// TIA Portal V17 export
// export: Created 2025-03-10T13:10:32.0915737Z, ExportSetting WithDefaults, DisplayName Totally Integrated Automation Portal, DisplayVersion V17 Update 8, DisplayName TIA Portal Openness, DisplayVersion V17 Update 8, DisplayName TIA Portal Version Control Interface, DisplayVersion V17, DisplayName SINAMICS Startdrive Advanced, DisplayVersion V17 SP2, DisplayName SINAMICS Startdrive G110M, G120, G120C, G120D, G120P, G115D, DisplayVersion V17 SP2, DisplayName SINAMICS Startdrive G130, G150, S120, S150, SINAMICS MV, S210, DisplayVersion V17 SP2, DisplayName STEP 7 Professional, DisplayVersion V17 Update 8, DisplayName SINUMERIK ONE STEP 7 Toolbox, DisplayVersion V17 Update 12, DisplayName SINUMERIK 840D sl STEP 7 Toolbox, DisplayVersion V17 Update 12, DisplayName STEP 7 Safety, DisplayVersion V17 Update 6, DisplayName WinCC Advanced, DisplayVersion V17 Update 8
FUNCTION "FC32_CLADDING_AXES" : Void   // FC32, LAD
{ S7_Optimized_Access := 'FALSE' }
AUTHOR : ETXETAR
VERSION : 1.0
// stored: AutoNumber false, IsIECCheckEnabled false, SetENOAutomatically false, UDAEnableTagReadback false
   VAR_TEMP
      O_BLOCKING_DEV_C : Bool;   // OPTION BLOCKING DEVICE FOR C AXIS
      AUX_1 : Real;
      POSITION_TO_GO_AUX : Real;
   END_VAR
   VAR_TEMP   // added for the SCL form of the ladder/FBD networks
      _w1 : Bool;
      _w2 : Bool;
   END_VAR
BEGIN

REGION Network 1: AXIS E10 MOVE AXIS AND FEED HOLD CONDITIONS
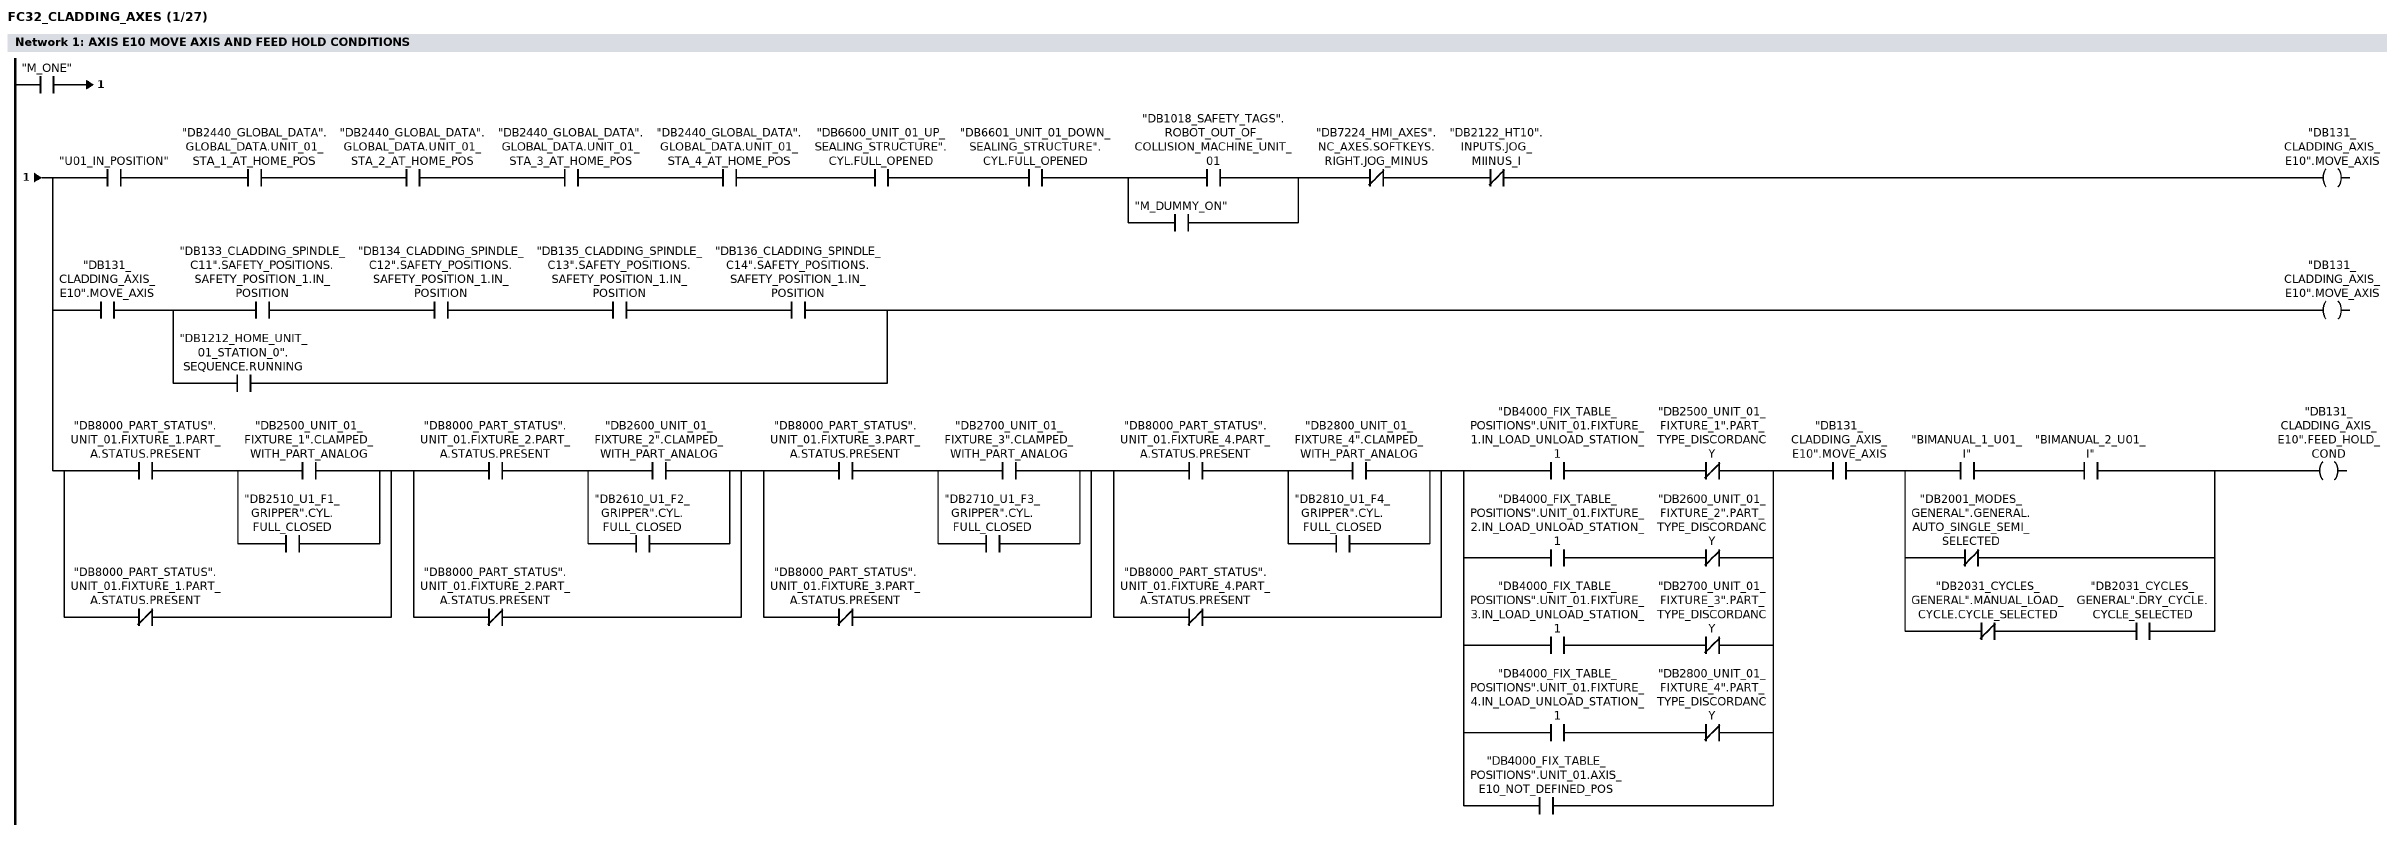
   RUNG wire#powerrail
      Contact( "M_ONE" )
      wire#w1
      Contact( "U01_IN_POSITION" )
      Contact( "DB2440_GLOBAL_DATA".GLOBAL_DATA.UNIT_01_STA_1_AT_HOME_POS )
      Contact( "DB2440_GLOBAL_DATA".GLOBAL_DATA.UNIT_01_STA_2_AT_HOME_POS )
      Contact( "DB2440_GLOBAL_DATA".GLOBAL_DATA.UNIT_01_STA_3_AT_HOME_POS )
      Contact( "DB2440_GLOBAL_DATA".GLOBAL_DATA.UNIT_01_STA_4_AT_HOME_POS )
      Contact( "DB6600_UNIT_01_UP_SEALING_STRUCTURE".CYL.FULL_OPENED )
      Contact( "DB6601_UNIT_01_DOWN_SEALING_STRUCTURE".CYL.FULL_OPENED )
      wire#w2
      Contact( "DB1018_SAFETY_TAGS".ROBOT_OUT_OF_COLLISION_MACHINE_UNIT_01 )
      wire#w3
      I_Contact( "DB7224_HMI_AXES".NC_AXES.SOFTKEYS.RIGHT.JOG_MINUS )
      I_Contact( "DB2122_HT10".INPUTS.JOG_MIINUS_I )
      Coil( "DB131_CLADDING_AXIS_E10".MOVE_AXIS )
   END_RUNG
   RUNG wire#w2
      Contact( "M_DUMMY_ON" )
   END_RUNG wire#w3
   RUNG wire#w1
      Contact( "DB131_CLADDING_AXIS_E10".MOVE_AXIS )
      wire#w4
      Contact( "DB133_CLADDING_SPINDLE_C11".SAFETY_POSITIONS.SAFETY_POSITION_1.IN_POSITION )
      Contact( "DB134_CLADDING_SPINDLE_C12".SAFETY_POSITIONS.SAFETY_POSITION_1.IN_POSITION )
      Contact( "DB135_CLADDING_SPINDLE_C13".SAFETY_POSITIONS.SAFETY_POSITION_1.IN_POSITION )
      Contact( "DB136_CLADDING_SPINDLE_C14".SAFETY_POSITIONS.SAFETY_POSITION_1.IN_POSITION )
      wire#w5
      Coil( "DB131_CLADDING_AXIS_E10".MOVE_AXIS )
   END_RUNG
   RUNG wire#w4
      Contact( "DB1212_HOME_UNIT_01_STATION_0".SEQUENCE.RUNNING )
   END_RUNG wire#w5
   RUNG wire#w1
      Contact( "DB8000_PART_STATUS".UNIT_01.FIXTURE_1.PART_A.STATUS.PRESENT )
      wire#w6
      Contact( "DB2500_UNIT_01_FIXTURE_1".CLAMPED_WITH_PART_ANALOG )
      wire#w7
      Contact( "DB8000_PART_STATUS".UNIT_01.FIXTURE_2.PART_A.STATUS.PRESENT )
      wire#w8
      Contact( "DB2600_UNIT_01_FIXTURE_2".CLAMPED_WITH_PART_ANALOG )
      wire#w9
      Contact( "DB8000_PART_STATUS".UNIT_01.FIXTURE_3.PART_A.STATUS.PRESENT )
      wire#w10
      Contact( "DB2700_UNIT_01_FIXTURE_3".CLAMPED_WITH_PART_ANALOG )
      wire#w11
      Contact( "DB8000_PART_STATUS".UNIT_01.FIXTURE_4.PART_A.STATUS.PRESENT )
      wire#w12
      Contact( "DB2800_UNIT_01_FIXTURE_4".CLAMPED_WITH_PART_ANALOG )
      wire#w13
      Contact( "DB4000_FIX_TABLE_POSITIONS".UNIT_01.FIXTURE_1.IN_LOAD_UNLOAD_STATION_1 )
      I_Contact( "DB2500_UNIT_01_FIXTURE_1".PART_TYPE_DISCORDANCY )
      wire#w14
      Contact( "DB131_CLADDING_AXIS_E10".MOVE_AXIS )
      wire#w15
      Contact( "BIMANUAL_1_U01_I" )
      Contact( "BIMANUAL_2_U01_I" )
      wire#w16
      Coil( "DB131_CLADDING_AXIS_E10".FEED_HOLD_COND )
   END_RUNG
   RUNG wire#w6
      Contact( "DB2510_U1_F1_GRIPPER".CYL.FULL_CLOSED )
   END_RUNG wire#w7
   RUNG wire#w1
      I_Contact( "DB8000_PART_STATUS".UNIT_01.FIXTURE_1.PART_A.STATUS.PRESENT )
   END_RUNG wire#w7
   RUNG wire#w8
      Contact( "DB2610_U1_F2_GRIPPER".CYL.FULL_CLOSED )
   END_RUNG wire#w9
   RUNG wire#w7
      I_Contact( "DB8000_PART_STATUS".UNIT_01.FIXTURE_2.PART_A.STATUS.PRESENT )
   END_RUNG wire#w9
   RUNG wire#w10
      Contact( "DB2710_U1_F3_GRIPPER".CYL.FULL_CLOSED )
   END_RUNG wire#w11
   RUNG wire#w9
      I_Contact( "DB8000_PART_STATUS".UNIT_01.FIXTURE_3.PART_A.STATUS.PRESENT )
   END_RUNG wire#w11
   RUNG wire#w12
      Contact( "DB2810_U1_F4_GRIPPER".CYL.FULL_CLOSED )
   END_RUNG wire#w13
   RUNG wire#w11
      I_Contact( "DB8000_PART_STATUS".UNIT_01.FIXTURE_4.PART_A.STATUS.PRESENT )
   END_RUNG wire#w13
   RUNG wire#w13
      Contact( "DB4000_FIX_TABLE_POSITIONS".UNIT_01.FIXTURE_2.IN_LOAD_UNLOAD_STATION_1 )
      I_Contact( "DB2600_UNIT_01_FIXTURE_2".PART_TYPE_DISCORDANCY )
   END_RUNG wire#w14
   RUNG wire#w13
      Contact( "DB4000_FIX_TABLE_POSITIONS".UNIT_01.FIXTURE_3.IN_LOAD_UNLOAD_STATION_1 )
      I_Contact( "DB2700_UNIT_01_FIXTURE_3".PART_TYPE_DISCORDANCY )
   END_RUNG wire#w14
   RUNG wire#w13
      Contact( "DB4000_FIX_TABLE_POSITIONS".UNIT_01.FIXTURE_4.IN_LOAD_UNLOAD_STATION_1 )
      I_Contact( "DB2800_UNIT_01_FIXTURE_4".PART_TYPE_DISCORDANCY )
   END_RUNG wire#w14
   RUNG wire#w13
      Contact( "DB4000_FIX_TABLE_POSITIONS".UNIT_01.AXIS_E10_NOT_DEFINED_POS )
   END_RUNG wire#w14
   RUNG wire#w15
      I_Contact( "DB2001_MODES_GENERAL".GENERAL.AUTO_SINGLE_SEMI_SELECTED )
   END_RUNG wire#w16
   RUNG wire#w15
      I_Contact( "DB2031_CYCLES_GENERAL".MANUAL_LOAD_CYCLE.CYCLE_SELECTED )
      Contact( "DB2031_CYCLES_GENERAL".DRY_CYCLE.CYCLE_SELECTED )
   END_RUNG wire#w16
   // the same network as SCL:
   "DB131_CLADDING_AXIS_E10".MOVE_AXIS := "M_ONE" AND "U01_IN_POSITION" AND "DB2440_GLOBAL_DATA".GLOBAL_DATA.UNIT_01_STA_1_AT_HOME_POS AND "DB2440_GLOBAL_DATA".GLOBAL_DATA.UNIT_01_STA_2_AT_HOME_POS AND "DB2440_GLOBAL_DATA".GLOBAL_DATA.UNIT_01_STA_3_AT_HOME_POS AND "DB2440_GLOBAL_DATA".GLOBAL_DATA.UNIT_01_STA_4_AT_HOME_POS AND "DB6600_UNIT_01_UP_SEALING_STRUCTURE".CYL.FULL_OPENED AND "DB6601_UNIT_01_DOWN_SEALING_STRUCTURE".CYL.FULL_OPENED AND ("DB1018_SAFETY_TAGS".ROBOT_OUT_OF_COLLISION_MACHINE_UNIT_01 OR "M_DUMMY_ON") AND NOT "DB7224_HMI_AXES".NC_AXES.SOFTKEYS.RIGHT.JOG_MINUS AND NOT "DB2122_HT10".INPUTS.JOG_MIINUS_I;
   "DB131_CLADDING_AXIS_E10".MOVE_AXIS := "M_ONE" AND "DB131_CLADDING_AXIS_E10".MOVE_AXIS AND (("DB133_CLADDING_SPINDLE_C11".SAFETY_POSITIONS.SAFETY_POSITION_1.IN_POSITION AND "DB134_CLADDING_SPINDLE_C12".SAFETY_POSITIONS.SAFETY_POSITION_1.IN_POSITION AND "DB135_CLADDING_SPINDLE_C13".SAFETY_POSITIONS.SAFETY_POSITION_1.IN_POSITION AND "DB136_CLADDING_SPINDLE_C14".SAFETY_POSITIONS.SAFETY_POSITION_1.IN_POSITION) OR "DB1212_HOME_UNIT_01_STATION_0".SEQUENCE.RUNNING);
   "DB131_CLADDING_AXIS_E10".FEED_HOLD_COND := "M_ONE" AND (("DB8000_PART_STATUS".UNIT_01.FIXTURE_1.PART_A.STATUS.PRESENT AND ("DB2500_UNIT_01_FIXTURE_1".CLAMPED_WITH_PART_ANALOG OR "DB2510_U1_F1_GRIPPER".CYL.FULL_CLOSED)) OR NOT "DB8000_PART_STATUS".UNIT_01.FIXTURE_1.PART_A.STATUS.PRESENT) AND (("DB8000_PART_STATUS".UNIT_01.FIXTURE_2.PART_A.STATUS.PRESENT AND ("DB2600_UNIT_01_FIXTURE_2".CLAMPED_WITH_PART_ANALOG OR "DB2610_U1_F2_GRIPPER".CYL.FULL_CLOSED)) OR NOT "DB8000_PART_STATUS".UNIT_01.FIXTURE_2.PART_A.STATUS.PRESENT) AND (("DB8000_PART_STATUS".UNIT_01.FIXTURE_3.PART_A.STATUS.PRESENT AND ("DB2700_UNIT_01_FIXTURE_3".CLAMPED_WITH_PART_ANALOG OR "DB2710_U1_F3_GRIPPER".CYL.FULL_CLOSED)) OR NOT "DB8000_PART_STATUS".UNIT_01.FIXTURE_3.PART_A.STATUS.PRESENT) AND (("DB8000_PART_STATUS".UNIT_01.FIXTURE_4.PART_A.STATUS.PRESENT AND ("DB2800_UNIT_01_FIXTURE_4".CLAMPED_WITH_PART_ANALOG OR "DB2810_U1_F4_GRIPPER".CYL.FULL_CLOSED)) OR NOT "DB8000_PART_STATUS".UNIT_01.FIXTURE_4.PART_A.STATUS.PRESENT) AND (("DB4000_FIX_TABLE_POSITIONS".UNIT_01.FIXTURE_1.IN_LOAD_UNLOAD_STATION_1 AND NOT "DB2500_UNIT_01_FIXTURE_1".PART_TYPE_DISCORDANCY) OR ("DB4000_FIX_TABLE_POSITIONS".UNIT_01.FIXTURE_2.IN_LOAD_UNLOAD_STATION_1 AND NOT "DB2600_UNIT_01_FIXTURE_2".PART_TYPE_DISCORDANCY) OR ("DB4000_FIX_TABLE_POSITIONS".UNIT_01.FIXTURE_3.IN_LOAD_UNLOAD_STATION_1 AND NOT "DB2700_UNIT_01_FIXTURE_3".PART_TYPE_DISCORDANCY) OR ("DB4000_FIX_TABLE_POSITIONS".UNIT_01.FIXTURE_4.IN_LOAD_UNLOAD_STATION_1 AND NOT "DB2800_UNIT_01_FIXTURE_4".PART_TYPE_DISCORDANCY) OR "DB4000_FIX_TABLE_POSITIONS".UNIT_01.AXIS_E10_NOT_DEFINED_POS) AND "DB131_CLADDING_AXIS_E10".MOVE_AXIS AND (("BIMANUAL_1_U01_I" AND "BIMANUAL_2_U01_I") OR NOT "DB2001_MODES_GENERAL".GENERAL.AUTO_SINGLE_SEMI_SELECTED OR (NOT "DB2031_CYCLES_GENERAL".MANUAL_LOAD_CYCLE.CYCLE_SELECTED AND "DB2031_CYCLES_GENERAL".DRY_CYCLE.CYCLE_SELECTED));
END_REGION

REGION Network 2: CALL FB32 AXIS E10
   // 2#0000_0001 OPTIONS 0 BIT 0 MEASURING SYSTEM 2 OPTION
   // 2#0000_0010 OPTIONS 0 BIT 1 ENABLE FC18 OPTION
   // 2#0000_0100 OPTIONS 0 BIT 2 FC18 EXTERNAL POSITION OPTION
   // 2#0000_1000 OPTIONS 0 BIT 3 AXIS B ENABLE FAULTS OPTION
   // 2#0001_0000 OPTIONS 0 BIT 4 SPARE OPTION
   // 2#0010_0000 OPTIONS 0 BIT 5 SPARE OPTION
   // 2#0100_0000 OPTIONS 0 BIT 6 SPARE OPTION
   // 2#1000_0000 OPTIONS 0 BIT 7 SPARE OPTION
   // 
   // 2#0000_0001 OPTIONS 1 BIT 0 AXIS ROLLER OPTION
   // 2#0000_0010 OPTIONS 1 BIT 1 MASTER AXIS OPTION
   // 2#0000_0100 OPTIONS 1 BIT 2 SLAVE AXIS OPTION
   // 2#0000_1000 OPTIONS 1 BIT 3 MASTER-SLAVE AXES INDEPENDENT MOVEMENT WITH HT10 OPTION
   // 2#0001_0000 OPTIONS 1 BIT 4 GANTRY MODE MASTER AXIS OPTION
   // 2#0010_0000 OPTIONS 1 BIT 5 SPARE OPTION
   // 2#0100_0000 OPTIONS 1 BIT 6 SPARE OPTION
   // 2#1000_0000 OPTIONS 1 BIT 7 SPARE OPTION
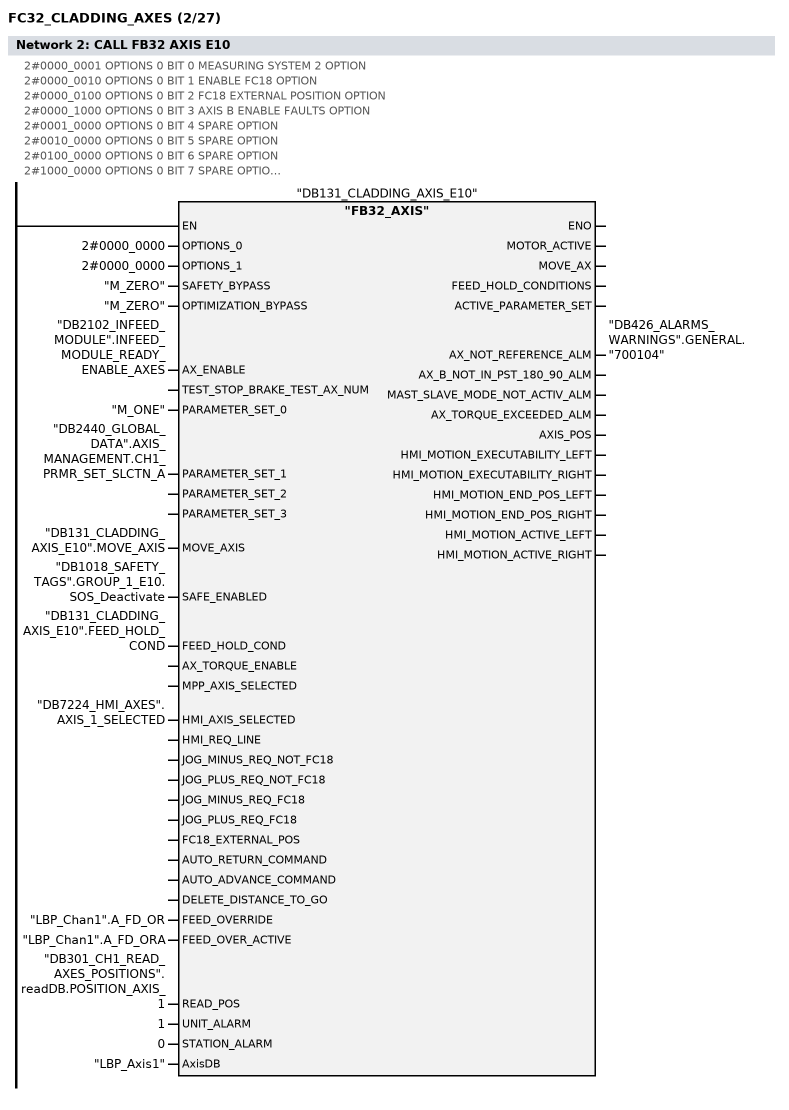
   RUNG wire#powerrail
      "DB131_CLADDING_AXIS_E10"(OPTIONS_0 := 2#0000_0000, OPTIONS_1 := 2#0000_0000, SAFETY_BYPASS := "M_ZERO", OPTIMIZATION_BYPASS := "M_ZERO", AX_ENABLE := "DB2102_INFEED_MODULE".INFEED_MODULE_READY_ENABLE_AXES, TEST_STOP_BRAKE_TEST_AX_NUM :=, PARAMETER_SET_0 := "M_ONE", PARAMETER_SET_1 := "DB2440_GLOBAL_DATA".AXIS_MANAGEMENT.CH1_PRMR_SET_SLCTN_A, PARAMETER_SET_2 :=, PARAMETER_SET_3 :=, MOVE_AXIS := "DB131_CLADDING_AXIS_E10".MOVE_AXIS, SAFE_ENABLED := "DB1018_SAFETY_TAGS".GROUP_1_E10.SOS_Deactivate, FEED_HOLD_COND := "DB131_CLADDING_AXIS_E10".FEED_HOLD_COND, AX_TORQUE_ENABLE :=, MPP_AXIS_SELECTED :=, HMI_AXIS_SELECTED := "DB7224_HMI_AXES".AXIS_1_SELECTED, HMI_REQ_LINE :=, JOG_MINUS_REQ_NOT_FC18 :=, JOG_PLUS_REQ_NOT_FC18 :=, JOG_MINUS_REQ_FC18 :=, JOG_PLUS_REQ_FC18 :=, FC18_EXTERNAL_POS :=, AUTO_RETURN_COMMAND :=, AUTO_ADVANCE_COMMAND :=, DELETE_DISTANCE_TO_GO :=, FEED_OVERRIDE := "LBP_Chan1".A_FD_OR, FEED_OVER_ACTIVE := "LBP_Chan1".A_FD_ORA, READ_POS := "DB301_CH1_READ_AXES_POSITIONS".readDB.POSITION_AXIS_1, UNIT_ALARM := 1, STATION_ALARM := 0, AxisDB := "LBP_Axis1", MOTOR_ACTIVE =>, MOVE_AX =>, FEED_HOLD_CONDITIONS =>, ACTIVE_PARAMETER_SET =>, AX_NOT_REFERENCE_ALM => "DB426_ALARMS_WARNINGS".GENERAL."700104", AX_B_NOT_IN_PST_180_90_ALM =>, MAST_SLAVE_MODE_NOT_ACTIV_ALM =>, AX_TORQUE_EXCEEDED_ALM =>, AXIS_POS =>, HMI_MOTION_EXECUTABILITY_LEFT =>, HMI_MOTION_EXECUTABILITY_RIGHT =>, HMI_MOTION_END_POS_LEFT =>, HMI_MOTION_END_POS_RIGHT =>, HMI_MOTION_ACTIVE_LEFT =>, HMI_MOTION_ACTIVE_RIGHT =>)
   END_RUNG
   // the same network as SCL:
   "DB131_CLADDING_AXIS_E10"(OPTIONS_0 := 2#0000_0000,   // "FB32_AXIS"
                           OPTIONS_1 := 2#0000_0000,
                           SAFETY_BYPASS := "M_ZERO",
                           OPTIMIZATION_BYPASS := "M_ZERO",
                           AX_ENABLE := "DB2102_INFEED_MODULE".INFEED_MODULE_READY_ENABLE_AXES,
                           PARAMETER_SET_0 := "M_ONE",
                           PARAMETER_SET_1 := "DB2440_GLOBAL_DATA".AXIS_MANAGEMENT.CH1_PRMR_SET_SLCTN_A,
                           MOVE_AXIS := "DB131_CLADDING_AXIS_E10".MOVE_AXIS,
                           SAFE_ENABLED := "DB1018_SAFETY_TAGS".GROUP_1_E10.SOS_Deactivate,
                           FEED_HOLD_COND := "DB131_CLADDING_AXIS_E10".FEED_HOLD_COND,
                           HMI_AXIS_SELECTED := "DB7224_HMI_AXES".AXIS_1_SELECTED,
                           FEED_OVERRIDE := "LBP_Chan1".A_FD_OR,
                           FEED_OVER_ACTIVE := "LBP_Chan1".A_FD_ORA,
                           READ_POS := "DB301_CH1_READ_AXES_POSITIONS".readDB.POSITION_AXIS_1,
                           UNIT_ALARM := 1,
                           STATION_ALARM := 0,
                           AxisDB := "LBP_Axis1",
                           AX_NOT_REFERENCE_ALM => "DB426_ALARMS_WARNINGS".GENERAL."700104");
END_REGION

REGION Network 3: AXIS E10 OPERATOR HELP
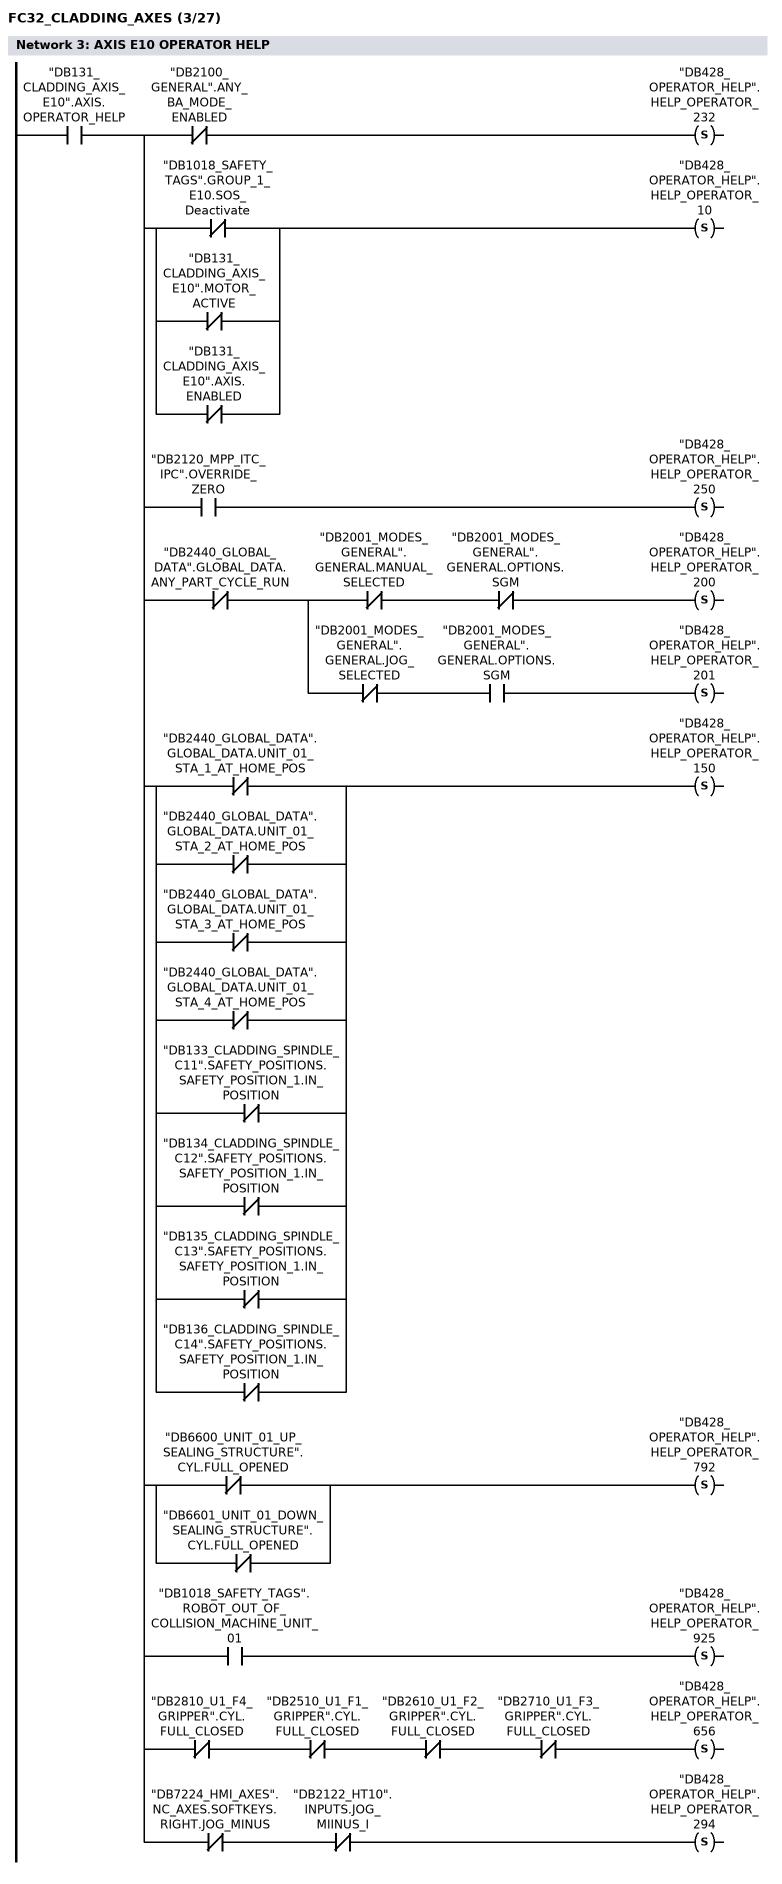
   RUNG wire#powerrail
      Contact( "DB131_CLADDING_AXIS_E10".AXIS.OPERATOR_HELP )
      wire#w1
      I_Contact( "DB2100_GENERAL".ANY_BA_MODE_ENABLED )
      S_Coil( "DB428_OPERATOR_HELP".HELP_OPERATOR_232 )
   END_RUNG
   RUNG wire#w1
      I_Contact( "DB1018_SAFETY_TAGS".GROUP_1_E10.SOS_Deactivate )
      wire#w2
      S_Coil( "DB428_OPERATOR_HELP".HELP_OPERATOR_10 )
   END_RUNG
   RUNG wire#w1
      I_Contact( "DB131_CLADDING_AXIS_E10".MOTOR_ACTIVE )
   END_RUNG wire#w2
   RUNG wire#w1
      I_Contact( "DB131_CLADDING_AXIS_E10".AXIS.ENABLED )
   END_RUNG wire#w2
   RUNG wire#w1
      Contact( "DB2120_MPP_ITC_IPC".OVERRIDE_ZERO )
      S_Coil( "DB428_OPERATOR_HELP".HELP_OPERATOR_250 )
   END_RUNG
   RUNG wire#w1
      I_Contact( "DB2440_GLOBAL_DATA".GLOBAL_DATA.ANY_PART_CYCLE_RUN )
      wire#w3
      I_Contact( "DB2001_MODES_GENERAL".GENERAL.MANUAL_SELECTED )
      I_Contact( "DB2001_MODES_GENERAL".GENERAL.OPTIONS.SGM )
      S_Coil( "DB428_OPERATOR_HELP".HELP_OPERATOR_200 )
   END_RUNG
   RUNG wire#w3
      I_Contact( "DB2001_MODES_GENERAL".GENERAL.JOG_SELECTED )
      Contact( "DB2001_MODES_GENERAL".GENERAL.OPTIONS.SGM )
      S_Coil( "DB428_OPERATOR_HELP".HELP_OPERATOR_201 )
   END_RUNG
   RUNG wire#w1
      I_Contact( "DB2440_GLOBAL_DATA".GLOBAL_DATA.UNIT_01_STA_1_AT_HOME_POS )
      wire#w4
      S_Coil( "DB428_OPERATOR_HELP".HELP_OPERATOR_150 )
   END_RUNG
   RUNG wire#w1
      I_Contact( "DB2440_GLOBAL_DATA".GLOBAL_DATA.UNIT_01_STA_2_AT_HOME_POS )
   END_RUNG wire#w4
   RUNG wire#w1
      I_Contact( "DB2440_GLOBAL_DATA".GLOBAL_DATA.UNIT_01_STA_3_AT_HOME_POS )
   END_RUNG wire#w4
   RUNG wire#w1
      I_Contact( "DB2440_GLOBAL_DATA".GLOBAL_DATA.UNIT_01_STA_4_AT_HOME_POS )
   END_RUNG wire#w4
   RUNG wire#w1
      I_Contact( "DB133_CLADDING_SPINDLE_C11".SAFETY_POSITIONS.SAFETY_POSITION_1.IN_POSITION )
   END_RUNG wire#w4
   RUNG wire#w1
      I_Contact( "DB134_CLADDING_SPINDLE_C12".SAFETY_POSITIONS.SAFETY_POSITION_1.IN_POSITION )
   END_RUNG wire#w4
   RUNG wire#w1
      I_Contact( "DB135_CLADDING_SPINDLE_C13".SAFETY_POSITIONS.SAFETY_POSITION_1.IN_POSITION )
   END_RUNG wire#w4
   RUNG wire#w1
      I_Contact( "DB136_CLADDING_SPINDLE_C14".SAFETY_POSITIONS.SAFETY_POSITION_1.IN_POSITION )
   END_RUNG wire#w4
   RUNG wire#w1
      I_Contact( "DB6600_UNIT_01_UP_SEALING_STRUCTURE".CYL.FULL_OPENED )
      wire#w5
      S_Coil( "DB428_OPERATOR_HELP".HELP_OPERATOR_792 )
   END_RUNG
   RUNG wire#w1
      I_Contact( "DB6601_UNIT_01_DOWN_SEALING_STRUCTURE".CYL.FULL_OPENED )
   END_RUNG wire#w5
   RUNG wire#w1
      Contact( "DB1018_SAFETY_TAGS".ROBOT_OUT_OF_COLLISION_MACHINE_UNIT_01 )
      S_Coil( "DB428_OPERATOR_HELP".HELP_OPERATOR_925 )
   END_RUNG
   RUNG wire#w1
      I_Contact( "DB2810_U1_F4_GRIPPER".CYL.FULL_CLOSED )
      I_Contact( "DB2510_U1_F1_GRIPPER".CYL.FULL_CLOSED )
      I_Contact( "DB2610_U1_F2_GRIPPER".CYL.FULL_CLOSED )
      I_Contact( "DB2710_U1_F3_GRIPPER".CYL.FULL_CLOSED )
      S_Coil( "DB428_OPERATOR_HELP".HELP_OPERATOR_656 )
   END_RUNG
   RUNG wire#w1
      I_Contact( "DB7224_HMI_AXES".NC_AXES.SOFTKEYS.RIGHT.JOG_MINUS )
      I_Contact( "DB2122_HT10".INPUTS.JOG_MIINUS_I )
      S_Coil( "DB428_OPERATOR_HELP".HELP_OPERATOR_294 )
   END_RUNG
   // the same network as SCL:
   IF "DB131_CLADDING_AXIS_E10".AXIS.OPERATOR_HELP AND NOT "DB2100_GENERAL".ANY_BA_MODE_ENABLED THEN
       "DB428_OPERATOR_HELP".HELP_OPERATOR_232 := TRUE;
   END_IF;
   IF "DB131_CLADDING_AXIS_E10".AXIS.OPERATOR_HELP AND (NOT "DB1018_SAFETY_TAGS".GROUP_1_E10.SOS_Deactivate OR NOT "DB131_CLADDING_AXIS_E10".MOTOR_ACTIVE OR NOT "DB131_CLADDING_AXIS_E10".AXIS.ENABLED) THEN
       "DB428_OPERATOR_HELP".HELP_OPERATOR_10 := TRUE;
   END_IF;
   IF "DB131_CLADDING_AXIS_E10".AXIS.OPERATOR_HELP AND "DB2120_MPP_ITC_IPC".OVERRIDE_ZERO THEN
       "DB428_OPERATOR_HELP".HELP_OPERATOR_250 := TRUE;
   END_IF;
   #_w1 := "DB131_CLADDING_AXIS_E10".AXIS.OPERATOR_HELP AND NOT "DB2440_GLOBAL_DATA".GLOBAL_DATA.ANY_PART_CYCLE_RUN;
   IF #_w1 AND NOT "DB2001_MODES_GENERAL".GENERAL.MANUAL_SELECTED AND NOT "DB2001_MODES_GENERAL".GENERAL.OPTIONS.SGM THEN
       "DB428_OPERATOR_HELP".HELP_OPERATOR_200 := TRUE;
   END_IF;
   IF #_w1 AND NOT "DB2001_MODES_GENERAL".GENERAL.JOG_SELECTED AND "DB2001_MODES_GENERAL".GENERAL.OPTIONS.SGM THEN
       "DB428_OPERATOR_HELP".HELP_OPERATOR_201 := TRUE;
   END_IF;
   IF "DB131_CLADDING_AXIS_E10".AXIS.OPERATOR_HELP AND (NOT "DB2440_GLOBAL_DATA".GLOBAL_DATA.UNIT_01_STA_1_AT_HOME_POS OR NOT "DB2440_GLOBAL_DATA".GLOBAL_DATA.UNIT_01_STA_2_AT_HOME_POS OR NOT "DB2440_GLOBAL_DATA".GLOBAL_DATA.UNIT_01_STA_3_AT_HOME_POS OR NOT "DB2440_GLOBAL_DATA".GLOBAL_DATA.UNIT_01_STA_4_AT_HOME_POS OR NOT "DB133_CLADDING_SPINDLE_C11".SAFETY_POSITIONS.SAFETY_POSITION_1.IN_POSITION OR NOT "DB134_CLADDING_SPINDLE_C12".SAFETY_POSITIONS.SAFETY_POSITION_1.IN_POSITION OR NOT "DB135_CLADDING_SPINDLE_C13".SAFETY_POSITIONS.SAFETY_POSITION_1.IN_POSITION OR NOT "DB136_CLADDING_SPINDLE_C14".SAFETY_POSITIONS.SAFETY_POSITION_1.IN_POSITION) THEN
       "DB428_OPERATOR_HELP".HELP_OPERATOR_150 := TRUE;
   END_IF;
   IF "DB131_CLADDING_AXIS_E10".AXIS.OPERATOR_HELP AND (NOT "DB6600_UNIT_01_UP_SEALING_STRUCTURE".CYL.FULL_OPENED OR NOT "DB6601_UNIT_01_DOWN_SEALING_STRUCTURE".CYL.FULL_OPENED) THEN
       "DB428_OPERATOR_HELP".HELP_OPERATOR_792 := TRUE;
   END_IF;
   IF "DB131_CLADDING_AXIS_E10".AXIS.OPERATOR_HELP AND "DB1018_SAFETY_TAGS".ROBOT_OUT_OF_COLLISION_MACHINE_UNIT_01 THEN
       "DB428_OPERATOR_HELP".HELP_OPERATOR_925 := TRUE;
   END_IF;
   IF "DB131_CLADDING_AXIS_E10".AXIS.OPERATOR_HELP AND NOT "DB2810_U1_F4_GRIPPER".CYL.FULL_CLOSED AND NOT "DB2510_U1_F1_GRIPPER".CYL.FULL_CLOSED AND NOT "DB2610_U1_F2_GRIPPER".CYL.FULL_CLOSED AND NOT "DB2710_U1_F3_GRIPPER".CYL.FULL_CLOSED THEN
       "DB428_OPERATOR_HELP".HELP_OPERATOR_656 := TRUE;
   END_IF;
   IF "DB131_CLADDING_AXIS_E10".AXIS.OPERATOR_HELP AND NOT "DB7224_HMI_AXES".NC_AXES.SOFTKEYS.RIGHT.JOG_MINUS AND NOT "DB2122_HT10".INPUTS.JOG_MIINUS_I THEN
       "DB428_OPERATOR_HELP".HELP_OPERATOR_294 := TRUE;
   END_IF;
END_REGION

REGION Network 4: AXIS X13 MOVE AXIS AND FEED HOLD CONDITIONS
   // AÑADIR QUE TODO ESTE CONECTADO
   // DISCO AMARRADO
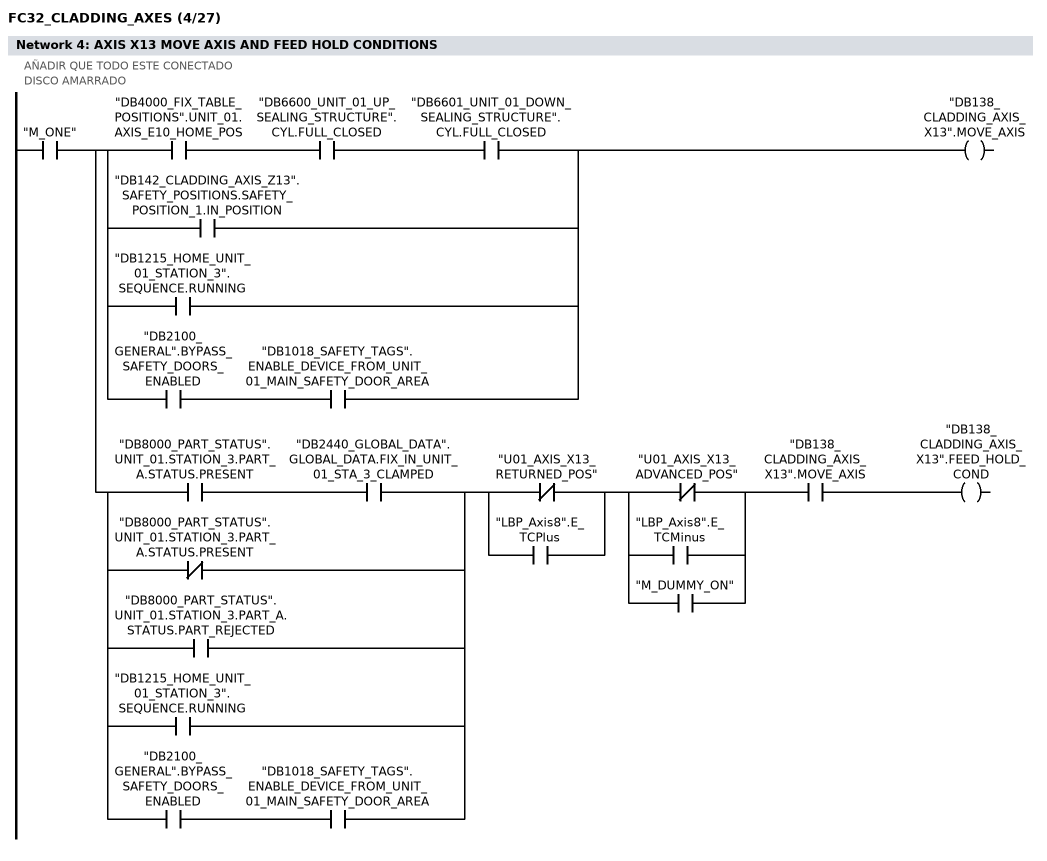
   RUNG wire#powerrail
      Contact( "M_ONE" )
      wire#w1
      Contact( "DB4000_FIX_TABLE_POSITIONS".UNIT_01.AXIS_E10_HOME_POS )
      Contact( "DB6600_UNIT_01_UP_SEALING_STRUCTURE".CYL.FULL_CLOSED )
      Contact( "DB6601_UNIT_01_DOWN_SEALING_STRUCTURE".CYL.FULL_CLOSED )
      wire#w2
      Coil( "DB138_CLADDING_AXIS_X13".MOVE_AXIS )
   END_RUNG
   RUNG wire#w1
      Contact( "DB142_CLADDING_AXIS_Z13".SAFETY_POSITIONS.SAFETY_POSITION_1.IN_POSITION )
   END_RUNG wire#w2
   RUNG wire#w1
      Contact( "DB1215_HOME_UNIT_01_STATION_3".SEQUENCE.RUNNING )
   END_RUNG wire#w2
   RUNG wire#w1
      Contact( "DB2100_GENERAL".BYPASS_SAFETY_DOORS_ENABLED )
      Contact( "DB1018_SAFETY_TAGS".ENABLE_DEVICE_FROM_UNIT_01_MAIN_SAFETY_DOOR_AREA )
   END_RUNG wire#w2
   RUNG wire#w1
      Contact( "DB8000_PART_STATUS".UNIT_01.STATION_3.PART_A.STATUS.PRESENT )
      Contact( "DB2440_GLOBAL_DATA".GLOBAL_DATA.FIX_IN_UNIT_01_STA_3_CLAMPED )
      wire#w3
      I_Contact( "U01_AXIS_X13_RETURNED_POS" )
      wire#w4
      I_Contact( "U01_AXIS_X13_ADVANCED_POS" )
      wire#w5
      Contact( "DB138_CLADDING_AXIS_X13".MOVE_AXIS )
      Coil( "DB138_CLADDING_AXIS_X13".FEED_HOLD_COND )
   END_RUNG
   RUNG wire#w1
      I_Contact( "DB8000_PART_STATUS".UNIT_01.STATION_3.PART_A.STATUS.PRESENT )
   END_RUNG wire#w3
   RUNG wire#w1
      Contact( "DB8000_PART_STATUS".UNIT_01.STATION_3.PART_A.STATUS.PART_REJECTED )
   END_RUNG wire#w3
   RUNG wire#w1
      Contact( "DB1215_HOME_UNIT_01_STATION_3".SEQUENCE.RUNNING )
   END_RUNG wire#w3
   RUNG wire#w1
      Contact( "DB2100_GENERAL".BYPASS_SAFETY_DOORS_ENABLED )
      Contact( "DB1018_SAFETY_TAGS".ENABLE_DEVICE_FROM_UNIT_01_MAIN_SAFETY_DOOR_AREA )
   END_RUNG wire#w3
   RUNG wire#w3
      Contact( "LBP_Axis8".E_TCPlus )
   END_RUNG wire#w4
   RUNG wire#w4
      Contact( "LBP_Axis8".E_TCMinus )
   END_RUNG wire#w5
   RUNG wire#w4
      Contact( "M_DUMMY_ON" )
   END_RUNG wire#w5
   // the same network as SCL:
   "DB138_CLADDING_AXIS_X13".MOVE_AXIS := "M_ONE" AND (("DB4000_FIX_TABLE_POSITIONS".UNIT_01.AXIS_E10_HOME_POS AND "DB6600_UNIT_01_UP_SEALING_STRUCTURE".CYL.FULL_CLOSED AND "DB6601_UNIT_01_DOWN_SEALING_STRUCTURE".CYL.FULL_CLOSED) OR "DB142_CLADDING_AXIS_Z13".SAFETY_POSITIONS.SAFETY_POSITION_1.IN_POSITION OR "DB1215_HOME_UNIT_01_STATION_3".SEQUENCE.RUNNING OR ("DB2100_GENERAL".BYPASS_SAFETY_DOORS_ENABLED AND "DB1018_SAFETY_TAGS".ENABLE_DEVICE_FROM_UNIT_01_MAIN_SAFETY_DOOR_AREA));
   "DB138_CLADDING_AXIS_X13".FEED_HOLD_COND := "M_ONE" AND (("DB8000_PART_STATUS".UNIT_01.STATION_3.PART_A.STATUS.PRESENT AND "DB2440_GLOBAL_DATA".GLOBAL_DATA.FIX_IN_UNIT_01_STA_3_CLAMPED) OR NOT "DB8000_PART_STATUS".UNIT_01.STATION_3.PART_A.STATUS.PRESENT OR "DB8000_PART_STATUS".UNIT_01.STATION_3.PART_A.STATUS.PART_REJECTED OR "DB1215_HOME_UNIT_01_STATION_3".SEQUENCE.RUNNING OR ("DB2100_GENERAL".BYPASS_SAFETY_DOORS_ENABLED AND "DB1018_SAFETY_TAGS".ENABLE_DEVICE_FROM_UNIT_01_MAIN_SAFETY_DOOR_AREA)) AND (NOT "U01_AXIS_X13_RETURNED_POS" OR "LBP_Axis8".E_TCPlus) AND (NOT "U01_AXIS_X13_ADVANCED_POS" OR "LBP_Axis8".E_TCMinus OR "M_DUMMY_ON") AND "DB138_CLADDING_AXIS_X13".MOVE_AXIS;
END_REGION

REGION Network 5: CALL FB32 AXIS X13
   // 2#0000_0001 OPTIONS 0 BIT 0 MEASURING SYSTEM 2 OPTION
   // 2#0000_0010 OPTIONS 0 BIT 1 ENABLE FC18 OPTION
   // 2#0000_0100 OPTIONS 0 BIT 2 FC18 EXTERNAL POSITION OPTION
   // 2#0000_1000 OPTIONS 0 BIT 3 AXIS B ENABLE FAULTS OPTION
   // 2#0001_0000 OPTIONS 0 BIT 4 SPARE OPTION
   // 2#0010_0000 OPTIONS 0 BIT 5 SPARE OPTION
   // 2#0100_0000 OPTIONS 0 BIT 6 SPARE OPTION
   // 2#1000_0000 OPTIONS 0 BIT 7 SPARE OPTION
   // 
   // 2#0000_0001 OPTIONS 1 BIT 0 AXIS ROLLER OPTION
   // 2#0000_0010 OPTIONS 1 BIT 1 MASTER AXIS OPTION
   // 2#0000_0100 OPTIONS 1 BIT 2 SLAVE AXIS OPTION
   // 2#0000_1000 OPTIONS 1 BIT 3 MASTER-SLAVE AXES INDEPENDENT MOVEMENT WITH HT10 OPTION
   // 2#0001_0000 OPTIONS 1 BIT 4 GANTRY MODE MASTER AXIS OPTION
   // 2#0010_0000 OPTIONS 1 BIT 5 SPARE OPTION
   // 2#0100_0000 OPTIONS 1 BIT 6 SPARE OPTION
   // 2#1000_0000 OPTIONS 1 BIT 7 SPARE OPTION
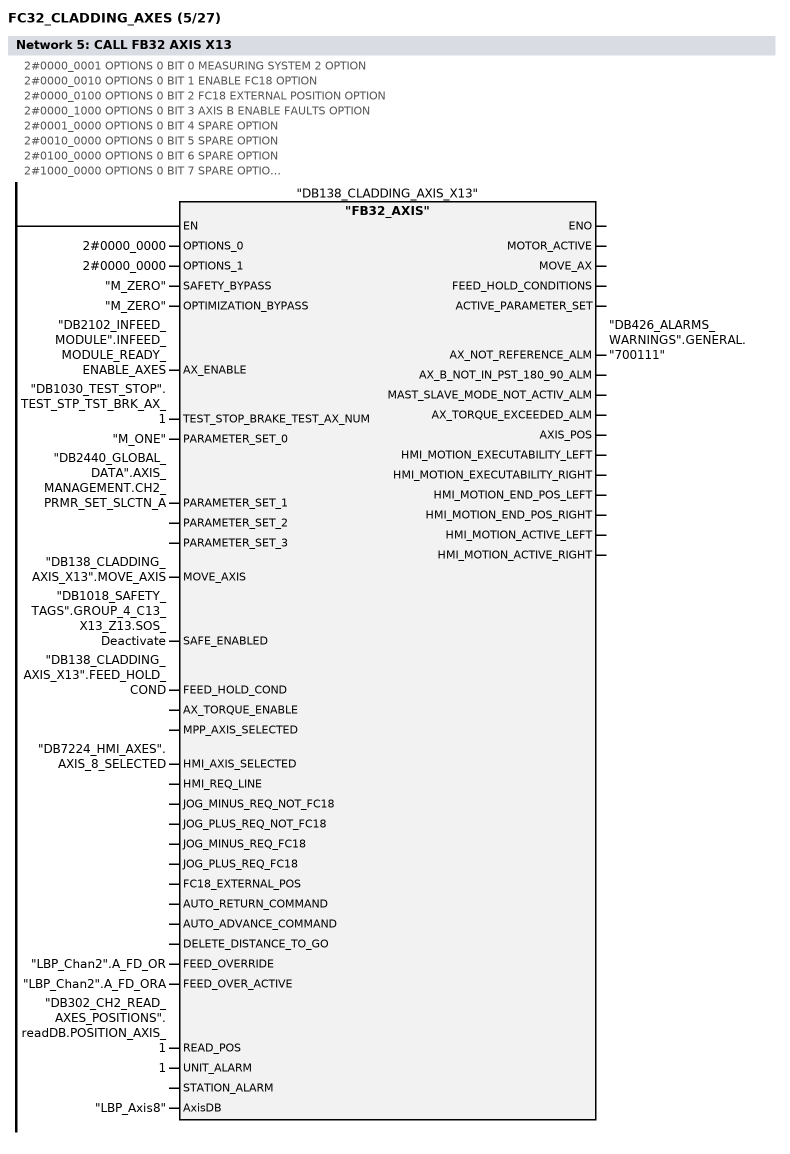
   RUNG wire#powerrail
      "DB138_CLADDING_AXIS_X13"(OPTIONS_0 := 2#0000_0000, OPTIONS_1 := 2#0000_0000, SAFETY_BYPASS := "M_ZERO", OPTIMIZATION_BYPASS := "M_ZERO", AX_ENABLE := "DB2102_INFEED_MODULE".INFEED_MODULE_READY_ENABLE_AXES, TEST_STOP_BRAKE_TEST_AX_NUM := "DB1030_TEST_STOP".TEST_STP_TST_BRK_AX_1, PARAMETER_SET_0 := "M_ONE", PARAMETER_SET_1 := "DB2440_GLOBAL_DATA".AXIS_MANAGEMENT.CH2_PRMR_SET_SLCTN_A, PARAMETER_SET_2 :=, PARAMETER_SET_3 :=, MOVE_AXIS := "DB138_CLADDING_AXIS_X13".MOVE_AXIS, SAFE_ENABLED := "DB1018_SAFETY_TAGS".GROUP_4_C13_X13_Z13.SOS_Deactivate, FEED_HOLD_COND := "DB138_CLADDING_AXIS_X13".FEED_HOLD_COND, AX_TORQUE_ENABLE :=, MPP_AXIS_SELECTED :=, HMI_AXIS_SELECTED := "DB7224_HMI_AXES".AXIS_8_SELECTED, HMI_REQ_LINE :=, JOG_MINUS_REQ_NOT_FC18 :=, JOG_PLUS_REQ_NOT_FC18 :=, JOG_MINUS_REQ_FC18 :=, JOG_PLUS_REQ_FC18 :=, FC18_EXTERNAL_POS :=, AUTO_RETURN_COMMAND :=, AUTO_ADVANCE_COMMAND :=, DELETE_DISTANCE_TO_GO :=, FEED_OVERRIDE := "LBP_Chan2".A_FD_OR, FEED_OVER_ACTIVE := "LBP_Chan2".A_FD_ORA, READ_POS := "DB302_CH2_READ_AXES_POSITIONS".readDB.POSITION_AXIS_1, UNIT_ALARM := 1, STATION_ALARM :=, AxisDB := "LBP_Axis8", MOTOR_ACTIVE =>, MOVE_AX =>, FEED_HOLD_CONDITIONS =>, ACTIVE_PARAMETER_SET =>, AX_NOT_REFERENCE_ALM => "DB426_ALARMS_WARNINGS".GENERAL."700111", AX_B_NOT_IN_PST_180_90_ALM =>, MAST_SLAVE_MODE_NOT_ACTIV_ALM =>, AX_TORQUE_EXCEEDED_ALM =>, AXIS_POS =>, HMI_MOTION_EXECUTABILITY_LEFT =>, HMI_MOTION_EXECUTABILITY_RIGHT =>, HMI_MOTION_END_POS_LEFT =>, HMI_MOTION_END_POS_RIGHT =>, HMI_MOTION_ACTIVE_LEFT =>, HMI_MOTION_ACTIVE_RIGHT =>)
   END_RUNG
   // the same network as SCL:
   "DB138_CLADDING_AXIS_X13"(OPTIONS_0 := 2#0000_0000,   // "FB32_AXIS"
                           OPTIONS_1 := 2#0000_0000,
                           SAFETY_BYPASS := "M_ZERO",
                           OPTIMIZATION_BYPASS := "M_ZERO",
                           AX_ENABLE := "DB2102_INFEED_MODULE".INFEED_MODULE_READY_ENABLE_AXES,
                           TEST_STOP_BRAKE_TEST_AX_NUM := "DB1030_TEST_STOP".TEST_STP_TST_BRK_AX_1,
                           PARAMETER_SET_0 := "M_ONE",
                           PARAMETER_SET_1 := "DB2440_GLOBAL_DATA".AXIS_MANAGEMENT.CH2_PRMR_SET_SLCTN_A,
                           MOVE_AXIS := "DB138_CLADDING_AXIS_X13".MOVE_AXIS,
                           SAFE_ENABLED := "DB1018_SAFETY_TAGS".GROUP_4_C13_X13_Z13.SOS_Deactivate,
                           FEED_HOLD_COND := "DB138_CLADDING_AXIS_X13".FEED_HOLD_COND,
                           HMI_AXIS_SELECTED := "DB7224_HMI_AXES".AXIS_8_SELECTED,
                           FEED_OVERRIDE := "LBP_Chan2".A_FD_OR,
                           FEED_OVER_ACTIVE := "LBP_Chan2".A_FD_ORA,
                           READ_POS := "DB302_CH2_READ_AXES_POSITIONS".readDB.POSITION_AXIS_1,
                           UNIT_ALARM := 1,
                           AxisDB := "LBP_Axis8",
                           AX_NOT_REFERENCE_ALM => "DB426_ALARMS_WARNINGS".GENERAL."700111");
END_REGION

REGION Network 6: AXIS X13 OPERATOR HELP
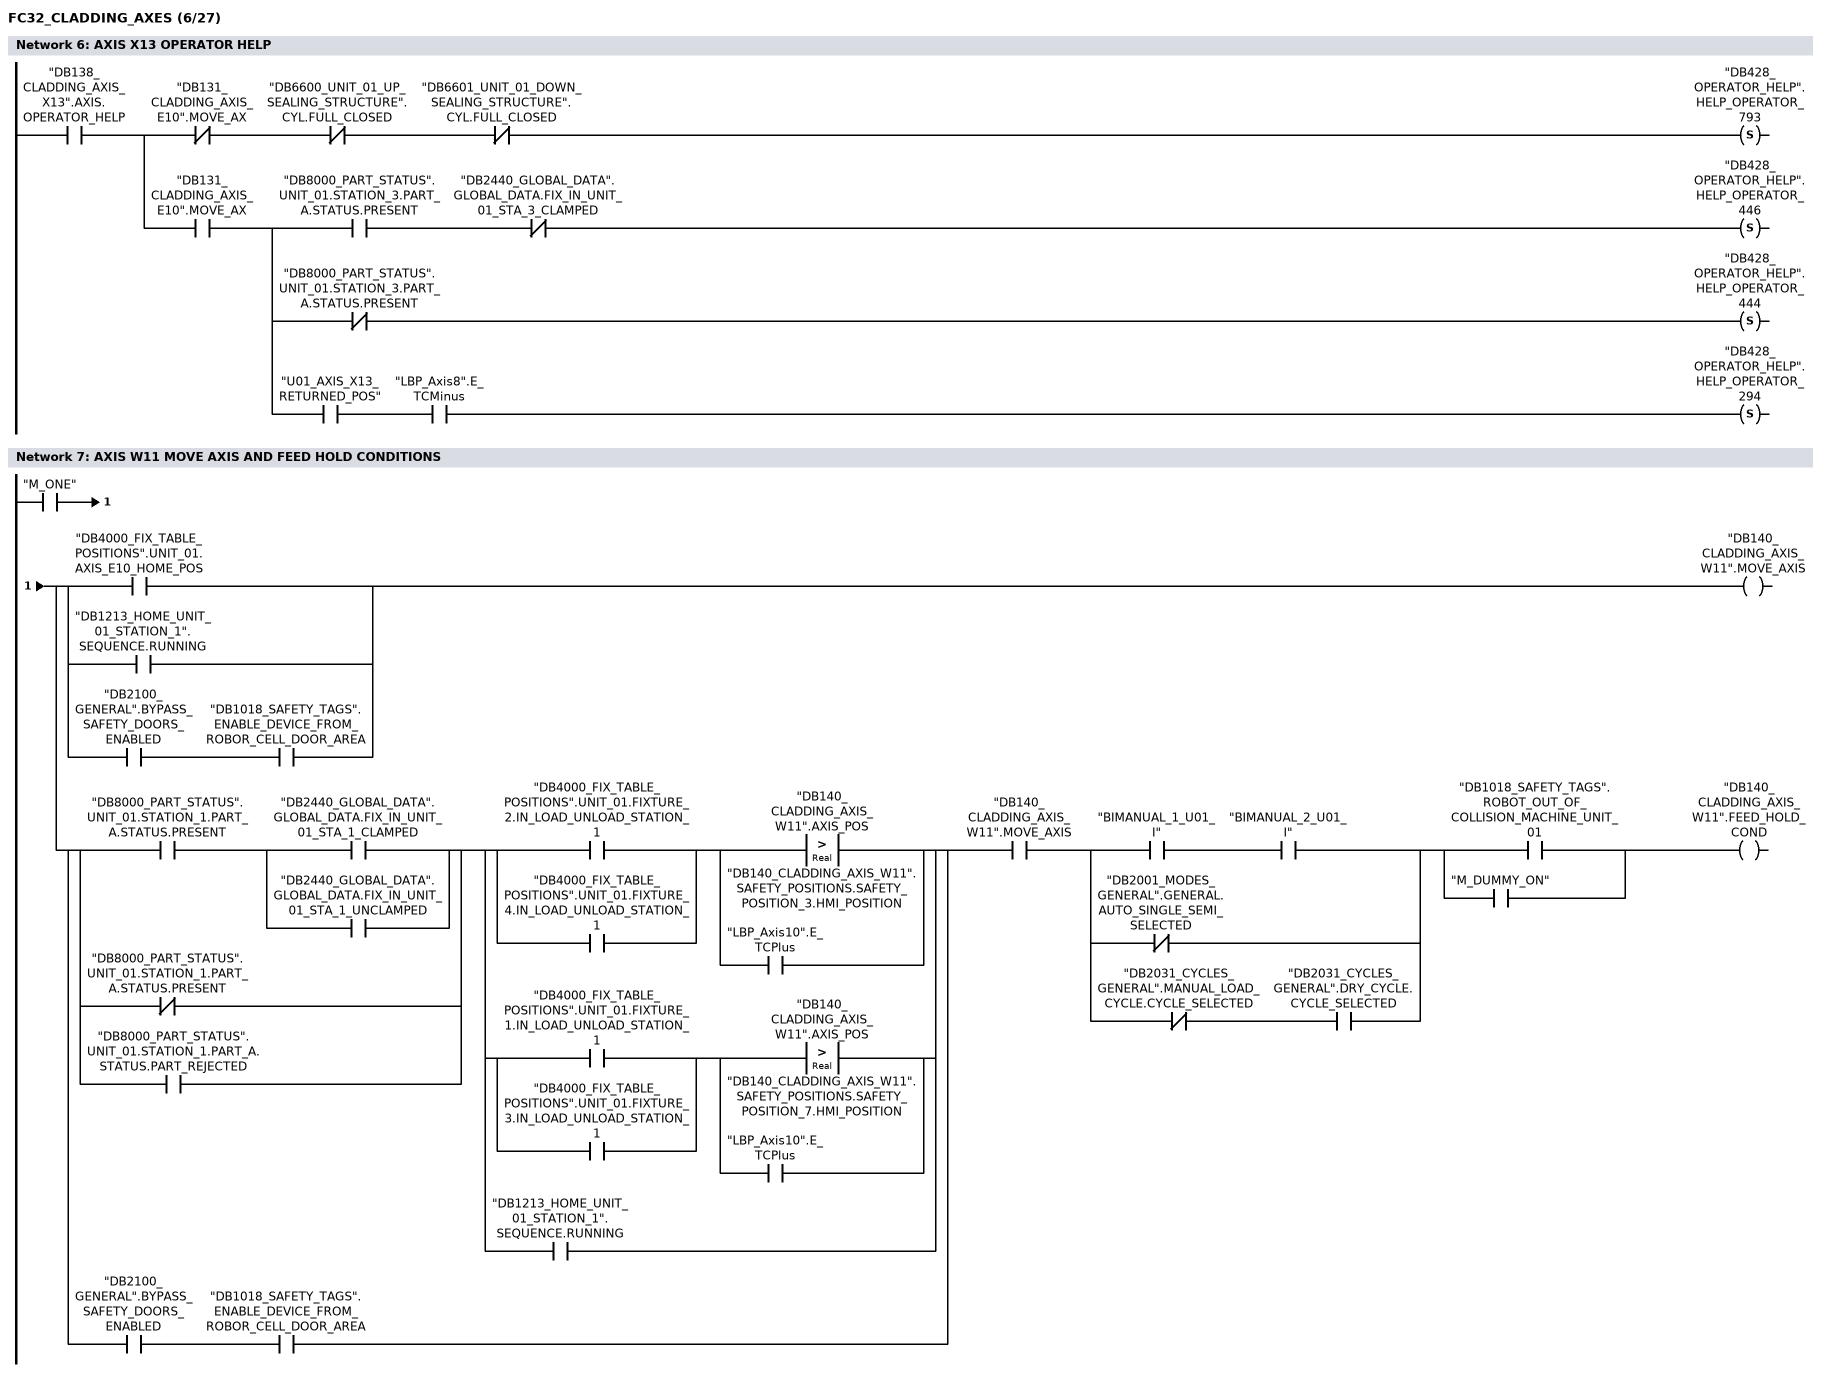
   RUNG wire#powerrail
      Contact( "DB138_CLADDING_AXIS_X13".AXIS.OPERATOR_HELP )
      wire#w1
      I_Contact( "DB131_CLADDING_AXIS_E10".MOVE_AX )
      I_Contact( "DB6600_UNIT_01_UP_SEALING_STRUCTURE".CYL.FULL_CLOSED )
      I_Contact( "DB6601_UNIT_01_DOWN_SEALING_STRUCTURE".CYL.FULL_CLOSED )
      S_Coil( "DB428_OPERATOR_HELP".HELP_OPERATOR_793 )
   END_RUNG
   RUNG wire#w1
      Contact( "DB131_CLADDING_AXIS_E10".MOVE_AX )
      wire#w2
      Contact( "DB8000_PART_STATUS".UNIT_01.STATION_3.PART_A.STATUS.PRESENT )
      I_Contact( "DB2440_GLOBAL_DATA".GLOBAL_DATA.FIX_IN_UNIT_01_STA_3_CLAMPED )
      S_Coil( "DB428_OPERATOR_HELP".HELP_OPERATOR_446 )
   END_RUNG
   RUNG wire#w2
      I_Contact( "DB8000_PART_STATUS".UNIT_01.STATION_3.PART_A.STATUS.PRESENT )
      S_Coil( "DB428_OPERATOR_HELP".HELP_OPERATOR_444 )
   END_RUNG
   RUNG wire#w2
      Contact( "U01_AXIS_X13_RETURNED_POS" )
      Contact( "LBP_Axis8".E_TCMinus )
      S_Coil( "DB428_OPERATOR_HELP".HELP_OPERATOR_294 )
   END_RUNG
   // the same network as SCL:
   IF "DB138_CLADDING_AXIS_X13".AXIS.OPERATOR_HELP AND NOT "DB131_CLADDING_AXIS_E10".MOVE_AX AND NOT "DB6600_UNIT_01_UP_SEALING_STRUCTURE".CYL.FULL_CLOSED AND NOT "DB6601_UNIT_01_DOWN_SEALING_STRUCTURE".CYL.FULL_CLOSED THEN
       "DB428_OPERATOR_HELP".HELP_OPERATOR_793 := TRUE;
   END_IF;
   #_w1 := "DB138_CLADDING_AXIS_X13".AXIS.OPERATOR_HELP AND "DB131_CLADDING_AXIS_E10".MOVE_AX;
   IF #_w1 AND "DB8000_PART_STATUS".UNIT_01.STATION_3.PART_A.STATUS.PRESENT AND NOT "DB2440_GLOBAL_DATA".GLOBAL_DATA.FIX_IN_UNIT_01_STA_3_CLAMPED THEN
       "DB428_OPERATOR_HELP".HELP_OPERATOR_446 := TRUE;
   END_IF;
   IF #_w1 AND NOT "DB8000_PART_STATUS".UNIT_01.STATION_3.PART_A.STATUS.PRESENT THEN
       "DB428_OPERATOR_HELP".HELP_OPERATOR_444 := TRUE;
   END_IF;
   IF #_w1 AND "U01_AXIS_X13_RETURNED_POS" AND "LBP_Axis8".E_TCMinus THEN
       "DB428_OPERATOR_HELP".HELP_OPERATOR_294 := TRUE;
   END_IF;
END_REGION

REGION Network 7: AXIS W11 MOVE AXIS AND FEED HOLD CONDITIONS
   RUNG wire#powerrail
      Contact( "M_ONE" )
      wire#w1
      Contact( "DB4000_FIX_TABLE_POSITIONS".UNIT_01.AXIS_E10_HOME_POS )
      wire#w2
      Coil( "DB140_CLADDING_AXIS_W11".MOVE_AXIS )
   END_RUNG
   RUNG wire#w1
      Contact( "DB1213_HOME_UNIT_01_STATION_1".SEQUENCE.RUNNING )
   END_RUNG wire#w2
   RUNG wire#w1
      Contact( "DB2100_GENERAL".BYPASS_SAFETY_DOORS_ENABLED )
      Contact( "DB1018_SAFETY_TAGS".ENABLE_DEVICE_FROM_ROBOR_CELL_DOOR_AREA )
   END_RUNG wire#w2
   RUNG wire#w1
      Contact( "DB8000_PART_STATUS".UNIT_01.STATION_1.PART_A.STATUS.PRESENT )
      wire#w3
      Contact( "DB2440_GLOBAL_DATA".GLOBAL_DATA.FIX_IN_UNIT_01_STA_1_CLAMPED )
      wire#w4
      Contact( "DB4000_FIX_TABLE_POSITIONS".UNIT_01.FIXTURE_2.IN_LOAD_UNLOAD_STATION_1 )
      wire#w5
      { S7_Templates := "SrcType := Real" } GT_Contact(in1 := "DB140_CLADDING_AXIS_W11".AXIS_POS, in2 := "DB140_CLADDING_AXIS_W11".SAFETY_POSITIONS.SAFETY_POSITION_3.HMI_POSITION)
      wire#w6
      Contact( "DB140_CLADDING_AXIS_W11".MOVE_AXIS )
      wire#w8
      Contact( "BIMANUAL_1_U01_I" )
      Contact( "BIMANUAL_2_U01_I" )
      wire#w9
      Contact( "DB1018_SAFETY_TAGS".ROBOT_OUT_OF_COLLISION_MACHINE_UNIT_01 )
      wire#w10
      Coil( "DB140_CLADDING_AXIS_W11".FEED_HOLD_COND )
   END_RUNG
   RUNG wire#w3
      Contact( "DB2440_GLOBAL_DATA".GLOBAL_DATA.FIX_IN_UNIT_01_STA_1_UNCLAMPED )
   END_RUNG wire#w4
   RUNG wire#w1
      I_Contact( "DB8000_PART_STATUS".UNIT_01.STATION_1.PART_A.STATUS.PRESENT )
   END_RUNG wire#w4
   RUNG wire#w1
      Contact( "DB8000_PART_STATUS".UNIT_01.STATION_1.PART_A.STATUS.PART_REJECTED )
   END_RUNG wire#w4
   RUNG wire#w4
      Contact( "DB4000_FIX_TABLE_POSITIONS".UNIT_01.FIXTURE_4.IN_LOAD_UNLOAD_STATION_1 )
   END_RUNG wire#w5
   RUNG wire#w5
      Contact( "LBP_Axis10".E_TCPlus )
   END_RUNG wire#w6
   RUNG wire#w4
      Contact( "DB4000_FIX_TABLE_POSITIONS".UNIT_01.FIXTURE_1.IN_LOAD_UNLOAD_STATION_1 )
      wire#w7
      { S7_Templates := "SrcType := Real" } GT_Contact(in1 := "DB140_CLADDING_AXIS_W11".AXIS_POS, in2 := "DB140_CLADDING_AXIS_W11".SAFETY_POSITIONS.SAFETY_POSITION_7.HMI_POSITION)
   END_RUNG wire#w6
   RUNG wire#w4
      Contact( "DB4000_FIX_TABLE_POSITIONS".UNIT_01.FIXTURE_3.IN_LOAD_UNLOAD_STATION_1 )
   END_RUNG wire#w7
   RUNG wire#w7
      Contact( "LBP_Axis10".E_TCPlus )
   END_RUNG wire#w6
   RUNG wire#w4
      Contact( "DB1213_HOME_UNIT_01_STATION_1".SEQUENCE.RUNNING )
   END_RUNG wire#w6
   RUNG wire#w1
      Contact( "DB2100_GENERAL".BYPASS_SAFETY_DOORS_ENABLED )
      Contact( "DB1018_SAFETY_TAGS".ENABLE_DEVICE_FROM_ROBOR_CELL_DOOR_AREA )
   END_RUNG wire#w6
   RUNG wire#w8
      I_Contact( "DB2001_MODES_GENERAL".GENERAL.AUTO_SINGLE_SEMI_SELECTED )
   END_RUNG wire#w9
   RUNG wire#w8
      I_Contact( "DB2031_CYCLES_GENERAL".MANUAL_LOAD_CYCLE.CYCLE_SELECTED )
      Contact( "DB2031_CYCLES_GENERAL".DRY_CYCLE.CYCLE_SELECTED )
   END_RUNG wire#w9
   RUNG wire#w9
      Contact( "M_DUMMY_ON" )
   END_RUNG wire#w10
   // the same network as SCL:
   "DB140_CLADDING_AXIS_W11".MOVE_AXIS := "M_ONE" AND ("DB4000_FIX_TABLE_POSITIONS".UNIT_01.AXIS_E10_HOME_POS OR "DB1213_HOME_UNIT_01_STATION_1".SEQUENCE.RUNNING OR ("DB2100_GENERAL".BYPASS_SAFETY_DOORS_ENABLED AND "DB1018_SAFETY_TAGS".ENABLE_DEVICE_FROM_ROBOR_CELL_DOOR_AREA));
   "DB140_CLADDING_AXIS_W11".FEED_HOLD_COND := "M_ONE" AND (((("DB8000_PART_STATUS".UNIT_01.STATION_1.PART_A.STATUS.PRESENT AND ("DB2440_GLOBAL_DATA".GLOBAL_DATA.FIX_IN_UNIT_01_STA_1_CLAMPED OR "DB2440_GLOBAL_DATA".GLOBAL_DATA.FIX_IN_UNIT_01_STA_1_UNCLAMPED)) OR NOT "DB8000_PART_STATUS".UNIT_01.STATION_1.PART_A.STATUS.PRESENT OR "DB8000_PART_STATUS".UNIT_01.STATION_1.PART_A.STATUS.PART_REJECTED) AND ((("DB4000_FIX_TABLE_POSITIONS".UNIT_01.FIXTURE_2.IN_LOAD_UNLOAD_STATION_1 OR "DB4000_FIX_TABLE_POSITIONS".UNIT_01.FIXTURE_4.IN_LOAD_UNLOAD_STATION_1) AND (("DB140_CLADDING_AXIS_W11".AXIS_POS > "DB140_CLADDING_AXIS_W11".SAFETY_POSITIONS.SAFETY_POSITION_3.HMI_POSITION) OR "LBP_Axis10".E_TCPlus)) OR (("DB4000_FIX_TABLE_POSITIONS".UNIT_01.FIXTURE_1.IN_LOAD_UNLOAD_STATION_1 OR "DB4000_FIX_TABLE_POSITIONS".UNIT_01.FIXTURE_3.IN_LOAD_UNLOAD_STATION_1) AND (("DB140_CLADDING_AXIS_W11".AXIS_POS > "DB140_CLADDING_AXIS_W11".SAFETY_POSITIONS.SAFETY_POSITION_7.HMI_POSITION) OR "LBP_Axis10".E_TCPlus)) OR "DB1213_HOME_UNIT_01_STATION_1".SEQUENCE.RUNNING)) OR ("DB2100_GENERAL".BYPASS_SAFETY_DOORS_ENABLED AND "DB1018_SAFETY_TAGS".ENABLE_DEVICE_FROM_ROBOR_CELL_DOOR_AREA)) AND "DB140_CLADDING_AXIS_W11".MOVE_AXIS AND (("BIMANUAL_1_U01_I" AND "BIMANUAL_2_U01_I") OR NOT "DB2001_MODES_GENERAL".GENERAL.AUTO_SINGLE_SEMI_SELECTED OR (NOT "DB2031_CYCLES_GENERAL".MANUAL_LOAD_CYCLE.CYCLE_SELECTED AND "DB2031_CYCLES_GENERAL".DRY_CYCLE.CYCLE_SELECTED)) AND ("DB1018_SAFETY_TAGS".ROBOT_OUT_OF_COLLISION_MACHINE_UNIT_01 OR "M_DUMMY_ON");
END_REGION

REGION Network 8: CALL FB32 AXIS W11
   // 2#0000_0001 OPTIONS 0 BIT 0 MEASURING SYSTEM 2 OPTION
   // 2#0000_0010 OPTIONS 0 BIT 1 ENABLE FC18 OPTION
   // 2#0000_0100 OPTIONS 0 BIT 2 FC18 EXTERNAL POSITION OPTION
   // 2#0000_1000 OPTIONS 0 BIT 3 AXIS B ENABLE FAULTS OPTION
   // 2#0001_0000 OPTIONS 0 BIT 4 SPARE OPTION
   // 2#0010_0000 OPTIONS 0 BIT 5 SPARE OPTION
   // 2#0100_0000 OPTIONS 0 BIT 6 SPARE OPTION
   // 2#1000_0000 OPTIONS 0 BIT 7 SPARE OPTION
   // 
   // 2#0000_0001 OPTIONS 1 BIT 0 AXIS ROLLER OPTION
   // 2#0000_0010 OPTIONS 1 BIT 1 MASTER AXIS OPTION
   // 2#0000_0100 OPTIONS 1 BIT 2 SLAVE AXIS OPTION
   // 2#0000_1000 OPTIONS 1 BIT 3 MASTER-SLAVE AXES INDEPENDENT MOVEMENT WITH HT10 OPTION
   // 2#0001_0000 OPTIONS 1 BIT 4 GANTRY MODE MASTER AXIS OPTION
   // 2#0010_0000 OPTIONS 1 BIT 5 SPARE OPTION
   // 2#0100_0000 OPTIONS 1 BIT 6 SPARE OPTION
   // 2#1000_0000 OPTIONS 1 BIT 7 SPARE OPTION
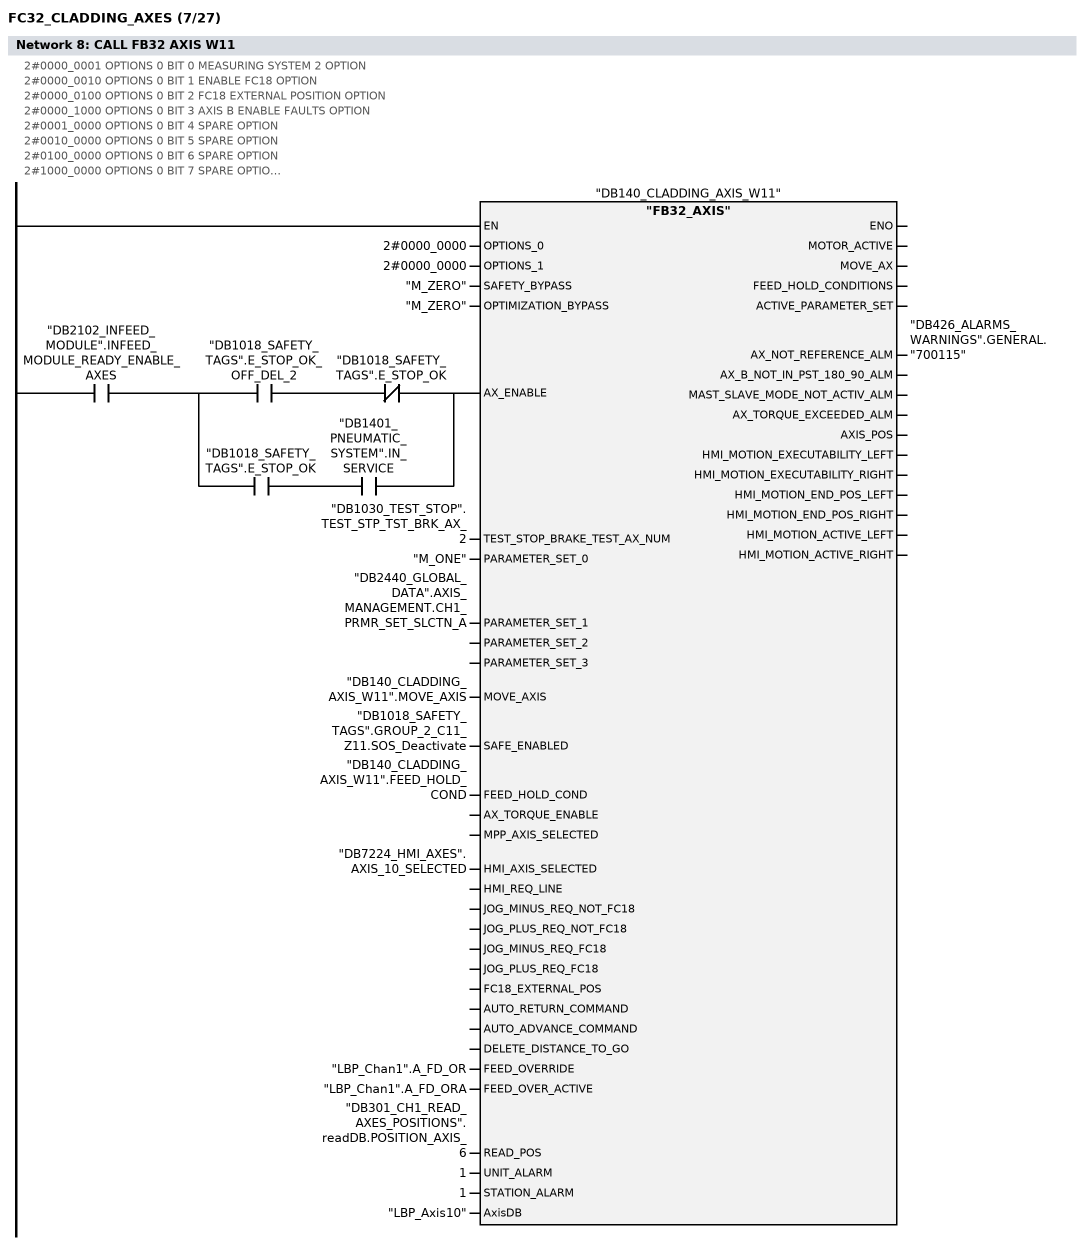
   RUNG wire#powerrail
      "DB140_CLADDING_AXIS_W11"(AX_ENABLE := wire#w2, OPTIONS_0 := 2#0000_0000, OPTIONS_1 := 2#0000_0000, SAFETY_BYPASS := "M_ZERO", OPTIMIZATION_BYPASS := "M_ZERO", TEST_STOP_BRAKE_TEST_AX_NUM := "DB1030_TEST_STOP".TEST_STP_TST_BRK_AX_2, PARAMETER_SET_0 := "M_ONE", PARAMETER_SET_1 := "DB2440_GLOBAL_DATA".AXIS_MANAGEMENT.CH1_PRMR_SET_SLCTN_A, PARAMETER_SET_2 :=, PARAMETER_SET_3 :=, MOVE_AXIS := "DB140_CLADDING_AXIS_W11".MOVE_AXIS, SAFE_ENABLED := "DB1018_SAFETY_TAGS".GROUP_2_C11_Z11.SOS_Deactivate, FEED_HOLD_COND := "DB140_CLADDING_AXIS_W11".FEED_HOLD_COND, AX_TORQUE_ENABLE :=, MPP_AXIS_SELECTED :=, HMI_AXIS_SELECTED := "DB7224_HMI_AXES".AXIS_10_SELECTED, HMI_REQ_LINE :=, JOG_MINUS_REQ_NOT_FC18 :=, JOG_PLUS_REQ_NOT_FC18 :=, JOG_MINUS_REQ_FC18 :=, JOG_PLUS_REQ_FC18 :=, FC18_EXTERNAL_POS :=, AUTO_RETURN_COMMAND :=, AUTO_ADVANCE_COMMAND :=, DELETE_DISTANCE_TO_GO :=, FEED_OVERRIDE := "LBP_Chan1".A_FD_OR, FEED_OVER_ACTIVE := "LBP_Chan1".A_FD_ORA, READ_POS := "DB301_CH1_READ_AXES_POSITIONS".readDB.POSITION_AXIS_6, UNIT_ALARM := 1, STATION_ALARM := 1, AxisDB := "LBP_Axis10", MOTOR_ACTIVE =>, MOVE_AX =>, FEED_HOLD_CONDITIONS =>, ACTIVE_PARAMETER_SET =>, AX_NOT_REFERENCE_ALM => "DB426_ALARMS_WARNINGS".GENERAL."700115", AX_B_NOT_IN_PST_180_90_ALM =>, MAST_SLAVE_MODE_NOT_ACTIV_ALM =>, AX_TORQUE_EXCEEDED_ALM =>, AXIS_POS =>, HMI_MOTION_EXECUTABILITY_LEFT =>, HMI_MOTION_EXECUTABILITY_RIGHT =>, HMI_MOTION_END_POS_LEFT =>, HMI_MOTION_END_POS_RIGHT =>, HMI_MOTION_ACTIVE_LEFT =>, HMI_MOTION_ACTIVE_RIGHT =>)
   END_RUNG
   RUNG wire#powerrail
      Contact( "DB2102_INFEED_MODULE".INFEED_MODULE_READY_ENABLE_AXES )
      wire#w1
      Contact( "DB1018_SAFETY_TAGS".E_STOP_OK_OFF_DEL_2 )
      I_Contact( "DB1018_SAFETY_TAGS".E_STOP_OK )
   END_RUNG wire#w2
   RUNG wire#w1
      Contact( "DB1018_SAFETY_TAGS".E_STOP_OK )
      Contact( "DB1401_PNEUMATIC_SYSTEM".IN_SERVICE )
   END_RUNG wire#w2
   // the same network as SCL:
   "DB140_CLADDING_AXIS_W11"(OPTIONS_0 := 2#0000_0000,   // "FB32_AXIS"
                           OPTIONS_1 := 2#0000_0000,
                           SAFETY_BYPASS := "M_ZERO",
                           OPTIMIZATION_BYPASS := "M_ZERO",
                           AX_ENABLE := "DB2102_INFEED_MODULE".INFEED_MODULE_READY_ENABLE_AXES AND (("DB1018_SAFETY_TAGS".E_STOP_OK_OFF_DEL_2 AND NOT "DB1018_SAFETY_TAGS".E_STOP_OK) OR ("DB1018_SAFETY_TAGS".E_STOP_OK AND "DB1401_PNEUMATIC_SYSTEM".IN_SERVICE)),
                           TEST_STOP_BRAKE_TEST_AX_NUM := "DB1030_TEST_STOP".TEST_STP_TST_BRK_AX_2,
                           PARAMETER_SET_0 := "M_ONE",
                           PARAMETER_SET_1 := "DB2440_GLOBAL_DATA".AXIS_MANAGEMENT.CH1_PRMR_SET_SLCTN_A,
                           MOVE_AXIS := "DB140_CLADDING_AXIS_W11".MOVE_AXIS,
                           SAFE_ENABLED := "DB1018_SAFETY_TAGS".GROUP_2_C11_Z11.SOS_Deactivate,
                           FEED_HOLD_COND := "DB140_CLADDING_AXIS_W11".FEED_HOLD_COND,
                           HMI_AXIS_SELECTED := "DB7224_HMI_AXES".AXIS_10_SELECTED,
                           FEED_OVERRIDE := "LBP_Chan1".A_FD_OR,
                           FEED_OVER_ACTIVE := "LBP_Chan1".A_FD_ORA,
                           READ_POS := "DB301_CH1_READ_AXES_POSITIONS".readDB.POSITION_AXIS_6,
                           UNIT_ALARM := 1,
                           STATION_ALARM := 1,
                           AxisDB := "LBP_Axis10",
                           AX_NOT_REFERENCE_ALM => "DB426_ALARMS_WARNINGS".GENERAL."700115");
END_REGION

REGION Network 9: AXIS W11 OPERATOR HELP
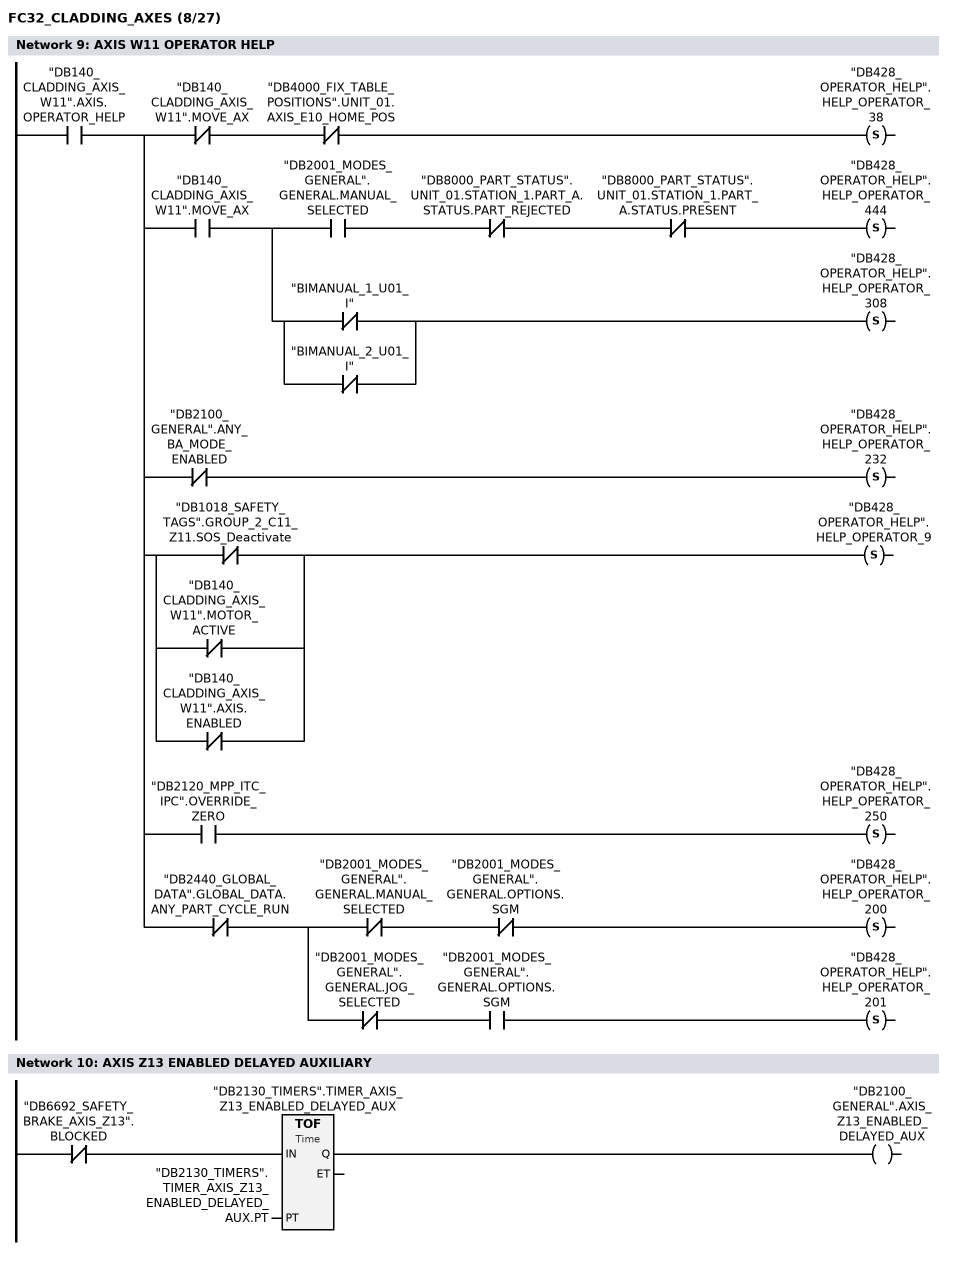
   RUNG wire#powerrail
      Contact( "DB140_CLADDING_AXIS_W11".AXIS.OPERATOR_HELP )
      wire#w1
      I_Contact( "DB140_CLADDING_AXIS_W11".MOVE_AX )
      I_Contact( "DB4000_FIX_TABLE_POSITIONS".UNIT_01.AXIS_E10_HOME_POS )
      S_Coil( "DB428_OPERATOR_HELP".HELP_OPERATOR_38 )
   END_RUNG
   RUNG wire#w1
      Contact( "DB140_CLADDING_AXIS_W11".MOVE_AX )
      wire#w2
      Contact( "DB2001_MODES_GENERAL".GENERAL.MANUAL_SELECTED )
      I_Contact( "DB8000_PART_STATUS".UNIT_01.STATION_1.PART_A.STATUS.PART_REJECTED )
      I_Contact( "DB8000_PART_STATUS".UNIT_01.STATION_1.PART_A.STATUS.PRESENT )
      S_Coil( "DB428_OPERATOR_HELP".HELP_OPERATOR_444 )
   END_RUNG
   RUNG wire#w2
      I_Contact( "BIMANUAL_1_U01_I" )
      wire#w3
      S_Coil( "DB428_OPERATOR_HELP".HELP_OPERATOR_308 )
   END_RUNG
   RUNG wire#w2
      I_Contact( "BIMANUAL_2_U01_I" )
   END_RUNG wire#w3
   RUNG wire#w1
      I_Contact( "DB2100_GENERAL".ANY_BA_MODE_ENABLED )
      S_Coil( "DB428_OPERATOR_HELP".HELP_OPERATOR_232 )
   END_RUNG
   RUNG wire#w1
      I_Contact( "DB1018_SAFETY_TAGS".GROUP_2_C11_Z11.SOS_Deactivate )
      wire#w4
      S_Coil( "DB428_OPERATOR_HELP".HELP_OPERATOR_9 )
   END_RUNG
   RUNG wire#w1
      I_Contact( "DB140_CLADDING_AXIS_W11".MOTOR_ACTIVE )
   END_RUNG wire#w4
   RUNG wire#w1
      I_Contact( "DB140_CLADDING_AXIS_W11".AXIS.ENABLED )
   END_RUNG wire#w4
   RUNG wire#w1
      Contact( "DB2120_MPP_ITC_IPC".OVERRIDE_ZERO )
      S_Coil( "DB428_OPERATOR_HELP".HELP_OPERATOR_250 )
   END_RUNG
   RUNG wire#w1
      I_Contact( "DB2440_GLOBAL_DATA".GLOBAL_DATA.ANY_PART_CYCLE_RUN )
      wire#w5
      I_Contact( "DB2001_MODES_GENERAL".GENERAL.MANUAL_SELECTED )
      I_Contact( "DB2001_MODES_GENERAL".GENERAL.OPTIONS.SGM )
      S_Coil( "DB428_OPERATOR_HELP".HELP_OPERATOR_200 )
   END_RUNG
   RUNG wire#w5
      I_Contact( "DB2001_MODES_GENERAL".GENERAL.JOG_SELECTED )
      Contact( "DB2001_MODES_GENERAL".GENERAL.OPTIONS.SGM )
      S_Coil( "DB428_OPERATOR_HELP".HELP_OPERATOR_201 )
   END_RUNG
   // the same network as SCL:
   IF "DB140_CLADDING_AXIS_W11".AXIS.OPERATOR_HELP AND NOT "DB140_CLADDING_AXIS_W11".MOVE_AX AND NOT "DB4000_FIX_TABLE_POSITIONS".UNIT_01.AXIS_E10_HOME_POS THEN
       "DB428_OPERATOR_HELP".HELP_OPERATOR_38 := TRUE;
   END_IF;
   #_w1 := "DB140_CLADDING_AXIS_W11".AXIS.OPERATOR_HELP AND "DB140_CLADDING_AXIS_W11".MOVE_AX;
   IF #_w1 AND "DB2001_MODES_GENERAL".GENERAL.MANUAL_SELECTED AND NOT "DB8000_PART_STATUS".UNIT_01.STATION_1.PART_A.STATUS.PART_REJECTED AND NOT "DB8000_PART_STATUS".UNIT_01.STATION_1.PART_A.STATUS.PRESENT THEN
       "DB428_OPERATOR_HELP".HELP_OPERATOR_444 := TRUE;
   END_IF;
   IF #_w1 AND (NOT "BIMANUAL_1_U01_I" OR NOT "BIMANUAL_2_U01_I") THEN
       "DB428_OPERATOR_HELP".HELP_OPERATOR_308 := TRUE;
   END_IF;
   IF "DB140_CLADDING_AXIS_W11".AXIS.OPERATOR_HELP AND NOT "DB2100_GENERAL".ANY_BA_MODE_ENABLED THEN
       "DB428_OPERATOR_HELP".HELP_OPERATOR_232 := TRUE;
   END_IF;
   IF "DB140_CLADDING_AXIS_W11".AXIS.OPERATOR_HELP AND (NOT "DB1018_SAFETY_TAGS".GROUP_2_C11_Z11.SOS_Deactivate OR NOT "DB140_CLADDING_AXIS_W11".MOTOR_ACTIVE OR NOT "DB140_CLADDING_AXIS_W11".AXIS.ENABLED) THEN
       "DB428_OPERATOR_HELP".HELP_OPERATOR_9 := TRUE;
   END_IF;
   IF "DB140_CLADDING_AXIS_W11".AXIS.OPERATOR_HELP AND "DB2120_MPP_ITC_IPC".OVERRIDE_ZERO THEN
       "DB428_OPERATOR_HELP".HELP_OPERATOR_250 := TRUE;
   END_IF;
   #_w2 := "DB140_CLADDING_AXIS_W11".AXIS.OPERATOR_HELP AND NOT "DB2440_GLOBAL_DATA".GLOBAL_DATA.ANY_PART_CYCLE_RUN;
   IF #_w2 AND NOT "DB2001_MODES_GENERAL".GENERAL.MANUAL_SELECTED AND NOT "DB2001_MODES_GENERAL".GENERAL.OPTIONS.SGM THEN
       "DB428_OPERATOR_HELP".HELP_OPERATOR_200 := TRUE;
   END_IF;
   IF #_w2 AND NOT "DB2001_MODES_GENERAL".GENERAL.JOG_SELECTED AND "DB2001_MODES_GENERAL".GENERAL.OPTIONS.SGM THEN
       "DB428_OPERATOR_HELP".HELP_OPERATOR_201 := TRUE;
   END_IF;
END_REGION

REGION Network 10: AXIS Z13 ENABLED DELAYED AUXILIARY
   RUNG wire#powerrail
      I_Contact( "DB6692_SAFETY_BRAKE_AXIS_Z13".BLOCKED )
      { S7_Templates := "time_type := Time" } "DB2130_TIMERS".TIMER_AXIS_Z13_ENABLED_DELAYED_AUX.TOF(pt := "DB2130_TIMERS".TIMER_AXIS_Z13_ENABLED_DELAYED_AUX.PT, et =>)
      Coil( "DB2100_GENERAL".AXIS_Z13_ENABLED_DELAYED_AUX )
   END_RUNG
   // the same network as SCL:
   "DB2130_TIMERS".TIMER_AXIS_Z13_ENABLED_DELAYED_AUX.TOF(IN := NOT "DB6692_SAFETY_BRAKE_AXIS_Z13".BLOCKED,
                           PT := "DB2130_TIMERS".TIMER_AXIS_Z13_ENABLED_DELAYED_AUX.PT);
   "DB2100_GENERAL".AXIS_Z13_ENABLED_DELAYED_AUX := "DB2130_TIMERS".TIMER_AXIS_Z13_ENABLED_DELAYED_AUX.Q;
END_REGION

REGION Network 11: AXIS Z13 MOVE AXIS AND FEED HOLD CONDITIONS
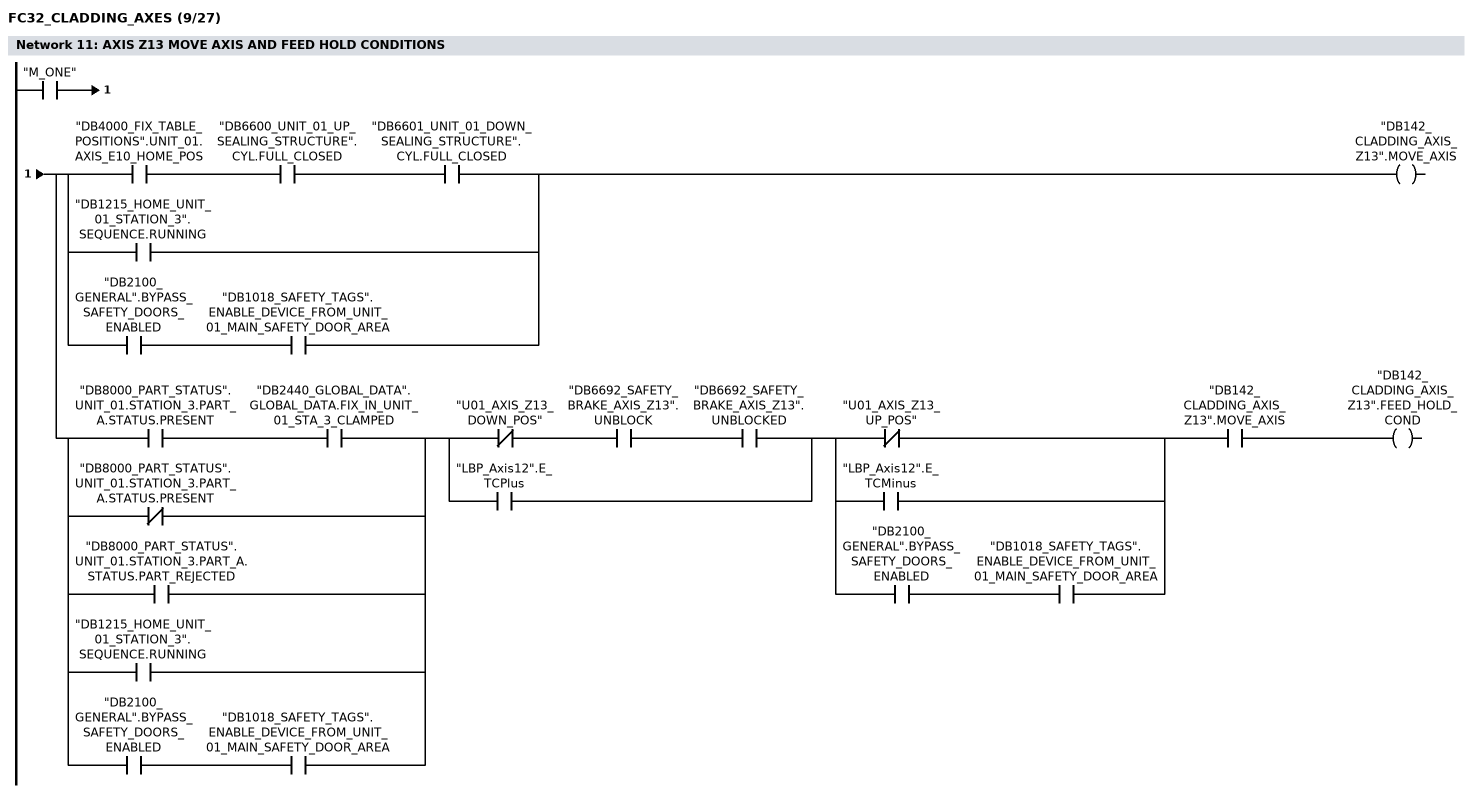
   RUNG wire#powerrail
      Contact( "M_ONE" )
      wire#w1
      Contact( "DB4000_FIX_TABLE_POSITIONS".UNIT_01.AXIS_E10_HOME_POS )
      Contact( "DB6600_UNIT_01_UP_SEALING_STRUCTURE".CYL.FULL_CLOSED )
      Contact( "DB6601_UNIT_01_DOWN_SEALING_STRUCTURE".CYL.FULL_CLOSED )
      wire#w2
      Coil( "DB142_CLADDING_AXIS_Z13".MOVE_AXIS )
   END_RUNG
   RUNG wire#w1
      Contact( "DB1215_HOME_UNIT_01_STATION_3".SEQUENCE.RUNNING )
   END_RUNG wire#w2
   RUNG wire#w1
      Contact( "DB2100_GENERAL".BYPASS_SAFETY_DOORS_ENABLED )
      Contact( "DB1018_SAFETY_TAGS".ENABLE_DEVICE_FROM_UNIT_01_MAIN_SAFETY_DOOR_AREA )
   END_RUNG wire#w2
   RUNG wire#w1
      Contact( "DB8000_PART_STATUS".UNIT_01.STATION_3.PART_A.STATUS.PRESENT )
      Contact( "DB2440_GLOBAL_DATA".GLOBAL_DATA.FIX_IN_UNIT_01_STA_3_CLAMPED )
      wire#w3
      I_Contact( "U01_AXIS_Z13_DOWN_POS" )
      Contact( "DB6692_SAFETY_BRAKE_AXIS_Z13".UNBLOCK )
      Contact( "DB6692_SAFETY_BRAKE_AXIS_Z13".UNBLOCKED )
      wire#w4
      I_Contact( "U01_AXIS_Z13_UP_POS" )
      wire#w5
      Contact( "DB142_CLADDING_AXIS_Z13".MOVE_AXIS )
      Coil( "DB142_CLADDING_AXIS_Z13".FEED_HOLD_COND )
   END_RUNG
   RUNG wire#w1
      I_Contact( "DB8000_PART_STATUS".UNIT_01.STATION_3.PART_A.STATUS.PRESENT )
   END_RUNG wire#w3
   RUNG wire#w1
      Contact( "DB8000_PART_STATUS".UNIT_01.STATION_3.PART_A.STATUS.PART_REJECTED )
   END_RUNG wire#w3
   RUNG wire#w1
      Contact( "DB1215_HOME_UNIT_01_STATION_3".SEQUENCE.RUNNING )
   END_RUNG wire#w3
   RUNG wire#w1
      Contact( "DB2100_GENERAL".BYPASS_SAFETY_DOORS_ENABLED )
      Contact( "DB1018_SAFETY_TAGS".ENABLE_DEVICE_FROM_UNIT_01_MAIN_SAFETY_DOOR_AREA )
   END_RUNG wire#w3
   RUNG wire#w3
      Contact( "LBP_Axis12".E_TCPlus )
   END_RUNG wire#w4
   RUNG wire#w4
      Contact( "LBP_Axis12".E_TCMinus )
   END_RUNG wire#w5
   RUNG wire#w4
      Contact( "DB2100_GENERAL".BYPASS_SAFETY_DOORS_ENABLED )
      Contact( "DB1018_SAFETY_TAGS".ENABLE_DEVICE_FROM_UNIT_01_MAIN_SAFETY_DOOR_AREA )
   END_RUNG wire#w5
   // the same network as SCL:
   "DB142_CLADDING_AXIS_Z13".MOVE_AXIS := "M_ONE" AND (("DB4000_FIX_TABLE_POSITIONS".UNIT_01.AXIS_E10_HOME_POS AND "DB6600_UNIT_01_UP_SEALING_STRUCTURE".CYL.FULL_CLOSED AND "DB6601_UNIT_01_DOWN_SEALING_STRUCTURE".CYL.FULL_CLOSED) OR "DB1215_HOME_UNIT_01_STATION_3".SEQUENCE.RUNNING OR ("DB2100_GENERAL".BYPASS_SAFETY_DOORS_ENABLED AND "DB1018_SAFETY_TAGS".ENABLE_DEVICE_FROM_UNIT_01_MAIN_SAFETY_DOOR_AREA));
   "DB142_CLADDING_AXIS_Z13".FEED_HOLD_COND := "M_ONE" AND (("DB8000_PART_STATUS".UNIT_01.STATION_3.PART_A.STATUS.PRESENT AND "DB2440_GLOBAL_DATA".GLOBAL_DATA.FIX_IN_UNIT_01_STA_3_CLAMPED) OR NOT "DB8000_PART_STATUS".UNIT_01.STATION_3.PART_A.STATUS.PRESENT OR "DB8000_PART_STATUS".UNIT_01.STATION_3.PART_A.STATUS.PART_REJECTED OR "DB1215_HOME_UNIT_01_STATION_3".SEQUENCE.RUNNING OR ("DB2100_GENERAL".BYPASS_SAFETY_DOORS_ENABLED AND "DB1018_SAFETY_TAGS".ENABLE_DEVICE_FROM_UNIT_01_MAIN_SAFETY_DOOR_AREA)) AND ((NOT "U01_AXIS_Z13_DOWN_POS" AND "DB6692_SAFETY_BRAKE_AXIS_Z13".UNBLOCK AND "DB6692_SAFETY_BRAKE_AXIS_Z13".UNBLOCKED) OR "LBP_Axis12".E_TCPlus) AND (NOT "U01_AXIS_Z13_UP_POS" OR "LBP_Axis12".E_TCMinus OR ("DB2100_GENERAL".BYPASS_SAFETY_DOORS_ENABLED AND "DB1018_SAFETY_TAGS".ENABLE_DEVICE_FROM_UNIT_01_MAIN_SAFETY_DOOR_AREA)) AND "DB142_CLADDING_AXIS_Z13".MOVE_AXIS;
END_REGION

REGION Network 12: CALL FB32 AXIS Z13
   // 2#0000_0001 OPTIONS 0 BIT 0 MEASURING SYSTEM 2 OPTION
   // 2#0000_0010 OPTIONS 0 BIT 1 ENABLE FC18 OPTION
   // 2#0000_0100 OPTIONS 0 BIT 2 FC18 EXTERNAL POSITION OPTION
   // 2#0000_1000 OPTIONS 0 BIT 3 AXIS B ENABLE FAULTS OPTION
   // 2#0001_0000 OPTIONS 0 BIT 4 SPARE OPTION
   // 2#0010_0000 OPTIONS 0 BIT 5 SPARE OPTION
   // 2#0100_0000 OPTIONS 0 BIT 6 SPARE OPTION
   // 2#1000_0000 OPTIONS 0 BIT 7 SPARE OPTION
   // 
   // 2#0000_0001 OPTIONS 1 BIT 0 AXIS ROLLER OPTION
   // 2#0000_0010 OPTIONS 1 BIT 1 MASTER AXIS OPTION
   // 2#0000_0100 OPTIONS 1 BIT 2 SLAVE AXIS OPTION
   // 2#0000_1000 OPTIONS 1 BIT 3 MASTER-SLAVE AXES INDEPENDENT MOVEMENT WITH HT10 OPTION
   // 2#0001_0000 OPTIONS 1 BIT 4 GANTRY MODE MASTER AXIS OPTION
   // 2#0010_0000 OPTIONS 1 BIT 5 SPARE OPTION
   // 2#0100_0000 OPTIONS 1 BIT 6 SPARE OPTION
   // 2#1000_0000 OPTIONS 1 BIT 7 SPARE OPTION
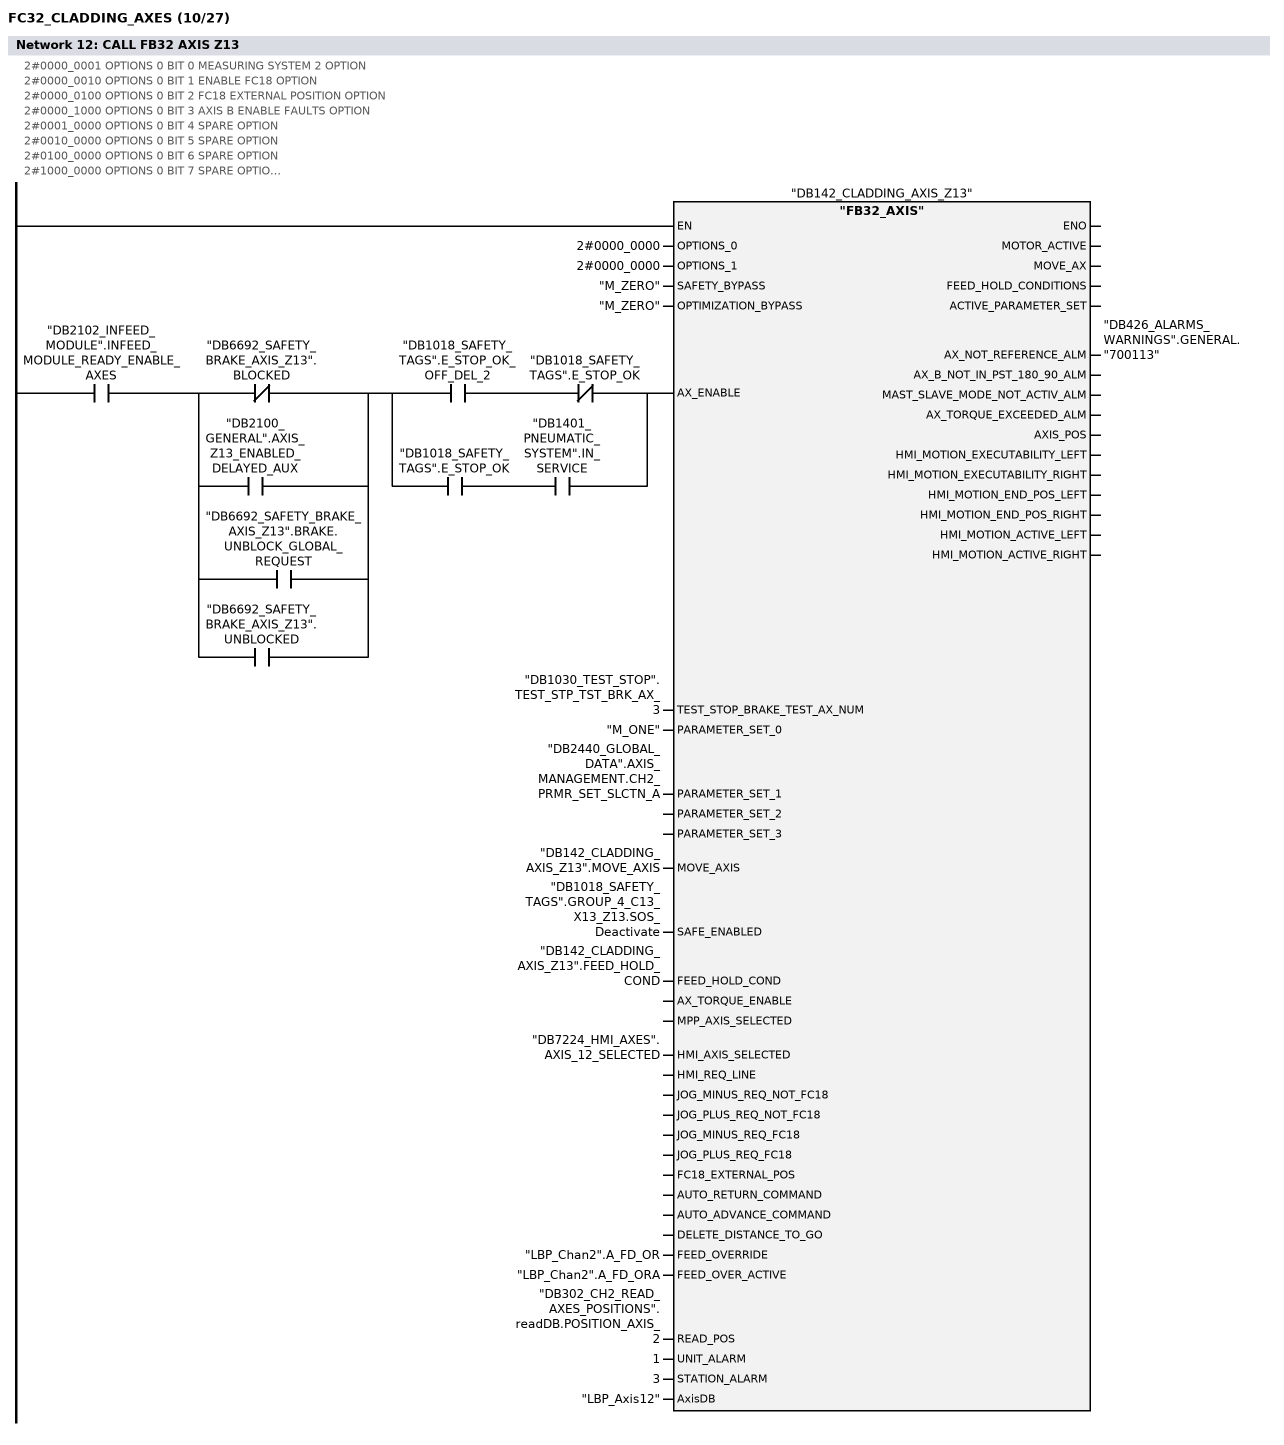
   RUNG wire#powerrail
      "DB142_CLADDING_AXIS_Z13"(AX_ENABLE := wire#w3, OPTIONS_0 := 2#0000_0000, OPTIONS_1 := 2#0000_0000, SAFETY_BYPASS := "M_ZERO", OPTIMIZATION_BYPASS := "M_ZERO", TEST_STOP_BRAKE_TEST_AX_NUM := "DB1030_TEST_STOP".TEST_STP_TST_BRK_AX_3, PARAMETER_SET_0 := "M_ONE", PARAMETER_SET_1 := "DB2440_GLOBAL_DATA".AXIS_MANAGEMENT.CH2_PRMR_SET_SLCTN_A, PARAMETER_SET_2 :=, PARAMETER_SET_3 :=, MOVE_AXIS := "DB142_CLADDING_AXIS_Z13".MOVE_AXIS, SAFE_ENABLED := "DB1018_SAFETY_TAGS".GROUP_4_C13_X13_Z13.SOS_Deactivate, FEED_HOLD_COND := "DB142_CLADDING_AXIS_Z13".FEED_HOLD_COND, AX_TORQUE_ENABLE :=, MPP_AXIS_SELECTED :=, HMI_AXIS_SELECTED := "DB7224_HMI_AXES".AXIS_12_SELECTED, HMI_REQ_LINE :=, JOG_MINUS_REQ_NOT_FC18 :=, JOG_PLUS_REQ_NOT_FC18 :=, JOG_MINUS_REQ_FC18 :=, JOG_PLUS_REQ_FC18 :=, FC18_EXTERNAL_POS :=, AUTO_RETURN_COMMAND :=, AUTO_ADVANCE_COMMAND :=, DELETE_DISTANCE_TO_GO :=, FEED_OVERRIDE := "LBP_Chan2".A_FD_OR, FEED_OVER_ACTIVE := "LBP_Chan2".A_FD_ORA, READ_POS := "DB302_CH2_READ_AXES_POSITIONS".readDB.POSITION_AXIS_2, UNIT_ALARM := 1, STATION_ALARM := 3, AxisDB := "LBP_Axis12", MOTOR_ACTIVE =>, MOVE_AX =>, FEED_HOLD_CONDITIONS =>, ACTIVE_PARAMETER_SET =>, AX_NOT_REFERENCE_ALM => "DB426_ALARMS_WARNINGS".GENERAL."700113", AX_B_NOT_IN_PST_180_90_ALM =>, MAST_SLAVE_MODE_NOT_ACTIV_ALM =>, AX_TORQUE_EXCEEDED_ALM =>, AXIS_POS =>, HMI_MOTION_EXECUTABILITY_LEFT =>, HMI_MOTION_EXECUTABILITY_RIGHT =>, HMI_MOTION_END_POS_LEFT =>, HMI_MOTION_END_POS_RIGHT =>, HMI_MOTION_ACTIVE_LEFT =>, HMI_MOTION_ACTIVE_RIGHT =>)
   END_RUNG
   RUNG wire#powerrail
      Contact( "DB2102_INFEED_MODULE".INFEED_MODULE_READY_ENABLE_AXES )
      wire#w1
      I_Contact( "DB6692_SAFETY_BRAKE_AXIS_Z13".BLOCKED )
      wire#w2
      Contact( "DB1018_SAFETY_TAGS".E_STOP_OK_OFF_DEL_2 )
      I_Contact( "DB1018_SAFETY_TAGS".E_STOP_OK )
   END_RUNG wire#w3
   RUNG wire#w1
      Contact( "DB2100_GENERAL".AXIS_Z13_ENABLED_DELAYED_AUX )
   END_RUNG wire#w2
   RUNG wire#w1
      Contact( "DB6692_SAFETY_BRAKE_AXIS_Z13".BRAKE.UNBLOCK_GLOBAL_REQUEST )
   END_RUNG wire#w2
   RUNG wire#w1
      Contact( "DB6692_SAFETY_BRAKE_AXIS_Z13".UNBLOCKED )
   END_RUNG wire#w2
   RUNG wire#w2
      Contact( "DB1018_SAFETY_TAGS".E_STOP_OK )
      Contact( "DB1401_PNEUMATIC_SYSTEM".IN_SERVICE )
   END_RUNG wire#w3
   // the same network as SCL:
   "DB142_CLADDING_AXIS_Z13"(OPTIONS_0 := 2#0000_0000,   // "FB32_AXIS"
                           OPTIONS_1 := 2#0000_0000,
                           SAFETY_BYPASS := "M_ZERO",
                           OPTIMIZATION_BYPASS := "M_ZERO",
                           AX_ENABLE := "DB2102_INFEED_MODULE".INFEED_MODULE_READY_ENABLE_AXES AND (NOT "DB6692_SAFETY_BRAKE_AXIS_Z13".BLOCKED OR "DB2100_GENERAL".AXIS_Z13_ENABLED_DELAYED_AUX OR "DB6692_SAFETY_BRAKE_AXIS_Z13".BRAKE.UNBLOCK_GLOBAL_REQUEST OR "DB6692_SAFETY_BRAKE_AXIS_Z13".UNBLOCKED) AND (("DB1018_SAFETY_TAGS".E_STOP_OK_OFF_DEL_2 AND NOT "DB1018_SAFETY_TAGS".E_STOP_OK) OR ("DB1018_SAFETY_TAGS".E_STOP_OK AND "DB1401_PNEUMATIC_SYSTEM".IN_SERVICE)),
                           TEST_STOP_BRAKE_TEST_AX_NUM := "DB1030_TEST_STOP".TEST_STP_TST_BRK_AX_3,
                           PARAMETER_SET_0 := "M_ONE",
                           PARAMETER_SET_1 := "DB2440_GLOBAL_DATA".AXIS_MANAGEMENT.CH2_PRMR_SET_SLCTN_A,
                           MOVE_AXIS := "DB142_CLADDING_AXIS_Z13".MOVE_AXIS,
                           SAFE_ENABLED := "DB1018_SAFETY_TAGS".GROUP_4_C13_X13_Z13.SOS_Deactivate,
                           FEED_HOLD_COND := "DB142_CLADDING_AXIS_Z13".FEED_HOLD_COND,
                           HMI_AXIS_SELECTED := "DB7224_HMI_AXES".AXIS_12_SELECTED,
                           FEED_OVERRIDE := "LBP_Chan2".A_FD_OR,
                           FEED_OVER_ACTIVE := "LBP_Chan2".A_FD_ORA,
                           READ_POS := "DB302_CH2_READ_AXES_POSITIONS".readDB.POSITION_AXIS_2,
                           UNIT_ALARM := 1,
                           STATION_ALARM := 3,
                           AxisDB := "LBP_Axis12",
                           AX_NOT_REFERENCE_ALM => "DB426_ALARMS_WARNINGS".GENERAL."700113");
END_REGION

REGION Network 13: AXIS Z13 OPERATOR HELP
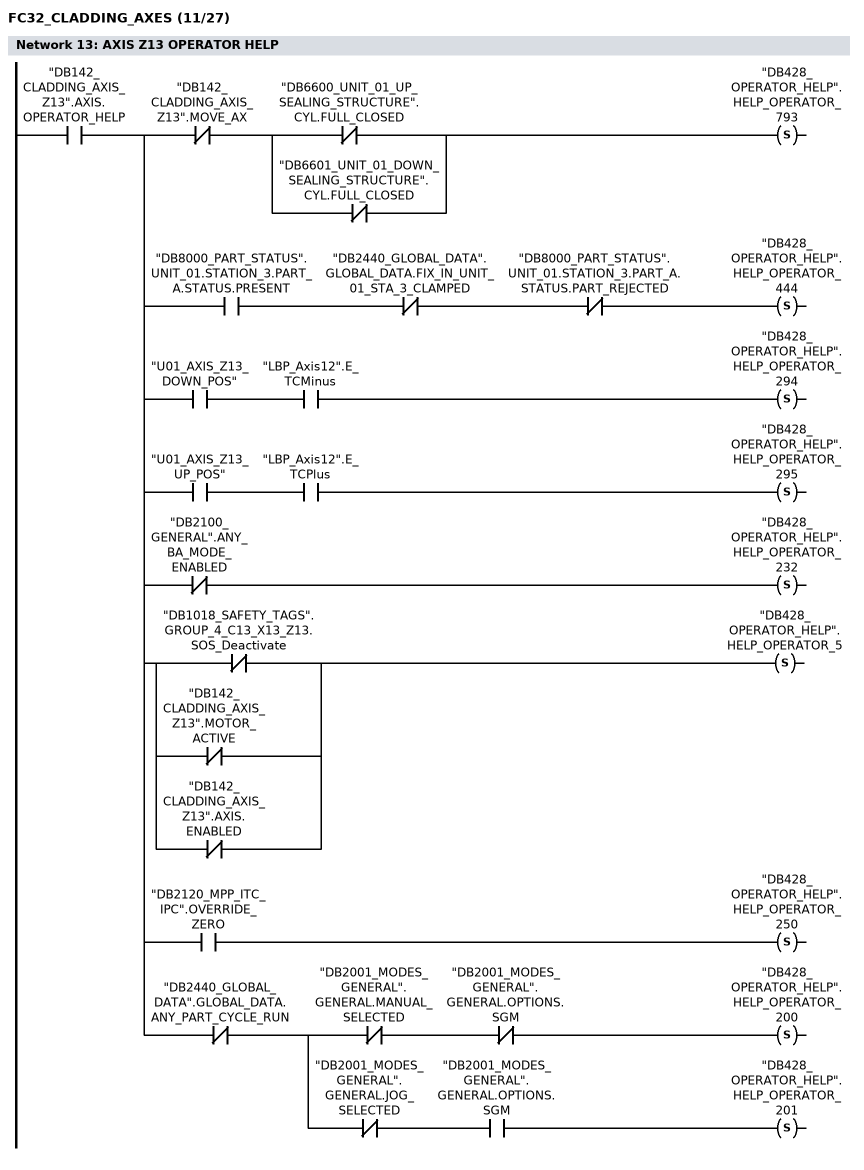
   RUNG wire#powerrail
      Contact( "DB142_CLADDING_AXIS_Z13".AXIS.OPERATOR_HELP )
      wire#w1
      I_Contact( "DB142_CLADDING_AXIS_Z13".MOVE_AX )
      wire#w2
      I_Contact( "DB6600_UNIT_01_UP_SEALING_STRUCTURE".CYL.FULL_CLOSED )
      wire#w3
      S_Coil( "DB428_OPERATOR_HELP".HELP_OPERATOR_793 )
   END_RUNG
   RUNG wire#w2
      I_Contact( "DB6601_UNIT_01_DOWN_SEALING_STRUCTURE".CYL.FULL_CLOSED )
   END_RUNG wire#w3
   RUNG wire#w1
      Contact( "DB8000_PART_STATUS".UNIT_01.STATION_3.PART_A.STATUS.PRESENT )
      I_Contact( "DB2440_GLOBAL_DATA".GLOBAL_DATA.FIX_IN_UNIT_01_STA_3_CLAMPED )
      I_Contact( "DB8000_PART_STATUS".UNIT_01.STATION_3.PART_A.STATUS.PART_REJECTED )
      S_Coil( "DB428_OPERATOR_HELP".HELP_OPERATOR_444 )
   END_RUNG
   RUNG wire#w1
      Contact( "U01_AXIS_Z13_DOWN_POS" )
      Contact( "LBP_Axis12".E_TCMinus )
      S_Coil( "DB428_OPERATOR_HELP".HELP_OPERATOR_294 )
   END_RUNG
   RUNG wire#w1
      Contact( "U01_AXIS_Z13_UP_POS" )
      Contact( "LBP_Axis12".E_TCPlus )
      S_Coil( "DB428_OPERATOR_HELP".HELP_OPERATOR_295 )
   END_RUNG
   RUNG wire#w1
      I_Contact( "DB2100_GENERAL".ANY_BA_MODE_ENABLED )
      S_Coil( "DB428_OPERATOR_HELP".HELP_OPERATOR_232 )
   END_RUNG
   RUNG wire#w1
      I_Contact( "DB1018_SAFETY_TAGS".GROUP_4_C13_X13_Z13.SOS_Deactivate )
      wire#w4
      S_Coil( "DB428_OPERATOR_HELP".HELP_OPERATOR_5 )
   END_RUNG
   RUNG wire#w1
      I_Contact( "DB142_CLADDING_AXIS_Z13".MOTOR_ACTIVE )
   END_RUNG wire#w4
   RUNG wire#w1
      I_Contact( "DB142_CLADDING_AXIS_Z13".AXIS.ENABLED )
   END_RUNG wire#w4
   RUNG wire#w1
      Contact( "DB2120_MPP_ITC_IPC".OVERRIDE_ZERO )
      S_Coil( "DB428_OPERATOR_HELP".HELP_OPERATOR_250 )
   END_RUNG
   RUNG wire#w1
      I_Contact( "DB2440_GLOBAL_DATA".GLOBAL_DATA.ANY_PART_CYCLE_RUN )
      wire#w5
      I_Contact( "DB2001_MODES_GENERAL".GENERAL.MANUAL_SELECTED )
      I_Contact( "DB2001_MODES_GENERAL".GENERAL.OPTIONS.SGM )
      S_Coil( "DB428_OPERATOR_HELP".HELP_OPERATOR_200 )
   END_RUNG
   RUNG wire#w5
      I_Contact( "DB2001_MODES_GENERAL".GENERAL.JOG_SELECTED )
      Contact( "DB2001_MODES_GENERAL".GENERAL.OPTIONS.SGM )
      S_Coil( "DB428_OPERATOR_HELP".HELP_OPERATOR_201 )
   END_RUNG
   // the same network as SCL:
   IF "DB142_CLADDING_AXIS_Z13".AXIS.OPERATOR_HELP AND NOT "DB142_CLADDING_AXIS_Z13".MOVE_AX AND (NOT "DB6600_UNIT_01_UP_SEALING_STRUCTURE".CYL.FULL_CLOSED OR NOT "DB6601_UNIT_01_DOWN_SEALING_STRUCTURE".CYL.FULL_CLOSED) THEN
       "DB428_OPERATOR_HELP".HELP_OPERATOR_793 := TRUE;
   END_IF;
   IF "DB142_CLADDING_AXIS_Z13".AXIS.OPERATOR_HELP AND "DB8000_PART_STATUS".UNIT_01.STATION_3.PART_A.STATUS.PRESENT AND NOT "DB2440_GLOBAL_DATA".GLOBAL_DATA.FIX_IN_UNIT_01_STA_3_CLAMPED AND NOT "DB8000_PART_STATUS".UNIT_01.STATION_3.PART_A.STATUS.PART_REJECTED THEN
       "DB428_OPERATOR_HELP".HELP_OPERATOR_444 := TRUE;
   END_IF;
   IF "DB142_CLADDING_AXIS_Z13".AXIS.OPERATOR_HELP AND "U01_AXIS_Z13_DOWN_POS" AND "LBP_Axis12".E_TCMinus THEN
       "DB428_OPERATOR_HELP".HELP_OPERATOR_294 := TRUE;
   END_IF;
   IF "DB142_CLADDING_AXIS_Z13".AXIS.OPERATOR_HELP AND "U01_AXIS_Z13_UP_POS" AND "LBP_Axis12".E_TCPlus THEN
       "DB428_OPERATOR_HELP".HELP_OPERATOR_295 := TRUE;
   END_IF;
   IF "DB142_CLADDING_AXIS_Z13".AXIS.OPERATOR_HELP AND NOT "DB2100_GENERAL".ANY_BA_MODE_ENABLED THEN
       "DB428_OPERATOR_HELP".HELP_OPERATOR_232 := TRUE;
   END_IF;
   IF "DB142_CLADDING_AXIS_Z13".AXIS.OPERATOR_HELP AND (NOT "DB1018_SAFETY_TAGS".GROUP_4_C13_X13_Z13.SOS_Deactivate OR NOT "DB142_CLADDING_AXIS_Z13".MOTOR_ACTIVE OR NOT "DB142_CLADDING_AXIS_Z13".AXIS.ENABLED) THEN
       "DB428_OPERATOR_HELP".HELP_OPERATOR_5 := TRUE;
   END_IF;
   IF "DB142_CLADDING_AXIS_Z13".AXIS.OPERATOR_HELP AND "DB2120_MPP_ITC_IPC".OVERRIDE_ZERO THEN
       "DB428_OPERATOR_HELP".HELP_OPERATOR_250 := TRUE;
   END_IF;
   #_w1 := "DB142_CLADDING_AXIS_Z13".AXIS.OPERATOR_HELP AND NOT "DB2440_GLOBAL_DATA".GLOBAL_DATA.ANY_PART_CYCLE_RUN;
   IF #_w1 AND NOT "DB2001_MODES_GENERAL".GENERAL.MANUAL_SELECTED AND NOT "DB2001_MODES_GENERAL".GENERAL.OPTIONS.SGM THEN
       "DB428_OPERATOR_HELP".HELP_OPERATOR_200 := TRUE;
   END_IF;
   IF #_w1 AND NOT "DB2001_MODES_GENERAL".GENERAL.JOG_SELECTED AND "DB2001_MODES_GENERAL".GENERAL.OPTIONS.SGM THEN
       "DB428_OPERATOR_HELP".HELP_OPERATOR_201 := TRUE;
   END_IF;
END_REGION

REGION Network 14: AXIS E20 MOVE AXIS AND FEED HOLD CONDITIONS
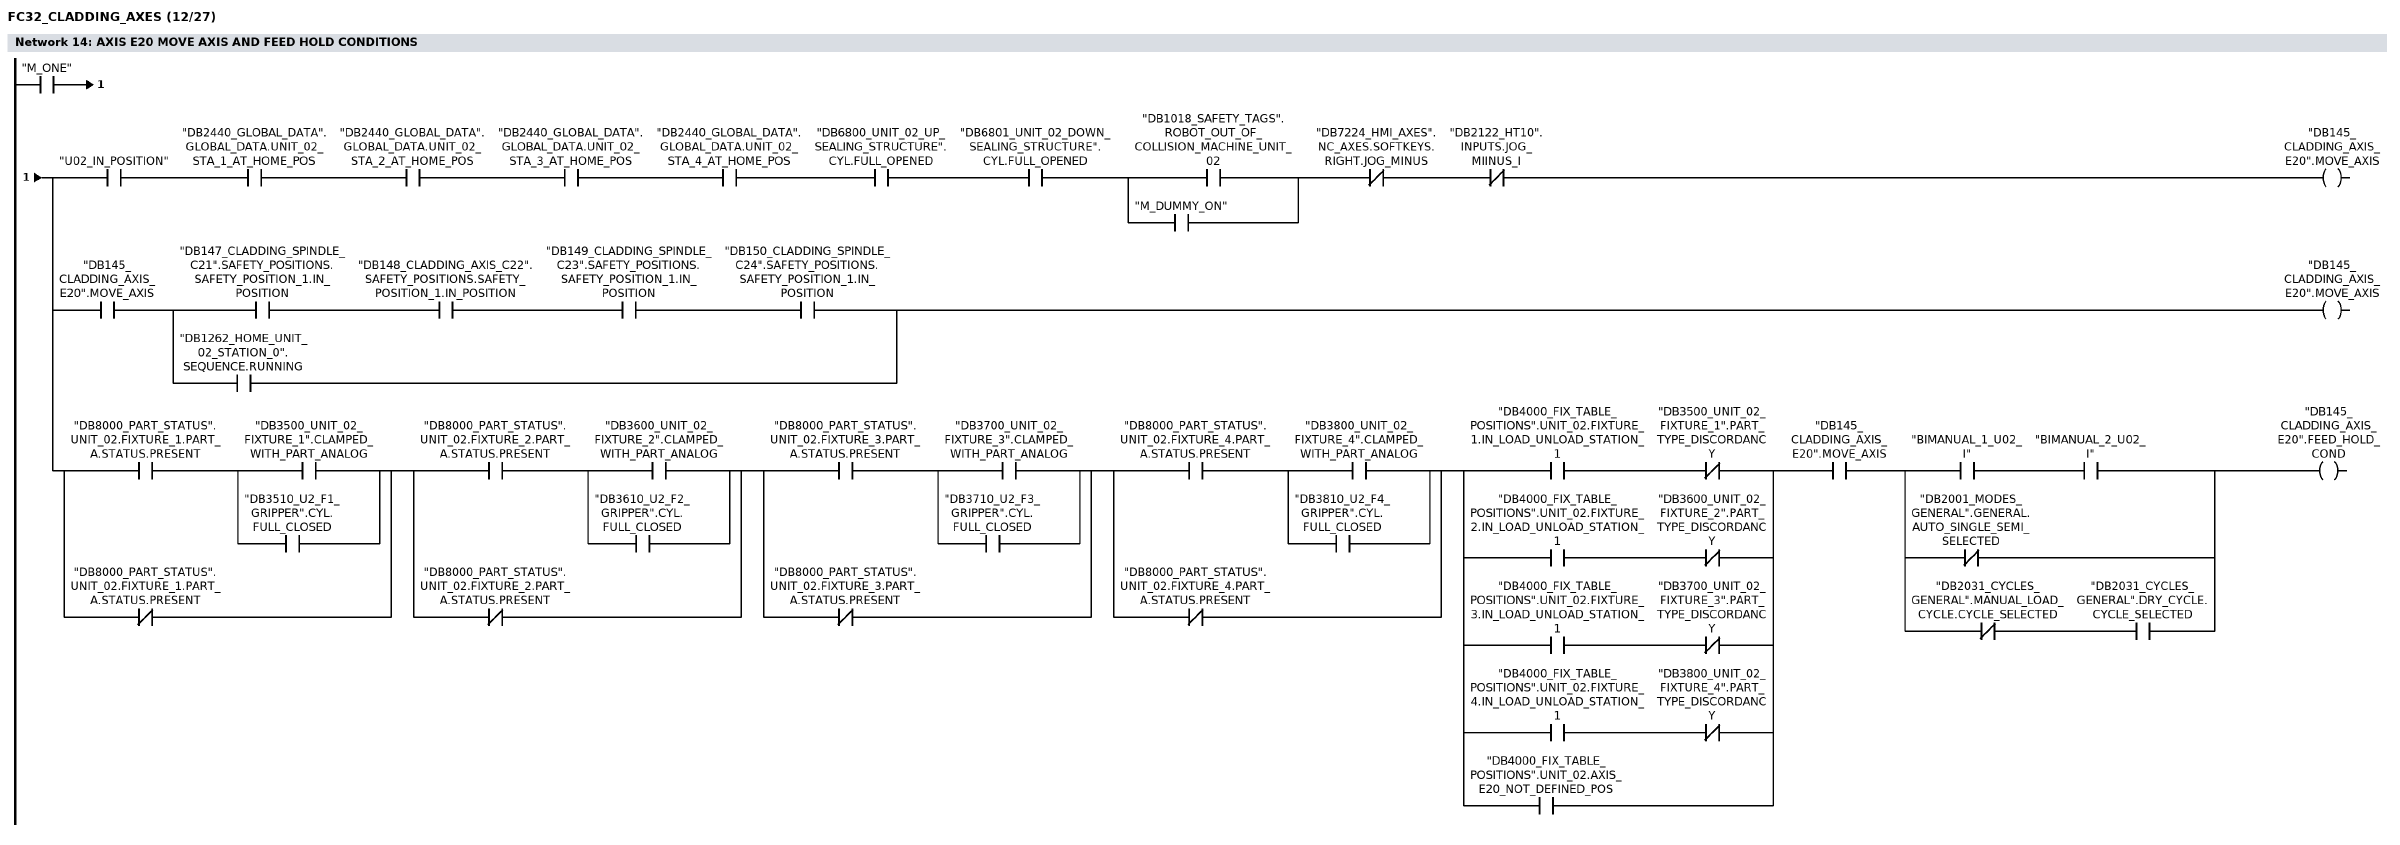
   RUNG wire#powerrail
      Contact( "M_ONE" )
      wire#w1
      Contact( "U02_IN_POSITION" )
      Contact( "DB2440_GLOBAL_DATA".GLOBAL_DATA.UNIT_02_STA_1_AT_HOME_POS )
      Contact( "DB2440_GLOBAL_DATA".GLOBAL_DATA.UNIT_02_STA_2_AT_HOME_POS )
      Contact( "DB2440_GLOBAL_DATA".GLOBAL_DATA.UNIT_02_STA_3_AT_HOME_POS )
      Contact( "DB2440_GLOBAL_DATA".GLOBAL_DATA.UNIT_02_STA_4_AT_HOME_POS )
      Contact( "DB6800_UNIT_02_UP_SEALING_STRUCTURE".CYL.FULL_OPENED )
      Contact( "DB6801_UNIT_02_DOWN_SEALING_STRUCTURE".CYL.FULL_OPENED )
      wire#w2
      Contact( "DB1018_SAFETY_TAGS".ROBOT_OUT_OF_COLLISION_MACHINE_UNIT_02 )
      wire#w3
      I_Contact( "DB7224_HMI_AXES".NC_AXES.SOFTKEYS.RIGHT.JOG_MINUS )
      I_Contact( "DB2122_HT10".INPUTS.JOG_MIINUS_I )
      Coil( "DB145_CLADDING_AXIS_E20".MOVE_AXIS )
   END_RUNG
   RUNG wire#w2
      Contact( "M_DUMMY_ON" )
   END_RUNG wire#w3
   RUNG wire#w1
      Contact( "DB145_CLADDING_AXIS_E20".MOVE_AXIS )
      wire#w4
      Contact( "DB147_CLADDING_SPINDLE_C21".SAFETY_POSITIONS.SAFETY_POSITION_1.IN_POSITION )
      Contact( "DB148_CLADDING_AXIS_C22".SAFETY_POSITIONS.SAFETY_POSITION_1.IN_POSITION )
      Contact( "DB149_CLADDING_SPINDLE_C23".SAFETY_POSITIONS.SAFETY_POSITION_1.IN_POSITION )
      Contact( "DB150_CLADDING_SPINDLE_C24".SAFETY_POSITIONS.SAFETY_POSITION_1.IN_POSITION )
      wire#w5
      Coil( "DB145_CLADDING_AXIS_E20".MOVE_AXIS )
   END_RUNG
   RUNG wire#w4
      Contact( "DB1262_HOME_UNIT_02_STATION_0".SEQUENCE.RUNNING )
   END_RUNG wire#w5
   RUNG wire#w1
      Contact( "DB8000_PART_STATUS".UNIT_02.FIXTURE_1.PART_A.STATUS.PRESENT )
      wire#w6
      Contact( "DB3500_UNIT_02_FIXTURE_1".CLAMPED_WITH_PART_ANALOG )
      wire#w7
      Contact( "DB8000_PART_STATUS".UNIT_02.FIXTURE_2.PART_A.STATUS.PRESENT )
      wire#w8
      Contact( "DB3600_UNIT_02_FIXTURE_2".CLAMPED_WITH_PART_ANALOG )
      wire#w9
      Contact( "DB8000_PART_STATUS".UNIT_02.FIXTURE_3.PART_A.STATUS.PRESENT )
      wire#w10
      Contact( "DB3700_UNIT_02_FIXTURE_3".CLAMPED_WITH_PART_ANALOG )
      wire#w11
      Contact( "DB8000_PART_STATUS".UNIT_02.FIXTURE_4.PART_A.STATUS.PRESENT )
      wire#w12
      Contact( "DB3800_UNIT_02_FIXTURE_4".CLAMPED_WITH_PART_ANALOG )
      wire#w13
      Contact( "DB4000_FIX_TABLE_POSITIONS".UNIT_02.FIXTURE_1.IN_LOAD_UNLOAD_STATION_1 )
      I_Contact( "DB3500_UNIT_02_FIXTURE_1".PART_TYPE_DISCORDANCY )
      wire#w14
      Contact( "DB145_CLADDING_AXIS_E20".MOVE_AXIS )
      wire#w15
      Contact( "BIMANUAL_1_U02_I" )
      Contact( "BIMANUAL_2_U02_I" )
      wire#w16
      Coil( "DB145_CLADDING_AXIS_E20".FEED_HOLD_COND )
   END_RUNG
   RUNG wire#w6
      Contact( "DB3510_U2_F1_GRIPPER".CYL.FULL_CLOSED )
   END_RUNG wire#w7
   RUNG wire#w1
      I_Contact( "DB8000_PART_STATUS".UNIT_02.FIXTURE_1.PART_A.STATUS.PRESENT )
   END_RUNG wire#w7
   RUNG wire#w8
      Contact( "DB3610_U2_F2_GRIPPER".CYL.FULL_CLOSED )
   END_RUNG wire#w9
   RUNG wire#w7
      I_Contact( "DB8000_PART_STATUS".UNIT_02.FIXTURE_2.PART_A.STATUS.PRESENT )
   END_RUNG wire#w9
   RUNG wire#w10
      Contact( "DB3710_U2_F3_GRIPPER".CYL.FULL_CLOSED )
   END_RUNG wire#w11
   RUNG wire#w9
      I_Contact( "DB8000_PART_STATUS".UNIT_02.FIXTURE_3.PART_A.STATUS.PRESENT )
   END_RUNG wire#w11
   RUNG wire#w12
      Contact( "DB3810_U2_F4_GRIPPER".CYL.FULL_CLOSED )
   END_RUNG wire#w13
   RUNG wire#w11
      I_Contact( "DB8000_PART_STATUS".UNIT_02.FIXTURE_4.PART_A.STATUS.PRESENT )
   END_RUNG wire#w13
   RUNG wire#w13
      Contact( "DB4000_FIX_TABLE_POSITIONS".UNIT_02.FIXTURE_2.IN_LOAD_UNLOAD_STATION_1 )
      I_Contact( "DB3600_UNIT_02_FIXTURE_2".PART_TYPE_DISCORDANCY )
   END_RUNG wire#w14
   RUNG wire#w13
      Contact( "DB4000_FIX_TABLE_POSITIONS".UNIT_02.FIXTURE_3.IN_LOAD_UNLOAD_STATION_1 )
      I_Contact( "DB3700_UNIT_02_FIXTURE_3".PART_TYPE_DISCORDANCY )
   END_RUNG wire#w14
   RUNG wire#w13
      Contact( "DB4000_FIX_TABLE_POSITIONS".UNIT_02.FIXTURE_4.IN_LOAD_UNLOAD_STATION_1 )
      I_Contact( "DB3800_UNIT_02_FIXTURE_4".PART_TYPE_DISCORDANCY )
   END_RUNG wire#w14
   RUNG wire#w13
      Contact( "DB4000_FIX_TABLE_POSITIONS".UNIT_02.AXIS_E20_NOT_DEFINED_POS )
   END_RUNG wire#w14
   RUNG wire#w15
      I_Contact( "DB2001_MODES_GENERAL".GENERAL.AUTO_SINGLE_SEMI_SELECTED )
   END_RUNG wire#w16
   RUNG wire#w15
      I_Contact( "DB2031_CYCLES_GENERAL".MANUAL_LOAD_CYCLE.CYCLE_SELECTED )
      Contact( "DB2031_CYCLES_GENERAL".DRY_CYCLE.CYCLE_SELECTED )
   END_RUNG wire#w16
   // the same network as SCL:
   "DB145_CLADDING_AXIS_E20".MOVE_AXIS := "M_ONE" AND "U02_IN_POSITION" AND "DB2440_GLOBAL_DATA".GLOBAL_DATA.UNIT_02_STA_1_AT_HOME_POS AND "DB2440_GLOBAL_DATA".GLOBAL_DATA.UNIT_02_STA_2_AT_HOME_POS AND "DB2440_GLOBAL_DATA".GLOBAL_DATA.UNIT_02_STA_3_AT_HOME_POS AND "DB2440_GLOBAL_DATA".GLOBAL_DATA.UNIT_02_STA_4_AT_HOME_POS AND "DB6800_UNIT_02_UP_SEALING_STRUCTURE".CYL.FULL_OPENED AND "DB6801_UNIT_02_DOWN_SEALING_STRUCTURE".CYL.FULL_OPENED AND ("DB1018_SAFETY_TAGS".ROBOT_OUT_OF_COLLISION_MACHINE_UNIT_02 OR "M_DUMMY_ON") AND NOT "DB7224_HMI_AXES".NC_AXES.SOFTKEYS.RIGHT.JOG_MINUS AND NOT "DB2122_HT10".INPUTS.JOG_MIINUS_I;
   "DB145_CLADDING_AXIS_E20".MOVE_AXIS := "M_ONE" AND "DB145_CLADDING_AXIS_E20".MOVE_AXIS AND (("DB147_CLADDING_SPINDLE_C21".SAFETY_POSITIONS.SAFETY_POSITION_1.IN_POSITION AND "DB148_CLADDING_AXIS_C22".SAFETY_POSITIONS.SAFETY_POSITION_1.IN_POSITION AND "DB149_CLADDING_SPINDLE_C23".SAFETY_POSITIONS.SAFETY_POSITION_1.IN_POSITION AND "DB150_CLADDING_SPINDLE_C24".SAFETY_POSITIONS.SAFETY_POSITION_1.IN_POSITION) OR "DB1262_HOME_UNIT_02_STATION_0".SEQUENCE.RUNNING);
   "DB145_CLADDING_AXIS_E20".FEED_HOLD_COND := "M_ONE" AND (("DB8000_PART_STATUS".UNIT_02.FIXTURE_1.PART_A.STATUS.PRESENT AND ("DB3500_UNIT_02_FIXTURE_1".CLAMPED_WITH_PART_ANALOG OR "DB3510_U2_F1_GRIPPER".CYL.FULL_CLOSED)) OR NOT "DB8000_PART_STATUS".UNIT_02.FIXTURE_1.PART_A.STATUS.PRESENT) AND (("DB8000_PART_STATUS".UNIT_02.FIXTURE_2.PART_A.STATUS.PRESENT AND ("DB3600_UNIT_02_FIXTURE_2".CLAMPED_WITH_PART_ANALOG OR "DB3610_U2_F2_GRIPPER".CYL.FULL_CLOSED)) OR NOT "DB8000_PART_STATUS".UNIT_02.FIXTURE_2.PART_A.STATUS.PRESENT) AND (("DB8000_PART_STATUS".UNIT_02.FIXTURE_3.PART_A.STATUS.PRESENT AND ("DB3700_UNIT_02_FIXTURE_3".CLAMPED_WITH_PART_ANALOG OR "DB3710_U2_F3_GRIPPER".CYL.FULL_CLOSED)) OR NOT "DB8000_PART_STATUS".UNIT_02.FIXTURE_3.PART_A.STATUS.PRESENT) AND (("DB8000_PART_STATUS".UNIT_02.FIXTURE_4.PART_A.STATUS.PRESENT AND ("DB3800_UNIT_02_FIXTURE_4".CLAMPED_WITH_PART_ANALOG OR "DB3810_U2_F4_GRIPPER".CYL.FULL_CLOSED)) OR NOT "DB8000_PART_STATUS".UNIT_02.FIXTURE_4.PART_A.STATUS.PRESENT) AND (("DB4000_FIX_TABLE_POSITIONS".UNIT_02.FIXTURE_1.IN_LOAD_UNLOAD_STATION_1 AND NOT "DB3500_UNIT_02_FIXTURE_1".PART_TYPE_DISCORDANCY) OR ("DB4000_FIX_TABLE_POSITIONS".UNIT_02.FIXTURE_2.IN_LOAD_UNLOAD_STATION_1 AND NOT "DB3600_UNIT_02_FIXTURE_2".PART_TYPE_DISCORDANCY) OR ("DB4000_FIX_TABLE_POSITIONS".UNIT_02.FIXTURE_3.IN_LOAD_UNLOAD_STATION_1 AND NOT "DB3700_UNIT_02_FIXTURE_3".PART_TYPE_DISCORDANCY) OR ("DB4000_FIX_TABLE_POSITIONS".UNIT_02.FIXTURE_4.IN_LOAD_UNLOAD_STATION_1 AND NOT "DB3800_UNIT_02_FIXTURE_4".PART_TYPE_DISCORDANCY) OR "DB4000_FIX_TABLE_POSITIONS".UNIT_02.AXIS_E20_NOT_DEFINED_POS) AND "DB145_CLADDING_AXIS_E20".MOVE_AXIS AND (("BIMANUAL_1_U02_I" AND "BIMANUAL_2_U02_I") OR NOT "DB2001_MODES_GENERAL".GENERAL.AUTO_SINGLE_SEMI_SELECTED OR (NOT "DB2031_CYCLES_GENERAL".MANUAL_LOAD_CYCLE.CYCLE_SELECTED AND "DB2031_CYCLES_GENERAL".DRY_CYCLE.CYCLE_SELECTED));
END_REGION

REGION Network 15: CALL FB32 AXIS E20
   // 2#0000_0001 OPTIONS 0 BIT 0 MEASURING SYSTEM 2 OPTION
   // 2#0000_0010 OPTIONS 0 BIT 1 ENABLE FC18 OPTION
   // 2#0000_0100 OPTIONS 0 BIT 2 FC18 EXTERNAL POSITION OPTION
   // 2#0000_1000 OPTIONS 0 BIT 3 AXIS B ENABLE FAULTS OPTION
   // 2#0001_0000 OPTIONS 0 BIT 4 SPARE OPTION
   // 2#0010_0000 OPTIONS 0 BIT 5 SPARE OPTION
   // 2#0100_0000 OPTIONS 0 BIT 6 SPARE OPTION
   // 2#1000_0000 OPTIONS 0 BIT 7 SPARE OPTION
   // 
   // 2#0000_0001 OPTIONS 1 BIT 0 AXIS ROLLER OPTION
   // 2#0000_0010 OPTIONS 1 BIT 1 MASTER AXIS OPTION
   // 2#0000_0100 OPTIONS 1 BIT 2 SLAVE AXIS OPTION
   // 2#0000_1000 OPTIONS 1 BIT 3 MASTER-SLAVE AXES INDEPENDENT MOVEMENT WITH HT10 OPTION
   // 2#0001_0000 OPTIONS 1 BIT 4 GANTRY MODE MASTER AXIS OPTION
   // 2#0010_0000 OPTIONS 1 BIT 5 SPARE OPTION
   // 2#0100_0000 OPTIONS 1 BIT 6 SPARE OPTION
   // 2#1000_0000 OPTIONS 1 BIT 7 SPARE OPTION
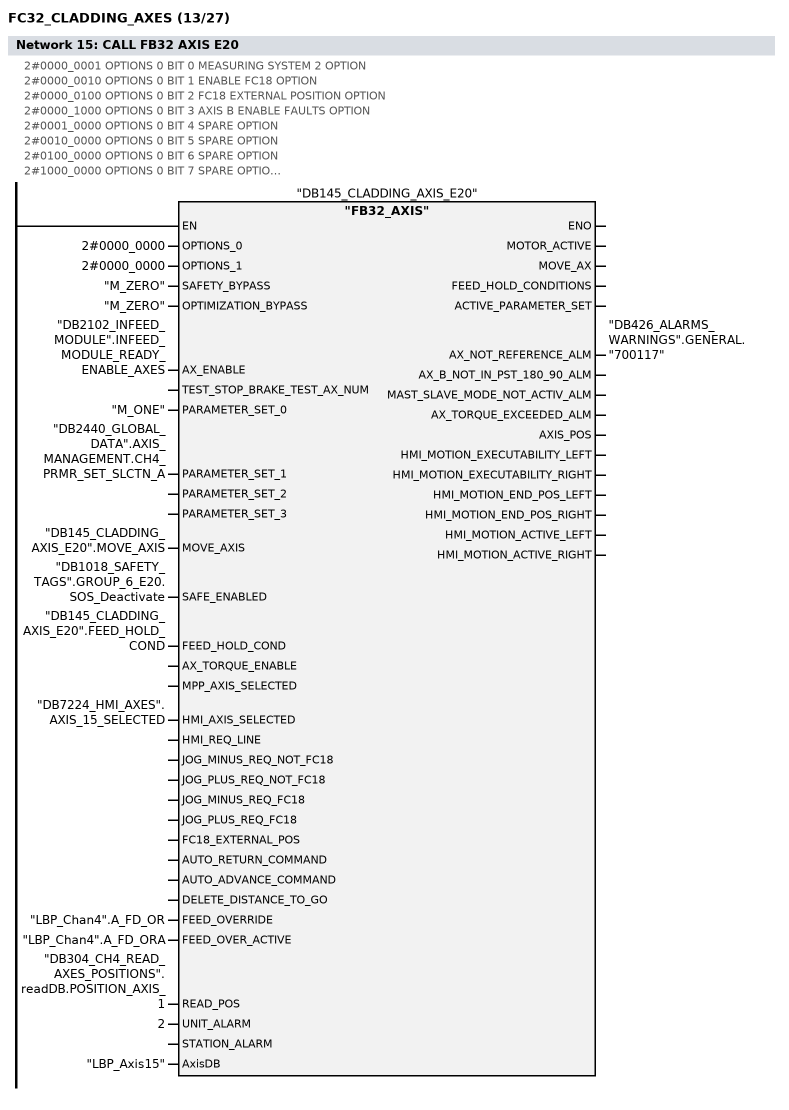
   RUNG wire#powerrail
      "DB145_CLADDING_AXIS_E20"(OPTIONS_0 := 2#0000_0000, OPTIONS_1 := 2#0000_0000, SAFETY_BYPASS := "M_ZERO", OPTIMIZATION_BYPASS := "M_ZERO", AX_ENABLE := "DB2102_INFEED_MODULE".INFEED_MODULE_READY_ENABLE_AXES, TEST_STOP_BRAKE_TEST_AX_NUM :=, PARAMETER_SET_0 := "M_ONE", PARAMETER_SET_1 := "DB2440_GLOBAL_DATA".AXIS_MANAGEMENT.CH4_PRMR_SET_SLCTN_A, PARAMETER_SET_2 :=, PARAMETER_SET_3 :=, MOVE_AXIS := "DB145_CLADDING_AXIS_E20".MOVE_AXIS, SAFE_ENABLED := "DB1018_SAFETY_TAGS".GROUP_6_E20.SOS_Deactivate, FEED_HOLD_COND := "DB145_CLADDING_AXIS_E20".FEED_HOLD_COND, AX_TORQUE_ENABLE :=, MPP_AXIS_SELECTED :=, HMI_AXIS_SELECTED := "DB7224_HMI_AXES".AXIS_15_SELECTED, HMI_REQ_LINE :=, JOG_MINUS_REQ_NOT_FC18 :=, JOG_PLUS_REQ_NOT_FC18 :=, JOG_MINUS_REQ_FC18 :=, JOG_PLUS_REQ_FC18 :=, FC18_EXTERNAL_POS :=, AUTO_RETURN_COMMAND :=, AUTO_ADVANCE_COMMAND :=, DELETE_DISTANCE_TO_GO :=, FEED_OVERRIDE := "LBP_Chan4".A_FD_OR, FEED_OVER_ACTIVE := "LBP_Chan4".A_FD_ORA, READ_POS := "DB304_CH4_READ_AXES_POSITIONS".readDB.POSITION_AXIS_1, UNIT_ALARM := 2, STATION_ALARM :=, AxisDB := "LBP_Axis15", MOTOR_ACTIVE =>, MOVE_AX =>, FEED_HOLD_CONDITIONS =>, ACTIVE_PARAMETER_SET =>, AX_NOT_REFERENCE_ALM => "DB426_ALARMS_WARNINGS".GENERAL."700117", AX_B_NOT_IN_PST_180_90_ALM =>, MAST_SLAVE_MODE_NOT_ACTIV_ALM =>, AX_TORQUE_EXCEEDED_ALM =>, AXIS_POS =>, HMI_MOTION_EXECUTABILITY_LEFT =>, HMI_MOTION_EXECUTABILITY_RIGHT =>, HMI_MOTION_END_POS_LEFT =>, HMI_MOTION_END_POS_RIGHT =>, HMI_MOTION_ACTIVE_LEFT =>, HMI_MOTION_ACTIVE_RIGHT =>)
   END_RUNG
   // the same network as SCL:
   "DB145_CLADDING_AXIS_E20"(OPTIONS_0 := 2#0000_0000,   // "FB32_AXIS"
                           OPTIONS_1 := 2#0000_0000,
                           SAFETY_BYPASS := "M_ZERO",
                           OPTIMIZATION_BYPASS := "M_ZERO",
                           AX_ENABLE := "DB2102_INFEED_MODULE".INFEED_MODULE_READY_ENABLE_AXES,
                           PARAMETER_SET_0 := "M_ONE",
                           PARAMETER_SET_1 := "DB2440_GLOBAL_DATA".AXIS_MANAGEMENT.CH4_PRMR_SET_SLCTN_A,
                           MOVE_AXIS := "DB145_CLADDING_AXIS_E20".MOVE_AXIS,
                           SAFE_ENABLED := "DB1018_SAFETY_TAGS".GROUP_6_E20.SOS_Deactivate,
                           FEED_HOLD_COND := "DB145_CLADDING_AXIS_E20".FEED_HOLD_COND,
                           HMI_AXIS_SELECTED := "DB7224_HMI_AXES".AXIS_15_SELECTED,
                           FEED_OVERRIDE := "LBP_Chan4".A_FD_OR,
                           FEED_OVER_ACTIVE := "LBP_Chan4".A_FD_ORA,
                           READ_POS := "DB304_CH4_READ_AXES_POSITIONS".readDB.POSITION_AXIS_1,
                           UNIT_ALARM := 2,
                           AxisDB := "LBP_Axis15",
                           AX_NOT_REFERENCE_ALM => "DB426_ALARMS_WARNINGS".GENERAL."700117");
END_REGION

REGION Network 16: AXIS E20 OPERATOR HELP
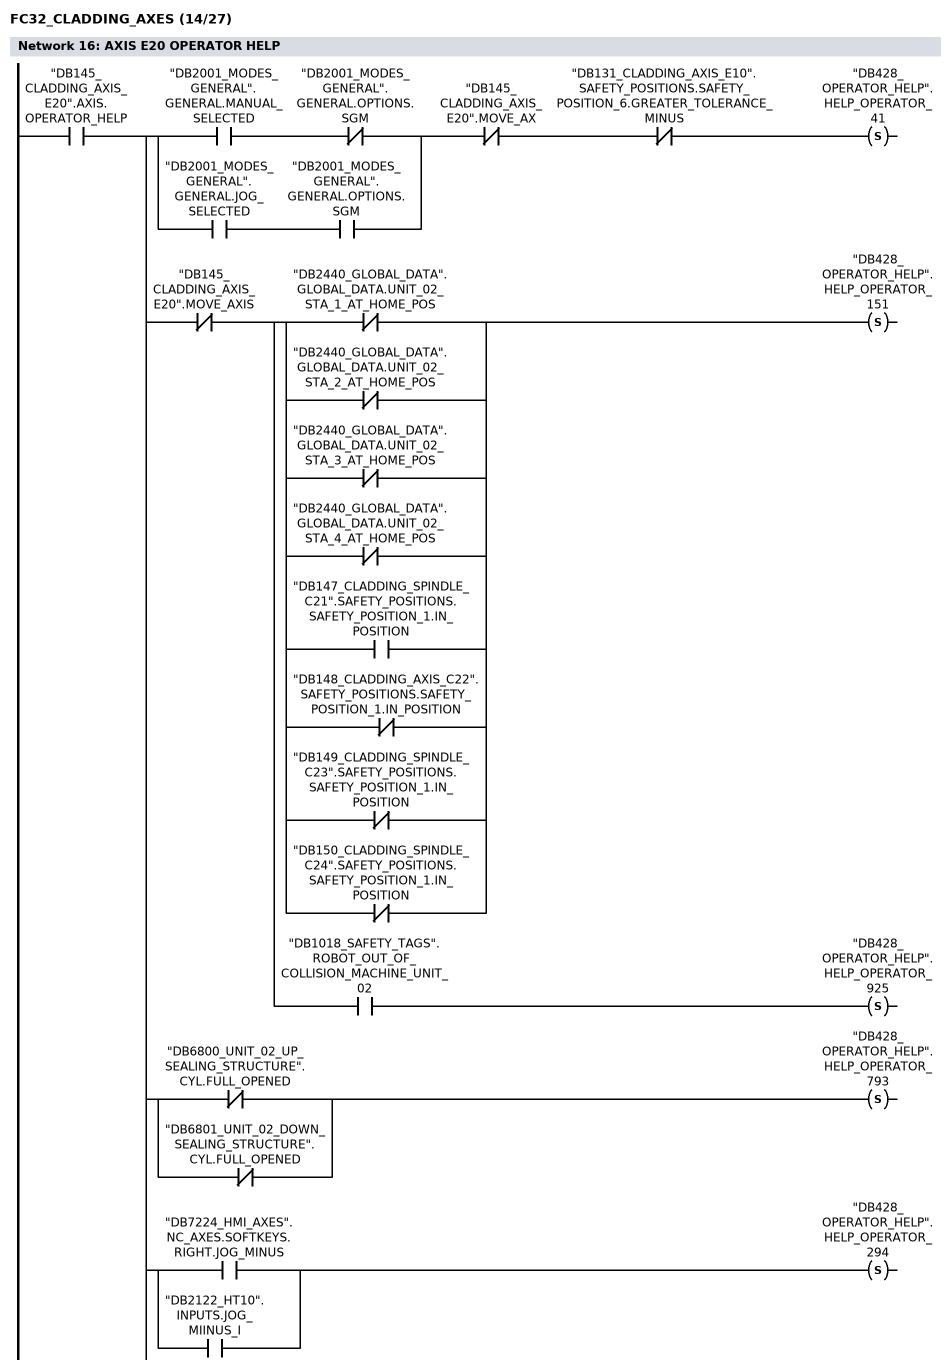
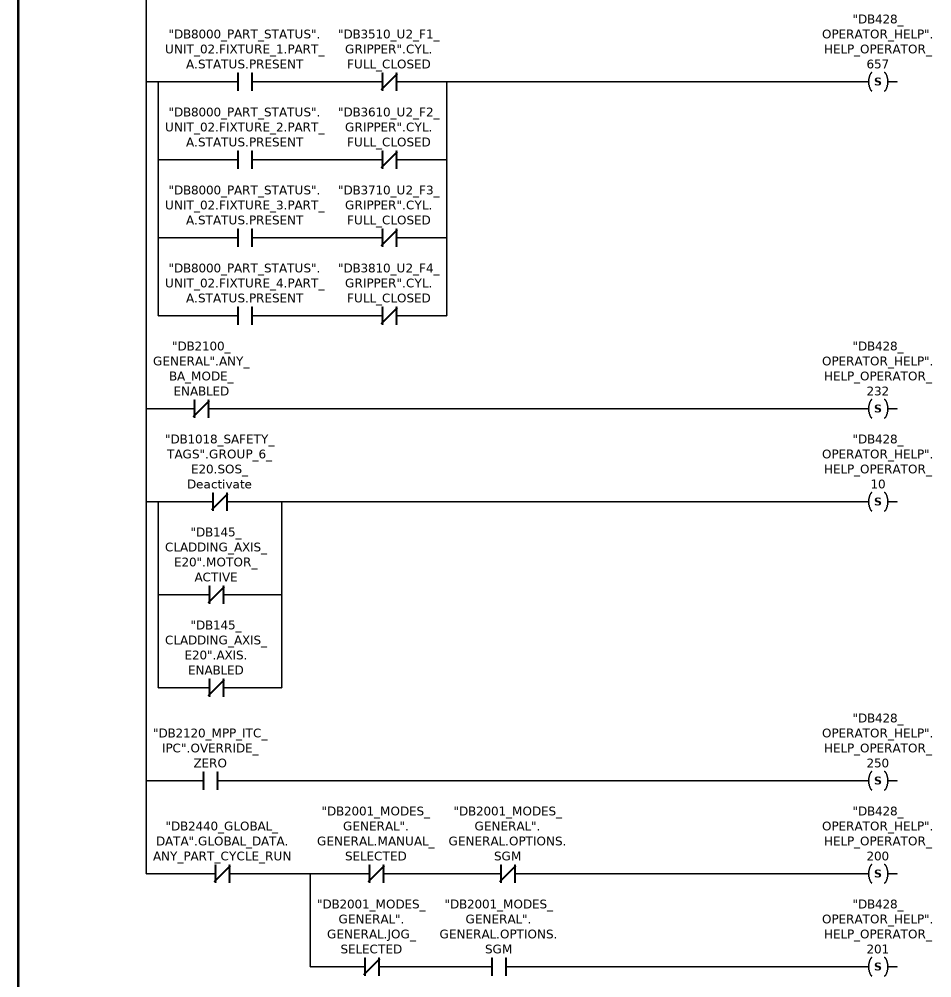
   RUNG wire#powerrail
      Contact( "DB145_CLADDING_AXIS_E20".AXIS.OPERATOR_HELP )
      wire#w1
      Contact( "DB2001_MODES_GENERAL".GENERAL.MANUAL_SELECTED )
      I_Contact( "DB2001_MODES_GENERAL".GENERAL.OPTIONS.SGM )
      wire#w2
      I_Contact( "DB145_CLADDING_AXIS_E20".MOVE_AX )
      I_Contact( "DB131_CLADDING_AXIS_E10".SAFETY_POSITIONS.SAFETY_POSITION_6.GREATER_TOLERANCE_MINUS )
      S_Coil( "DB428_OPERATOR_HELP".HELP_OPERATOR_41 )
   END_RUNG
   RUNG wire#w1
      Contact( "DB2001_MODES_GENERAL".GENERAL.JOG_SELECTED )
      Contact( "DB2001_MODES_GENERAL".GENERAL.OPTIONS.SGM )
   END_RUNG wire#w2
   RUNG wire#w1
      I_Contact( "DB145_CLADDING_AXIS_E20".MOVE_AXIS )
      wire#w3
      I_Contact( "DB2440_GLOBAL_DATA".GLOBAL_DATA.UNIT_02_STA_1_AT_HOME_POS )
      wire#w4
      S_Coil( "DB428_OPERATOR_HELP".HELP_OPERATOR_151 )
   END_RUNG
   RUNG wire#w3
      I_Contact( "DB2440_GLOBAL_DATA".GLOBAL_DATA.UNIT_02_STA_2_AT_HOME_POS )
   END_RUNG wire#w4
   RUNG wire#w3
      I_Contact( "DB2440_GLOBAL_DATA".GLOBAL_DATA.UNIT_02_STA_3_AT_HOME_POS )
   END_RUNG wire#w4
   RUNG wire#w3
      I_Contact( "DB2440_GLOBAL_DATA".GLOBAL_DATA.UNIT_02_STA_4_AT_HOME_POS )
   END_RUNG wire#w4
   RUNG wire#w3
      Contact( "DB147_CLADDING_SPINDLE_C21".SAFETY_POSITIONS.SAFETY_POSITION_1.IN_POSITION )
   END_RUNG wire#w4
   RUNG wire#w3
      I_Contact( "DB148_CLADDING_AXIS_C22".SAFETY_POSITIONS.SAFETY_POSITION_1.IN_POSITION )
   END_RUNG wire#w4
   RUNG wire#w3
      I_Contact( "DB149_CLADDING_SPINDLE_C23".SAFETY_POSITIONS.SAFETY_POSITION_1.IN_POSITION )
   END_RUNG wire#w4
   RUNG wire#w3
      I_Contact( "DB150_CLADDING_SPINDLE_C24".SAFETY_POSITIONS.SAFETY_POSITION_1.IN_POSITION )
   END_RUNG wire#w4
   RUNG wire#w3
      Contact( "DB1018_SAFETY_TAGS".ROBOT_OUT_OF_COLLISION_MACHINE_UNIT_02 )
      S_Coil( "DB428_OPERATOR_HELP".HELP_OPERATOR_925 )
   END_RUNG
   RUNG wire#w1
      I_Contact( "DB6800_UNIT_02_UP_SEALING_STRUCTURE".CYL.FULL_OPENED )
      wire#w5
      S_Coil( "DB428_OPERATOR_HELP".HELP_OPERATOR_793 )
   END_RUNG
   RUNG wire#w1
      I_Contact( "DB6801_UNIT_02_DOWN_SEALING_STRUCTURE".CYL.FULL_OPENED )
   END_RUNG wire#w5
   RUNG wire#w1
      Contact( "DB7224_HMI_AXES".NC_AXES.SOFTKEYS.RIGHT.JOG_MINUS )
      wire#w6
      S_Coil( "DB428_OPERATOR_HELP".HELP_OPERATOR_294 )
   END_RUNG
   RUNG wire#w1
      Contact( "DB2122_HT10".INPUTS.JOG_MIINUS_I )
   END_RUNG wire#w6
   RUNG wire#w1
      Contact( "DB8000_PART_STATUS".UNIT_02.FIXTURE_1.PART_A.STATUS.PRESENT )
      I_Contact( "DB3510_U2_F1_GRIPPER".CYL.FULL_CLOSED )
      wire#w7
      S_Coil( "DB428_OPERATOR_HELP".HELP_OPERATOR_657 )
   END_RUNG
   RUNG wire#w1
      Contact( "DB8000_PART_STATUS".UNIT_02.FIXTURE_2.PART_A.STATUS.PRESENT )
      I_Contact( "DB3610_U2_F2_GRIPPER".CYL.FULL_CLOSED )
   END_RUNG wire#w7
   RUNG wire#w1
      Contact( "DB8000_PART_STATUS".UNIT_02.FIXTURE_3.PART_A.STATUS.PRESENT )
      I_Contact( "DB3710_U2_F3_GRIPPER".CYL.FULL_CLOSED )
   END_RUNG wire#w7
   RUNG wire#w1
      Contact( "DB8000_PART_STATUS".UNIT_02.FIXTURE_4.PART_A.STATUS.PRESENT )
      I_Contact( "DB3810_U2_F4_GRIPPER".CYL.FULL_CLOSED )
   END_RUNG wire#w7
   RUNG wire#w1
      I_Contact( "DB2100_GENERAL".ANY_BA_MODE_ENABLED )
      S_Coil( "DB428_OPERATOR_HELP".HELP_OPERATOR_232 )
   END_RUNG
   RUNG wire#w1
      I_Contact( "DB1018_SAFETY_TAGS".GROUP_6_E20.SOS_Deactivate )
      wire#w8
      S_Coil( "DB428_OPERATOR_HELP".HELP_OPERATOR_10 )
   END_RUNG
   RUNG wire#w1
      I_Contact( "DB145_CLADDING_AXIS_E20".MOTOR_ACTIVE )
   END_RUNG wire#w8
   RUNG wire#w1
      I_Contact( "DB145_CLADDING_AXIS_E20".AXIS.ENABLED )
   END_RUNG wire#w8
   RUNG wire#w1
      Contact( "DB2120_MPP_ITC_IPC".OVERRIDE_ZERO )
      S_Coil( "DB428_OPERATOR_HELP".HELP_OPERATOR_250 )
   END_RUNG
   RUNG wire#w1
      I_Contact( "DB2440_GLOBAL_DATA".GLOBAL_DATA.ANY_PART_CYCLE_RUN )
      wire#w9
      I_Contact( "DB2001_MODES_GENERAL".GENERAL.MANUAL_SELECTED )
      I_Contact( "DB2001_MODES_GENERAL".GENERAL.OPTIONS.SGM )
      S_Coil( "DB428_OPERATOR_HELP".HELP_OPERATOR_200 )
   END_RUNG
   RUNG wire#w9
      I_Contact( "DB2001_MODES_GENERAL".GENERAL.JOG_SELECTED )
      Contact( "DB2001_MODES_GENERAL".GENERAL.OPTIONS.SGM )
      S_Coil( "DB428_OPERATOR_HELP".HELP_OPERATOR_201 )
   END_RUNG
   // the same network as SCL:
   IF "DB145_CLADDING_AXIS_E20".AXIS.OPERATOR_HELP AND (("DB2001_MODES_GENERAL".GENERAL.MANUAL_SELECTED AND NOT "DB2001_MODES_GENERAL".GENERAL.OPTIONS.SGM) OR ("DB2001_MODES_GENERAL".GENERAL.JOG_SELECTED AND "DB2001_MODES_GENERAL".GENERAL.OPTIONS.SGM)) AND NOT "DB145_CLADDING_AXIS_E20".MOVE_AX AND NOT "DB131_CLADDING_AXIS_E10".SAFETY_POSITIONS.SAFETY_POSITION_6.GREATER_TOLERANCE_MINUS THEN
       "DB428_OPERATOR_HELP".HELP_OPERATOR_41 := TRUE;
   END_IF;
   #_w1 := "DB145_CLADDING_AXIS_E20".AXIS.OPERATOR_HELP AND NOT "DB145_CLADDING_AXIS_E20".MOVE_AXIS;
   IF #_w1 AND (NOT "DB2440_GLOBAL_DATA".GLOBAL_DATA.UNIT_02_STA_1_AT_HOME_POS OR NOT "DB2440_GLOBAL_DATA".GLOBAL_DATA.UNIT_02_STA_2_AT_HOME_POS OR NOT "DB2440_GLOBAL_DATA".GLOBAL_DATA.UNIT_02_STA_3_AT_HOME_POS OR NOT "DB2440_GLOBAL_DATA".GLOBAL_DATA.UNIT_02_STA_4_AT_HOME_POS OR "DB147_CLADDING_SPINDLE_C21".SAFETY_POSITIONS.SAFETY_POSITION_1.IN_POSITION OR NOT "DB148_CLADDING_AXIS_C22".SAFETY_POSITIONS.SAFETY_POSITION_1.IN_POSITION OR NOT "DB149_CLADDING_SPINDLE_C23".SAFETY_POSITIONS.SAFETY_POSITION_1.IN_POSITION OR NOT "DB150_CLADDING_SPINDLE_C24".SAFETY_POSITIONS.SAFETY_POSITION_1.IN_POSITION) THEN
       "DB428_OPERATOR_HELP".HELP_OPERATOR_151 := TRUE;
   END_IF;
   IF #_w1 AND "DB1018_SAFETY_TAGS".ROBOT_OUT_OF_COLLISION_MACHINE_UNIT_02 THEN
       "DB428_OPERATOR_HELP".HELP_OPERATOR_925 := TRUE;
   END_IF;
   IF "DB145_CLADDING_AXIS_E20".AXIS.OPERATOR_HELP AND (NOT "DB6800_UNIT_02_UP_SEALING_STRUCTURE".CYL.FULL_OPENED OR NOT "DB6801_UNIT_02_DOWN_SEALING_STRUCTURE".CYL.FULL_OPENED) THEN
       "DB428_OPERATOR_HELP".HELP_OPERATOR_793 := TRUE;
   END_IF;
   IF "DB145_CLADDING_AXIS_E20".AXIS.OPERATOR_HELP AND ("DB7224_HMI_AXES".NC_AXES.SOFTKEYS.RIGHT.JOG_MINUS OR "DB2122_HT10".INPUTS.JOG_MIINUS_I) THEN
       "DB428_OPERATOR_HELP".HELP_OPERATOR_294 := TRUE;
   END_IF;
   IF "DB145_CLADDING_AXIS_E20".AXIS.OPERATOR_HELP AND (("DB8000_PART_STATUS".UNIT_02.FIXTURE_1.PART_A.STATUS.PRESENT AND NOT "DB3510_U2_F1_GRIPPER".CYL.FULL_CLOSED) OR ("DB8000_PART_STATUS".UNIT_02.FIXTURE_2.PART_A.STATUS.PRESENT AND NOT "DB3610_U2_F2_GRIPPER".CYL.FULL_CLOSED) OR ("DB8000_PART_STATUS".UNIT_02.FIXTURE_3.PART_A.STATUS.PRESENT AND NOT "DB3710_U2_F3_GRIPPER".CYL.FULL_CLOSED) OR ("DB8000_PART_STATUS".UNIT_02.FIXTURE_4.PART_A.STATUS.PRESENT AND NOT "DB3810_U2_F4_GRIPPER".CYL.FULL_CLOSED)) THEN
       "DB428_OPERATOR_HELP".HELP_OPERATOR_657 := TRUE;
   END_IF;
   IF "DB145_CLADDING_AXIS_E20".AXIS.OPERATOR_HELP AND NOT "DB2100_GENERAL".ANY_BA_MODE_ENABLED THEN
       "DB428_OPERATOR_HELP".HELP_OPERATOR_232 := TRUE;
   END_IF;
   IF "DB145_CLADDING_AXIS_E20".AXIS.OPERATOR_HELP AND (NOT "DB1018_SAFETY_TAGS".GROUP_6_E20.SOS_Deactivate OR NOT "DB145_CLADDING_AXIS_E20".MOTOR_ACTIVE OR NOT "DB145_CLADDING_AXIS_E20".AXIS.ENABLED) THEN
       "DB428_OPERATOR_HELP".HELP_OPERATOR_10 := TRUE;
   END_IF;
   IF "DB145_CLADDING_AXIS_E20".AXIS.OPERATOR_HELP AND "DB2120_MPP_ITC_IPC".OVERRIDE_ZERO THEN
       "DB428_OPERATOR_HELP".HELP_OPERATOR_250 := TRUE;
   END_IF;
   #_w2 := "DB145_CLADDING_AXIS_E20".AXIS.OPERATOR_HELP AND NOT "DB2440_GLOBAL_DATA".GLOBAL_DATA.ANY_PART_CYCLE_RUN;
   IF #_w2 AND NOT "DB2001_MODES_GENERAL".GENERAL.MANUAL_SELECTED AND NOT "DB2001_MODES_GENERAL".GENERAL.OPTIONS.SGM THEN
       "DB428_OPERATOR_HELP".HELP_OPERATOR_200 := TRUE;
   END_IF;
   IF #_w2 AND NOT "DB2001_MODES_GENERAL".GENERAL.JOG_SELECTED AND "DB2001_MODES_GENERAL".GENERAL.OPTIONS.SGM THEN
       "DB428_OPERATOR_HELP".HELP_OPERATOR_201 := TRUE;
   END_IF;
END_REGION

REGION Network 17: AXIS C22 MOVE AXIS AND FEED HOLD CONDITIONS
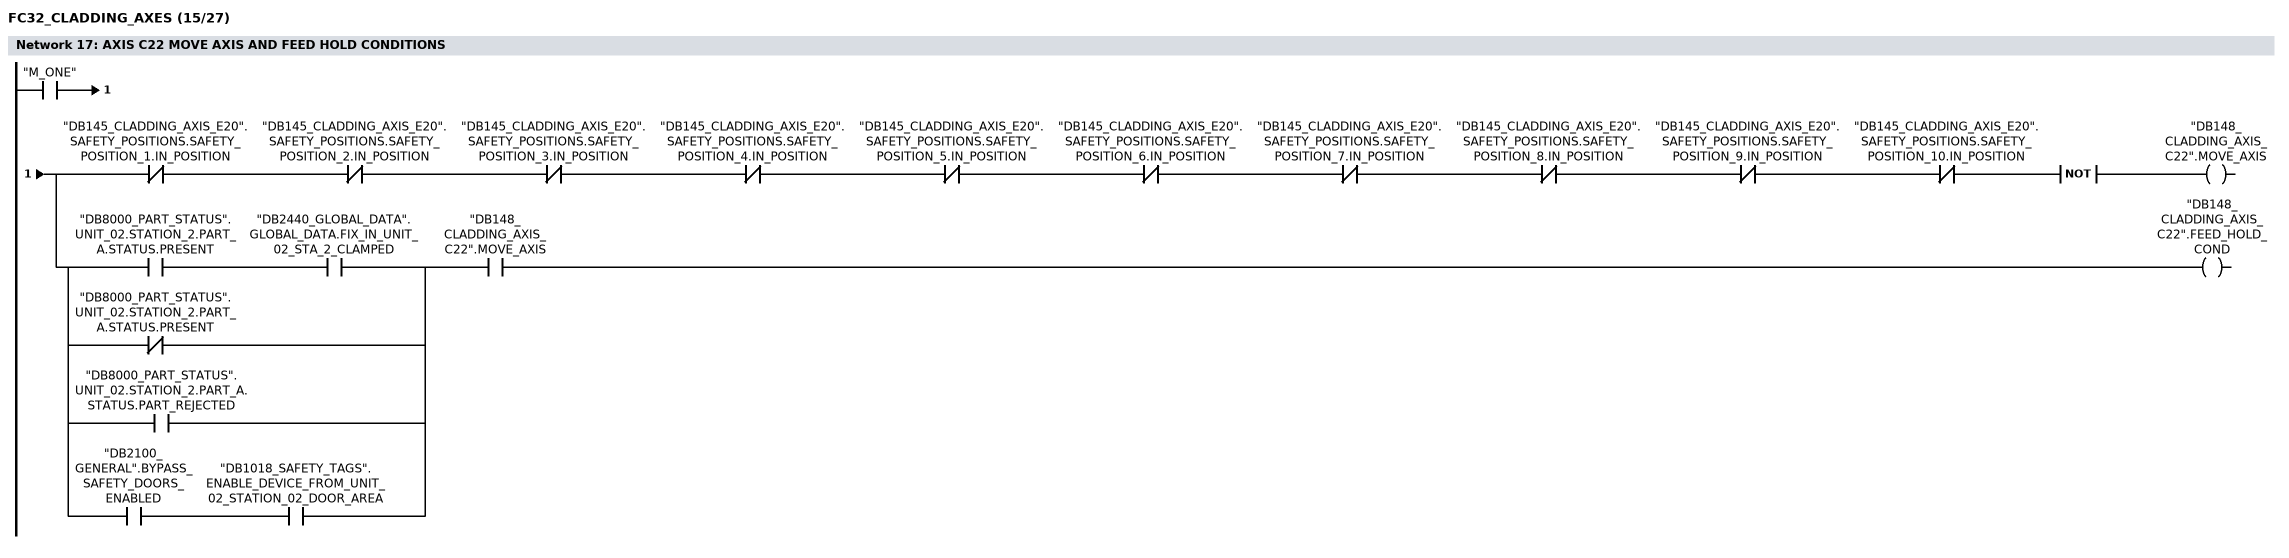
   RUNG wire#powerrail
      Contact( "M_ONE" )
      wire#w1
      I_Contact( "DB145_CLADDING_AXIS_E20".SAFETY_POSITIONS.SAFETY_POSITION_1.IN_POSITION )
      I_Contact( "DB145_CLADDING_AXIS_E20".SAFETY_POSITIONS.SAFETY_POSITION_2.IN_POSITION )
      I_Contact( "DB145_CLADDING_AXIS_E20".SAFETY_POSITIONS.SAFETY_POSITION_3.IN_POSITION )
      I_Contact( "DB145_CLADDING_AXIS_E20".SAFETY_POSITIONS.SAFETY_POSITION_4.IN_POSITION )
      I_Contact( "DB145_CLADDING_AXIS_E20".SAFETY_POSITIONS.SAFETY_POSITION_5.IN_POSITION )
      I_Contact( "DB145_CLADDING_AXIS_E20".SAFETY_POSITIONS.SAFETY_POSITION_6.IN_POSITION )
      I_Contact( "DB145_CLADDING_AXIS_E20".SAFETY_POSITIONS.SAFETY_POSITION_7.IN_POSITION )
      I_Contact( "DB145_CLADDING_AXIS_E20".SAFETY_POSITIONS.SAFETY_POSITION_8.IN_POSITION )
      I_Contact( "DB145_CLADDING_AXIS_E20".SAFETY_POSITIONS.SAFETY_POSITION_9.IN_POSITION )
      I_Contact( "DB145_CLADDING_AXIS_E20".SAFETY_POSITIONS.SAFETY_POSITION_10.IN_POSITION )
      Not()
      Coil( "DB148_CLADDING_AXIS_C22".MOVE_AXIS )
   END_RUNG
   RUNG wire#w1
      Contact( "DB8000_PART_STATUS".UNIT_02.STATION_2.PART_A.STATUS.PRESENT )
      Contact( "DB2440_GLOBAL_DATA".GLOBAL_DATA.FIX_IN_UNIT_02_STA_2_CLAMPED )
      wire#w2
      Contact( "DB148_CLADDING_AXIS_C22".MOVE_AXIS )
      Coil( "DB148_CLADDING_AXIS_C22".FEED_HOLD_COND )
   END_RUNG
   RUNG wire#w1
      I_Contact( "DB8000_PART_STATUS".UNIT_02.STATION_2.PART_A.STATUS.PRESENT )
   END_RUNG wire#w2
   RUNG wire#w1
      Contact( "DB8000_PART_STATUS".UNIT_02.STATION_2.PART_A.STATUS.PART_REJECTED )
   END_RUNG wire#w2
   RUNG wire#w1
      Contact( "DB2100_GENERAL".BYPASS_SAFETY_DOORS_ENABLED )
      Contact( "DB1018_SAFETY_TAGS".ENABLE_DEVICE_FROM_UNIT_02_STATION_02_DOOR_AREA )
   END_RUNG wire#w2
   // the same network as SCL:
   "DB148_CLADDING_AXIS_C22".MOVE_AXIS := NOT ("M_ONE" AND NOT "DB145_CLADDING_AXIS_E20".SAFETY_POSITIONS.SAFETY_POSITION_1.IN_POSITION AND NOT "DB145_CLADDING_AXIS_E20".SAFETY_POSITIONS.SAFETY_POSITION_2.IN_POSITION AND NOT "DB145_CLADDING_AXIS_E20".SAFETY_POSITIONS.SAFETY_POSITION_3.IN_POSITION AND NOT "DB145_CLADDING_AXIS_E20".SAFETY_POSITIONS.SAFETY_POSITION_4.IN_POSITION AND NOT "DB145_CLADDING_AXIS_E20".SAFETY_POSITIONS.SAFETY_POSITION_5.IN_POSITION AND NOT "DB145_CLADDING_AXIS_E20".SAFETY_POSITIONS.SAFETY_POSITION_6.IN_POSITION AND NOT "DB145_CLADDING_AXIS_E20".SAFETY_POSITIONS.SAFETY_POSITION_7.IN_POSITION AND NOT "DB145_CLADDING_AXIS_E20".SAFETY_POSITIONS.SAFETY_POSITION_8.IN_POSITION AND NOT "DB145_CLADDING_AXIS_E20".SAFETY_POSITIONS.SAFETY_POSITION_9.IN_POSITION AND NOT "DB145_CLADDING_AXIS_E20".SAFETY_POSITIONS.SAFETY_POSITION_10.IN_POSITION);
   "DB148_CLADDING_AXIS_C22".FEED_HOLD_COND := "M_ONE" AND (("DB8000_PART_STATUS".UNIT_02.STATION_2.PART_A.STATUS.PRESENT AND "DB2440_GLOBAL_DATA".GLOBAL_DATA.FIX_IN_UNIT_02_STA_2_CLAMPED) OR NOT "DB8000_PART_STATUS".UNIT_02.STATION_2.PART_A.STATUS.PRESENT OR "DB8000_PART_STATUS".UNIT_02.STATION_2.PART_A.STATUS.PART_REJECTED OR ("DB2100_GENERAL".BYPASS_SAFETY_DOORS_ENABLED AND "DB1018_SAFETY_TAGS".ENABLE_DEVICE_FROM_UNIT_02_STATION_02_DOOR_AREA)) AND "DB148_CLADDING_AXIS_C22".MOVE_AXIS;
END_REGION

REGION Network 18: CALL FB32 AXIS C22
   // 2#0000_0001 OPTIONS 0 BIT 0 MEASURING SYSTEM 2 OPTION
   // 2#0000_0010 OPTIONS 0 BIT 1 ENABLE FC18 OPTION
   // 2#0000_0100 OPTIONS 0 BIT 2 FC18 EXTERNAL POSITION OPTION
   // 2#0000_1000 OPTIONS 0 BIT 3 AXIS B ENABLE FAULTS OPTION
   // 2#0001_0000 OPTIONS 0 BIT 4 SPARE OPTION
   // 2#0010_0000 OPTIONS 0 BIT 5 SPARE OPTION
   // 2#0100_0000 OPTIONS 0 BIT 6 SPARE OPTION
   // 2#1000_0000 OPTIONS 0 BIT 7 SPARE OPTION
   // 
   // 2#0000_0001 OPTIONS 1 BIT 0 AXIS ROLLER OPTION
   // 2#0000_0010 OPTIONS 1 BIT 1 MASTER AXIS OPTION
   // 2#0000_0100 OPTIONS 1 BIT 2 SLAVE AXIS OPTION
   // 2#0000_1000 OPTIONS 1 BIT 3 MASTER-SLAVE AXES INDEPENDENT MOVEMENT WITH HT10 OPTION
   // 2#0001_0000 OPTIONS 1 BIT 4 GANTRY MODE MASTER AXIS OPTION
   // 2#0010_0000 OPTIONS 1 BIT 5 SPARE OPTION
   // 2#0100_0000 OPTIONS 1 BIT 6 SPARE OPTION
   // 2#1000_0000 OPTIONS 1 BIT 7 SPARE OPTION
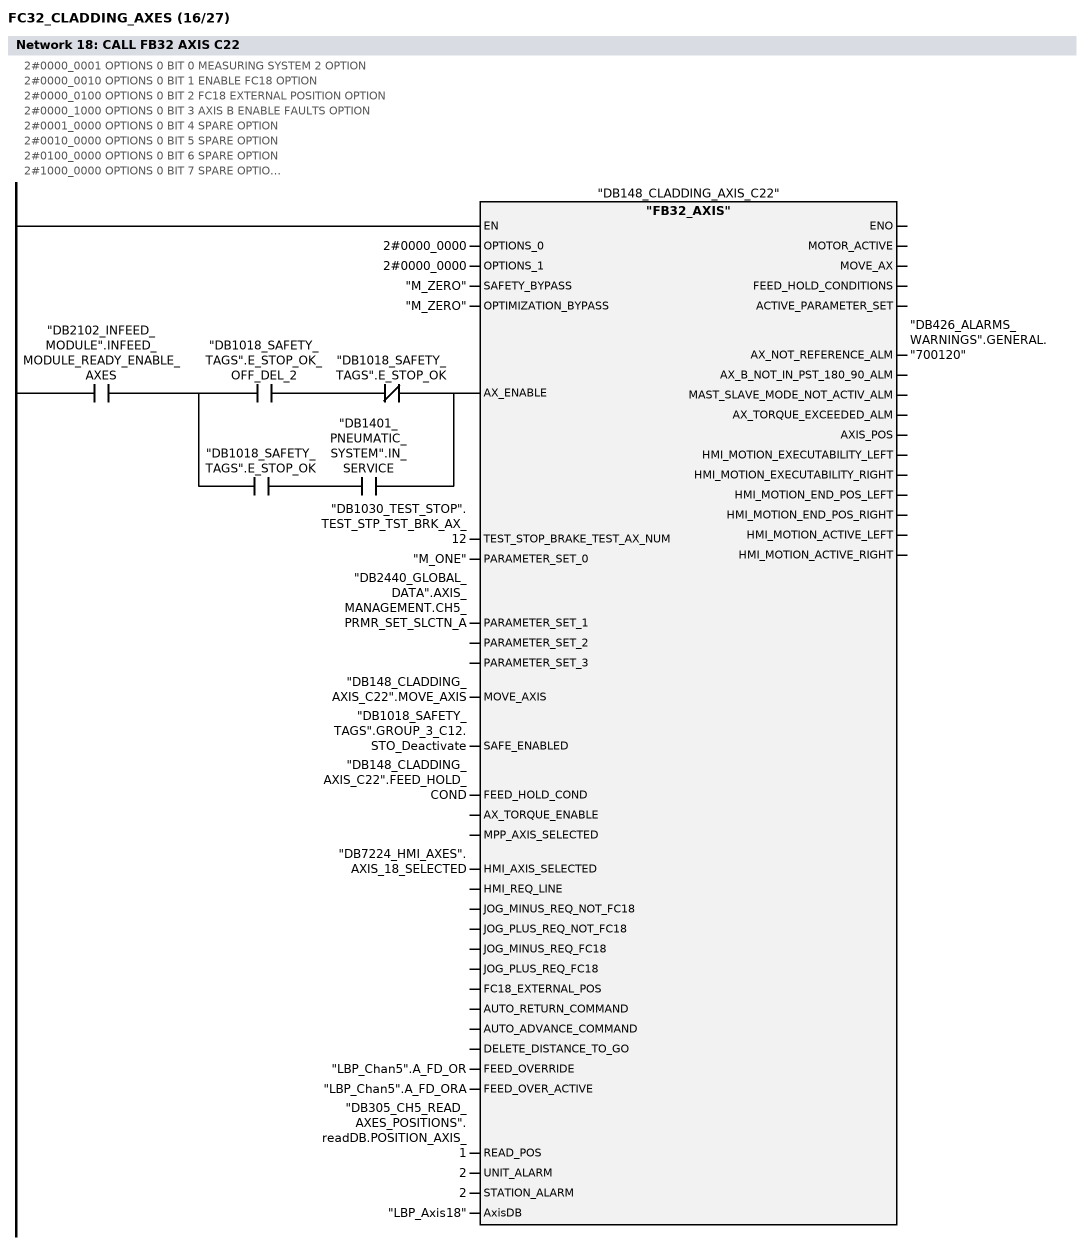
   RUNG wire#powerrail
      "DB148_CLADDING_AXIS_C22"(AX_ENABLE := wire#w2, OPTIONS_0 := 2#0000_0000, OPTIONS_1 := 2#0000_0000, SAFETY_BYPASS := "M_ZERO", OPTIMIZATION_BYPASS := "M_ZERO", TEST_STOP_BRAKE_TEST_AX_NUM := "DB1030_TEST_STOP".TEST_STP_TST_BRK_AX_12, PARAMETER_SET_0 := "M_ONE", PARAMETER_SET_1 := "DB2440_GLOBAL_DATA".AXIS_MANAGEMENT.CH5_PRMR_SET_SLCTN_A, PARAMETER_SET_2 :=, PARAMETER_SET_3 :=, MOVE_AXIS := "DB148_CLADDING_AXIS_C22".MOVE_AXIS, SAFE_ENABLED := "DB1018_SAFETY_TAGS".GROUP_3_C12.STO_Deactivate, FEED_HOLD_COND := "DB148_CLADDING_AXIS_C22".FEED_HOLD_COND, AX_TORQUE_ENABLE :=, MPP_AXIS_SELECTED :=, HMI_AXIS_SELECTED := "DB7224_HMI_AXES".AXIS_18_SELECTED, HMI_REQ_LINE :=, JOG_MINUS_REQ_NOT_FC18 :=, JOG_PLUS_REQ_NOT_FC18 :=, JOG_MINUS_REQ_FC18 :=, JOG_PLUS_REQ_FC18 :=, FC18_EXTERNAL_POS :=, AUTO_RETURN_COMMAND :=, AUTO_ADVANCE_COMMAND :=, DELETE_DISTANCE_TO_GO :=, FEED_OVERRIDE := "LBP_Chan5".A_FD_OR, FEED_OVER_ACTIVE := "LBP_Chan5".A_FD_ORA, READ_POS := "DB305_CH5_READ_AXES_POSITIONS".readDB.POSITION_AXIS_1, UNIT_ALARM := 2, STATION_ALARM := 2, AxisDB := "LBP_Axis18", MOTOR_ACTIVE =>, MOVE_AX =>, FEED_HOLD_CONDITIONS =>, ACTIVE_PARAMETER_SET =>, AX_NOT_REFERENCE_ALM => "DB426_ALARMS_WARNINGS".GENERAL."700120", AX_B_NOT_IN_PST_180_90_ALM =>, MAST_SLAVE_MODE_NOT_ACTIV_ALM =>, AX_TORQUE_EXCEEDED_ALM =>, AXIS_POS =>, HMI_MOTION_EXECUTABILITY_LEFT =>, HMI_MOTION_EXECUTABILITY_RIGHT =>, HMI_MOTION_END_POS_LEFT =>, HMI_MOTION_END_POS_RIGHT =>, HMI_MOTION_ACTIVE_LEFT =>, HMI_MOTION_ACTIVE_RIGHT =>)
   END_RUNG
   RUNG wire#powerrail
      Contact( "DB2102_INFEED_MODULE".INFEED_MODULE_READY_ENABLE_AXES )
      wire#w1
      Contact( "DB1018_SAFETY_TAGS".E_STOP_OK_OFF_DEL_2 )
      I_Contact( "DB1018_SAFETY_TAGS".E_STOP_OK )
   END_RUNG wire#w2
   RUNG wire#w1
      Contact( "DB1018_SAFETY_TAGS".E_STOP_OK )
      Contact( "DB1401_PNEUMATIC_SYSTEM".IN_SERVICE )
   END_RUNG wire#w2
   // the same network as SCL:
   "DB148_CLADDING_AXIS_C22"(OPTIONS_0 := 2#0000_0000,   // "FB32_AXIS"
                           OPTIONS_1 := 2#0000_0000,
                           SAFETY_BYPASS := "M_ZERO",
                           OPTIMIZATION_BYPASS := "M_ZERO",
                           AX_ENABLE := "DB2102_INFEED_MODULE".INFEED_MODULE_READY_ENABLE_AXES AND (("DB1018_SAFETY_TAGS".E_STOP_OK_OFF_DEL_2 AND NOT "DB1018_SAFETY_TAGS".E_STOP_OK) OR ("DB1018_SAFETY_TAGS".E_STOP_OK AND "DB1401_PNEUMATIC_SYSTEM".IN_SERVICE)),
                           TEST_STOP_BRAKE_TEST_AX_NUM := "DB1030_TEST_STOP".TEST_STP_TST_BRK_AX_12,
                           PARAMETER_SET_0 := "M_ONE",
                           PARAMETER_SET_1 := "DB2440_GLOBAL_DATA".AXIS_MANAGEMENT.CH5_PRMR_SET_SLCTN_A,
                           MOVE_AXIS := "DB148_CLADDING_AXIS_C22".MOVE_AXIS,
                           SAFE_ENABLED := "DB1018_SAFETY_TAGS".GROUP_3_C12.STO_Deactivate,
                           FEED_HOLD_COND := "DB148_CLADDING_AXIS_C22".FEED_HOLD_COND,
                           HMI_AXIS_SELECTED := "DB7224_HMI_AXES".AXIS_18_SELECTED,
                           FEED_OVERRIDE := "LBP_Chan5".A_FD_OR,
                           FEED_OVER_ACTIVE := "LBP_Chan5".A_FD_ORA,
                           READ_POS := "DB305_CH5_READ_AXES_POSITIONS".readDB.POSITION_AXIS_1,
                           UNIT_ALARM := 2,
                           STATION_ALARM := 2,
                           AxisDB := "LBP_Axis18",
                           AX_NOT_REFERENCE_ALM => "DB426_ALARMS_WARNINGS".GENERAL."700120");
END_REGION

REGION Network 19: AXIS C22 OPERATOR HELP
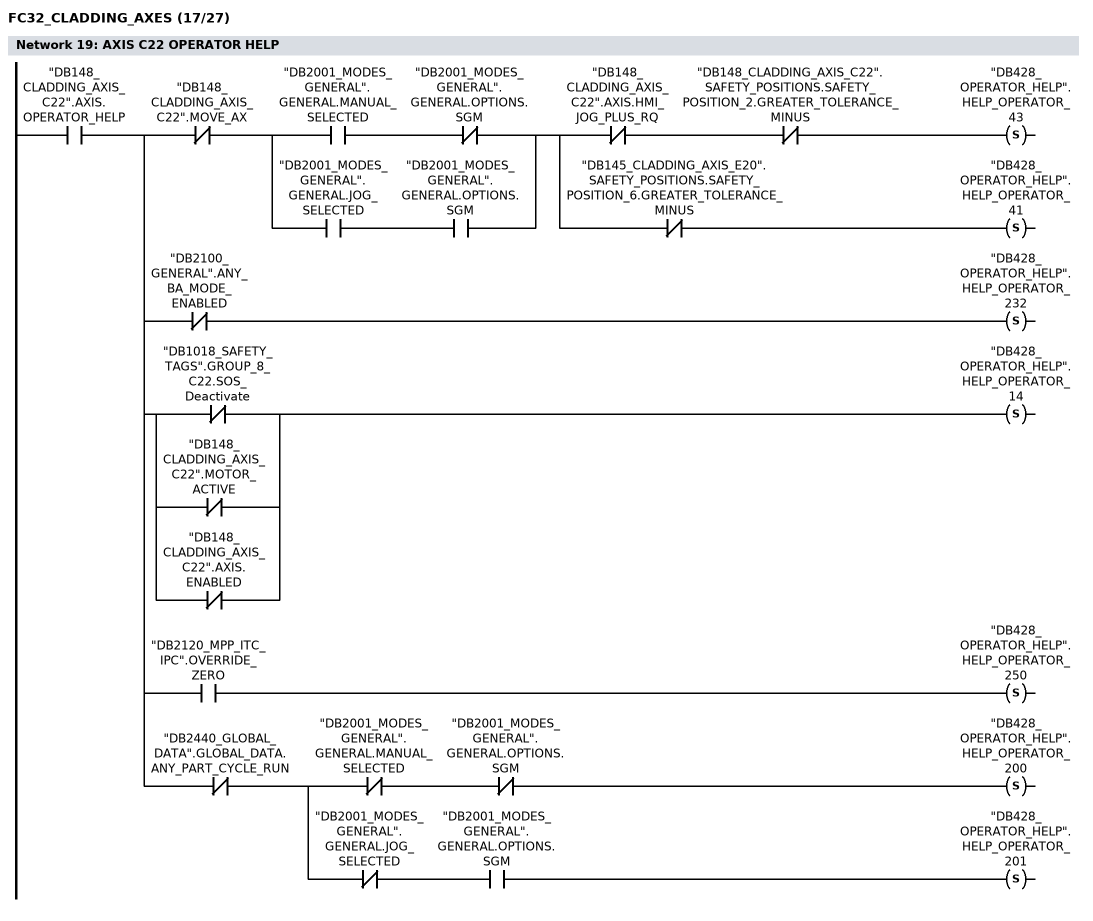
   RUNG wire#powerrail
      Contact( "DB148_CLADDING_AXIS_C22".AXIS.OPERATOR_HELP )
      wire#w1
      I_Contact( "DB148_CLADDING_AXIS_C22".MOVE_AX )
      wire#w2
      Contact( "DB2001_MODES_GENERAL".GENERAL.MANUAL_SELECTED )
      I_Contact( "DB2001_MODES_GENERAL".GENERAL.OPTIONS.SGM )
      wire#w3
      I_Contact( "DB148_CLADDING_AXIS_C22".AXIS.HMI_JOG_PLUS_RQ )
      I_Contact( "DB148_CLADDING_AXIS_C22".SAFETY_POSITIONS.SAFETY_POSITION_2.GREATER_TOLERANCE_MINUS )
      S_Coil( "DB428_OPERATOR_HELP".HELP_OPERATOR_43 )
   END_RUNG
   RUNG wire#w2
      Contact( "DB2001_MODES_GENERAL".GENERAL.JOG_SELECTED )
      Contact( "DB2001_MODES_GENERAL".GENERAL.OPTIONS.SGM )
   END_RUNG wire#w3
   RUNG wire#w3
      I_Contact( "DB145_CLADDING_AXIS_E20".SAFETY_POSITIONS.SAFETY_POSITION_6.GREATER_TOLERANCE_MINUS )
      S_Coil( "DB428_OPERATOR_HELP".HELP_OPERATOR_41 )
   END_RUNG
   RUNG wire#w1
      I_Contact( "DB2100_GENERAL".ANY_BA_MODE_ENABLED )
      S_Coil( "DB428_OPERATOR_HELP".HELP_OPERATOR_232 )
   END_RUNG
   RUNG wire#w1
      I_Contact( "DB1018_SAFETY_TAGS".GROUP_8_C22.SOS_Deactivate )
      wire#w4
      S_Coil( "DB428_OPERATOR_HELP".HELP_OPERATOR_14 )
   END_RUNG
   RUNG wire#w1
      I_Contact( "DB148_CLADDING_AXIS_C22".MOTOR_ACTIVE )
   END_RUNG wire#w4
   RUNG wire#w1
      I_Contact( "DB148_CLADDING_AXIS_C22".AXIS.ENABLED )
   END_RUNG wire#w4
   RUNG wire#w1
      Contact( "DB2120_MPP_ITC_IPC".OVERRIDE_ZERO )
      S_Coil( "DB428_OPERATOR_HELP".HELP_OPERATOR_250 )
   END_RUNG
   RUNG wire#w1
      I_Contact( "DB2440_GLOBAL_DATA".GLOBAL_DATA.ANY_PART_CYCLE_RUN )
      wire#w5
      I_Contact( "DB2001_MODES_GENERAL".GENERAL.MANUAL_SELECTED )
      I_Contact( "DB2001_MODES_GENERAL".GENERAL.OPTIONS.SGM )
      S_Coil( "DB428_OPERATOR_HELP".HELP_OPERATOR_200 )
   END_RUNG
   RUNG wire#w5
      I_Contact( "DB2001_MODES_GENERAL".GENERAL.JOG_SELECTED )
      Contact( "DB2001_MODES_GENERAL".GENERAL.OPTIONS.SGM )
      S_Coil( "DB428_OPERATOR_HELP".HELP_OPERATOR_201 )
   END_RUNG
   // the same network as SCL:
   #_w1 := "DB148_CLADDING_AXIS_C22".AXIS.OPERATOR_HELP AND NOT "DB148_CLADDING_AXIS_C22".MOVE_AX AND (("DB2001_MODES_GENERAL".GENERAL.MANUAL_SELECTED AND NOT "DB2001_MODES_GENERAL".GENERAL.OPTIONS.SGM) OR ("DB2001_MODES_GENERAL".GENERAL.JOG_SELECTED AND "DB2001_MODES_GENERAL".GENERAL.OPTIONS.SGM));
   IF #_w1 AND NOT "DB148_CLADDING_AXIS_C22".AXIS.HMI_JOG_PLUS_RQ AND NOT "DB148_CLADDING_AXIS_C22".SAFETY_POSITIONS.SAFETY_POSITION_2.GREATER_TOLERANCE_MINUS THEN
       "DB428_OPERATOR_HELP".HELP_OPERATOR_43 := TRUE;
   END_IF;
   IF #_w1 AND NOT "DB145_CLADDING_AXIS_E20".SAFETY_POSITIONS.SAFETY_POSITION_6.GREATER_TOLERANCE_MINUS THEN
       "DB428_OPERATOR_HELP".HELP_OPERATOR_41 := TRUE;
   END_IF;
   IF "DB148_CLADDING_AXIS_C22".AXIS.OPERATOR_HELP AND NOT "DB2100_GENERAL".ANY_BA_MODE_ENABLED THEN
       "DB428_OPERATOR_HELP".HELP_OPERATOR_232 := TRUE;
   END_IF;
   IF "DB148_CLADDING_AXIS_C22".AXIS.OPERATOR_HELP AND (NOT "DB1018_SAFETY_TAGS".GROUP_8_C22.SOS_Deactivate OR NOT "DB148_CLADDING_AXIS_C22".MOTOR_ACTIVE OR NOT "DB148_CLADDING_AXIS_C22".AXIS.ENABLED) THEN
       "DB428_OPERATOR_HELP".HELP_OPERATOR_14 := TRUE;
   END_IF;
   IF "DB148_CLADDING_AXIS_C22".AXIS.OPERATOR_HELP AND "DB2120_MPP_ITC_IPC".OVERRIDE_ZERO THEN
       "DB428_OPERATOR_HELP".HELP_OPERATOR_250 := TRUE;
   END_IF;
   #_w2 := "DB148_CLADDING_AXIS_C22".AXIS.OPERATOR_HELP AND NOT "DB2440_GLOBAL_DATA".GLOBAL_DATA.ANY_PART_CYCLE_RUN;
   IF #_w2 AND NOT "DB2001_MODES_GENERAL".GENERAL.MANUAL_SELECTED AND NOT "DB2001_MODES_GENERAL".GENERAL.OPTIONS.SGM THEN
       "DB428_OPERATOR_HELP".HELP_OPERATOR_200 := TRUE;
   END_IF;
   IF #_w2 AND NOT "DB2001_MODES_GENERAL".GENERAL.JOG_SELECTED AND "DB2001_MODES_GENERAL".GENERAL.OPTIONS.SGM THEN
       "DB428_OPERATOR_HELP".HELP_OPERATOR_201 := TRUE;
   END_IF;
END_REGION

REGION Network 20: AXIS X23 MOVE AXIS AND FEED HOLD CONDITIONS
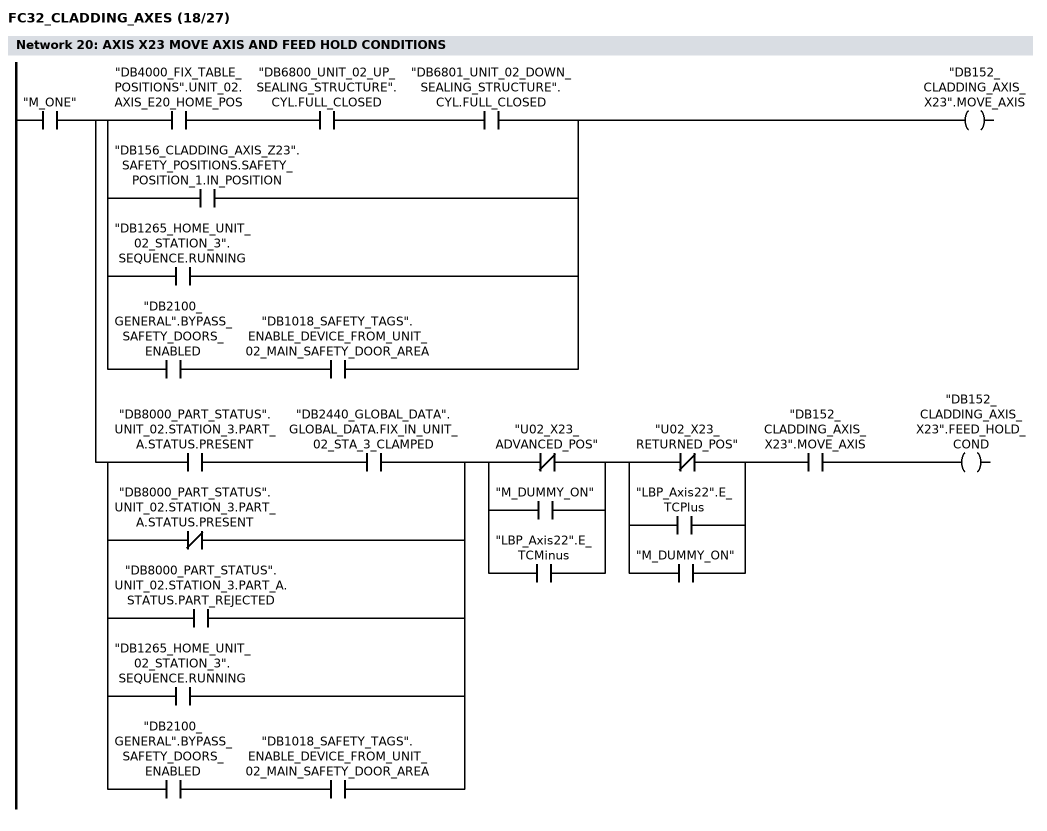
   RUNG wire#powerrail
      Contact( "M_ONE" )
      wire#w1
      Contact( "DB4000_FIX_TABLE_POSITIONS".UNIT_02.AXIS_E20_HOME_POS )
      Contact( "DB6800_UNIT_02_UP_SEALING_STRUCTURE".CYL.FULL_CLOSED )
      Contact( "DB6801_UNIT_02_DOWN_SEALING_STRUCTURE".CYL.FULL_CLOSED )
      wire#w2
      Coil( "DB152_CLADDING_AXIS_X23".MOVE_AXIS )
   END_RUNG
   RUNG wire#w1
      Contact( "DB156_CLADDING_AXIS_Z23".SAFETY_POSITIONS.SAFETY_POSITION_1.IN_POSITION )
   END_RUNG wire#w2
   RUNG wire#w1
      Contact( "DB1265_HOME_UNIT_02_STATION_3".SEQUENCE.RUNNING )
   END_RUNG wire#w2
   RUNG wire#w1
      Contact( "DB2100_GENERAL".BYPASS_SAFETY_DOORS_ENABLED )
      Contact( "DB1018_SAFETY_TAGS".ENABLE_DEVICE_FROM_UNIT_02_MAIN_SAFETY_DOOR_AREA )
   END_RUNG wire#w2
   RUNG wire#w1
      Contact( "DB8000_PART_STATUS".UNIT_02.STATION_3.PART_A.STATUS.PRESENT )
      Contact( "DB2440_GLOBAL_DATA".GLOBAL_DATA.FIX_IN_UNIT_02_STA_3_CLAMPED )
      wire#w3
      I_Contact( "U02_X23_ADVANCED_POS" )
      wire#w4
      I_Contact( "U02_X23_RETURNED_POS" )
      wire#w5
      Contact( "DB152_CLADDING_AXIS_X23".MOVE_AXIS )
      Coil( "DB152_CLADDING_AXIS_X23".FEED_HOLD_COND )
   END_RUNG
   RUNG wire#w1
      I_Contact( "DB8000_PART_STATUS".UNIT_02.STATION_3.PART_A.STATUS.PRESENT )
   END_RUNG wire#w3
   RUNG wire#w1
      Contact( "DB8000_PART_STATUS".UNIT_02.STATION_3.PART_A.STATUS.PART_REJECTED )
   END_RUNG wire#w3
   RUNG wire#w1
      Contact( "DB1265_HOME_UNIT_02_STATION_3".SEQUENCE.RUNNING )
   END_RUNG wire#w3
   RUNG wire#w1
      Contact( "DB2100_GENERAL".BYPASS_SAFETY_DOORS_ENABLED )
      Contact( "DB1018_SAFETY_TAGS".ENABLE_DEVICE_FROM_UNIT_02_MAIN_SAFETY_DOOR_AREA )
   END_RUNG wire#w3
   RUNG wire#w3
      Contact( "M_DUMMY_ON" )
   END_RUNG wire#w4
   RUNG wire#w3
      Contact( "LBP_Axis22".E_TCMinus )
   END_RUNG wire#w4
   RUNG wire#w4
      Contact( "LBP_Axis22".E_TCPlus )
   END_RUNG wire#w5
   RUNG wire#w4
      Contact( "M_DUMMY_ON" )
   END_RUNG wire#w5
   // the same network as SCL:
   "DB152_CLADDING_AXIS_X23".MOVE_AXIS := "M_ONE" AND (("DB4000_FIX_TABLE_POSITIONS".UNIT_02.AXIS_E20_HOME_POS AND "DB6800_UNIT_02_UP_SEALING_STRUCTURE".CYL.FULL_CLOSED AND "DB6801_UNIT_02_DOWN_SEALING_STRUCTURE".CYL.FULL_CLOSED) OR "DB156_CLADDING_AXIS_Z23".SAFETY_POSITIONS.SAFETY_POSITION_1.IN_POSITION OR "DB1265_HOME_UNIT_02_STATION_3".SEQUENCE.RUNNING OR ("DB2100_GENERAL".BYPASS_SAFETY_DOORS_ENABLED AND "DB1018_SAFETY_TAGS".ENABLE_DEVICE_FROM_UNIT_02_MAIN_SAFETY_DOOR_AREA));
   "DB152_CLADDING_AXIS_X23".FEED_HOLD_COND := "M_ONE" AND (("DB8000_PART_STATUS".UNIT_02.STATION_3.PART_A.STATUS.PRESENT AND "DB2440_GLOBAL_DATA".GLOBAL_DATA.FIX_IN_UNIT_02_STA_3_CLAMPED) OR NOT "DB8000_PART_STATUS".UNIT_02.STATION_3.PART_A.STATUS.PRESENT OR "DB8000_PART_STATUS".UNIT_02.STATION_3.PART_A.STATUS.PART_REJECTED OR "DB1265_HOME_UNIT_02_STATION_3".SEQUENCE.RUNNING OR ("DB2100_GENERAL".BYPASS_SAFETY_DOORS_ENABLED AND "DB1018_SAFETY_TAGS".ENABLE_DEVICE_FROM_UNIT_02_MAIN_SAFETY_DOOR_AREA)) AND (NOT "U02_X23_ADVANCED_POS" OR "M_DUMMY_ON" OR "LBP_Axis22".E_TCMinus) AND (NOT "U02_X23_RETURNED_POS" OR "LBP_Axis22".E_TCPlus OR "M_DUMMY_ON") AND "DB152_CLADDING_AXIS_X23".MOVE_AXIS;
END_REGION

REGION Network 21: CALL FB32 AXIS X23
   // 2#0000_0001 OPTIONS 0 BIT 0 MEASURING SYSTEM 2 OPTION
   // 2#0000_0010 OPTIONS 0 BIT 1 ENABLE FC18 OPTION
   // 2#0000_0100 OPTIONS 0 BIT 2 FC18 EXTERNAL POSITION OPTION
   // 2#0000_1000 OPTIONS 0 BIT 3 AXIS B ENABLE FAULTS OPTION
   // 2#0001_0000 OPTIONS 0 BIT 4 SPARE OPTION
   // 2#0010_0000 OPTIONS 0 BIT 5 SPARE OPTION
   // 2#0100_0000 OPTIONS 0 BIT 6 SPARE OPTION
   // 2#1000_0000 OPTIONS 0 BIT 7 SPARE OPTION
   // 
   // 2#0000_0001 OPTIONS 1 BIT 0 AXIS ROLLER OPTION
   // 2#0000_0010 OPTIONS 1 BIT 1 MASTER AXIS OPTION
   // 2#0000_0100 OPTIONS 1 BIT 2 SLAVE AXIS OPTION
   // 2#0000_1000 OPTIONS 1 BIT 3 MASTER-SLAVE AXES INDEPENDENT MOVEMENT WITH HT10 OPTION
   // 2#0001_0000 OPTIONS 1 BIT 4 GANTRY MODE MASTER AXIS OPTION
   // 2#0010_0000 OPTIONS 1 BIT 5 SPARE OPTION
   // 2#0100_0000 OPTIONS 1 BIT 6 SPARE OPTION
   // 2#1000_0000 OPTIONS 1 BIT 7 SPARE OPTION
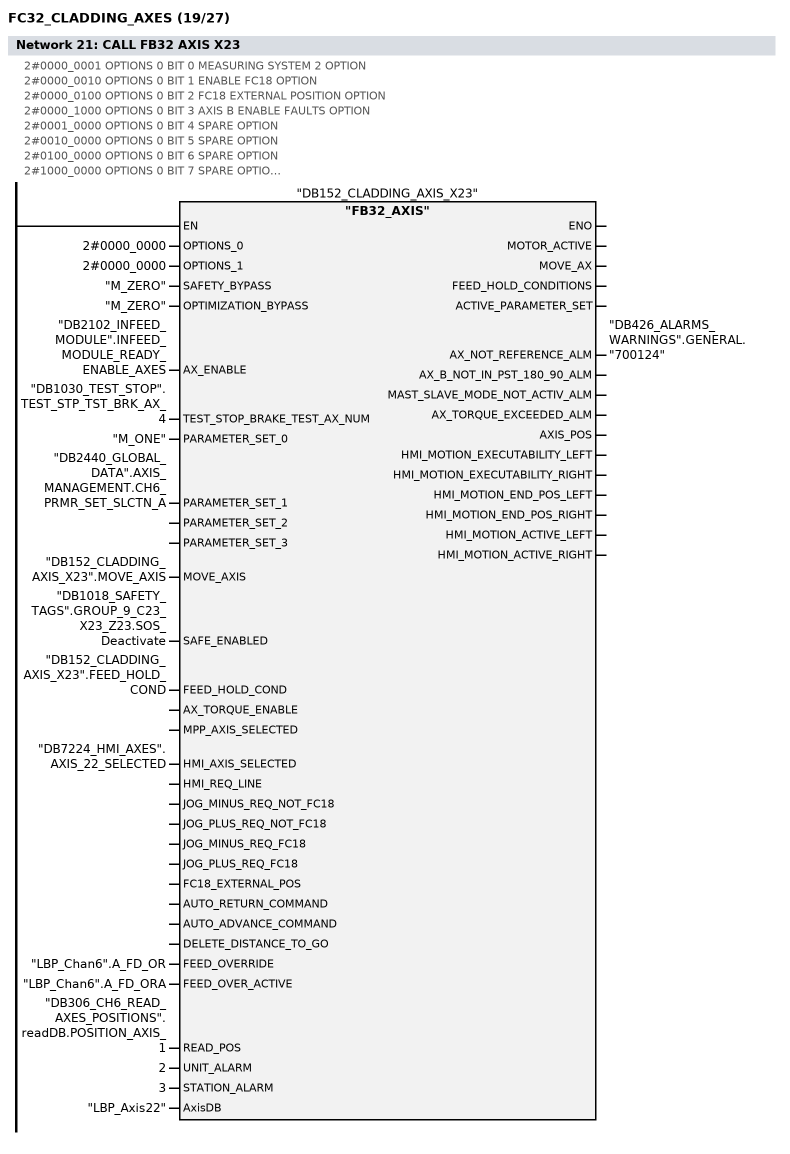
   RUNG wire#powerrail
      "DB152_CLADDING_AXIS_X23"(OPTIONS_0 := 2#0000_0000, OPTIONS_1 := 2#0000_0000, SAFETY_BYPASS := "M_ZERO", OPTIMIZATION_BYPASS := "M_ZERO", AX_ENABLE := "DB2102_INFEED_MODULE".INFEED_MODULE_READY_ENABLE_AXES, TEST_STOP_BRAKE_TEST_AX_NUM := "DB1030_TEST_STOP".TEST_STP_TST_BRK_AX_4, PARAMETER_SET_0 := "M_ONE", PARAMETER_SET_1 := "DB2440_GLOBAL_DATA".AXIS_MANAGEMENT.CH6_PRMR_SET_SLCTN_A, PARAMETER_SET_2 :=, PARAMETER_SET_3 :=, MOVE_AXIS := "DB152_CLADDING_AXIS_X23".MOVE_AXIS, SAFE_ENABLED := "DB1018_SAFETY_TAGS".GROUP_9_C23_X23_Z23.SOS_Deactivate, FEED_HOLD_COND := "DB152_CLADDING_AXIS_X23".FEED_HOLD_COND, AX_TORQUE_ENABLE :=, MPP_AXIS_SELECTED :=, HMI_AXIS_SELECTED := "DB7224_HMI_AXES".AXIS_22_SELECTED, HMI_REQ_LINE :=, JOG_MINUS_REQ_NOT_FC18 :=, JOG_PLUS_REQ_NOT_FC18 :=, JOG_MINUS_REQ_FC18 :=, JOG_PLUS_REQ_FC18 :=, FC18_EXTERNAL_POS :=, AUTO_RETURN_COMMAND :=, AUTO_ADVANCE_COMMAND :=, DELETE_DISTANCE_TO_GO :=, FEED_OVERRIDE := "LBP_Chan6".A_FD_OR, FEED_OVER_ACTIVE := "LBP_Chan6".A_FD_ORA, READ_POS := "DB306_CH6_READ_AXES_POSITIONS".readDB.POSITION_AXIS_1, UNIT_ALARM := 2, STATION_ALARM := 3, AxisDB := "LBP_Axis22", MOTOR_ACTIVE =>, MOVE_AX =>, FEED_HOLD_CONDITIONS =>, ACTIVE_PARAMETER_SET =>, AX_NOT_REFERENCE_ALM => "DB426_ALARMS_WARNINGS".GENERAL."700124", AX_B_NOT_IN_PST_180_90_ALM =>, MAST_SLAVE_MODE_NOT_ACTIV_ALM =>, AX_TORQUE_EXCEEDED_ALM =>, AXIS_POS =>, HMI_MOTION_EXECUTABILITY_LEFT =>, HMI_MOTION_EXECUTABILITY_RIGHT =>, HMI_MOTION_END_POS_LEFT =>, HMI_MOTION_END_POS_RIGHT =>, HMI_MOTION_ACTIVE_LEFT =>, HMI_MOTION_ACTIVE_RIGHT =>)
   END_RUNG
   // the same network as SCL:
   "DB152_CLADDING_AXIS_X23"(OPTIONS_0 := 2#0000_0000,   // "FB32_AXIS"
                           OPTIONS_1 := 2#0000_0000,
                           SAFETY_BYPASS := "M_ZERO",
                           OPTIMIZATION_BYPASS := "M_ZERO",
                           AX_ENABLE := "DB2102_INFEED_MODULE".INFEED_MODULE_READY_ENABLE_AXES,
                           TEST_STOP_BRAKE_TEST_AX_NUM := "DB1030_TEST_STOP".TEST_STP_TST_BRK_AX_4,
                           PARAMETER_SET_0 := "M_ONE",
                           PARAMETER_SET_1 := "DB2440_GLOBAL_DATA".AXIS_MANAGEMENT.CH6_PRMR_SET_SLCTN_A,
                           MOVE_AXIS := "DB152_CLADDING_AXIS_X23".MOVE_AXIS,
                           SAFE_ENABLED := "DB1018_SAFETY_TAGS".GROUP_9_C23_X23_Z23.SOS_Deactivate,
                           FEED_HOLD_COND := "DB152_CLADDING_AXIS_X23".FEED_HOLD_COND,
                           HMI_AXIS_SELECTED := "DB7224_HMI_AXES".AXIS_22_SELECTED,
                           FEED_OVERRIDE := "LBP_Chan6".A_FD_OR,
                           FEED_OVER_ACTIVE := "LBP_Chan6".A_FD_ORA,
                           READ_POS := "DB306_CH6_READ_AXES_POSITIONS".readDB.POSITION_AXIS_1,
                           UNIT_ALARM := 2,
                           STATION_ALARM := 3,
                           AxisDB := "LBP_Axis22",
                           AX_NOT_REFERENCE_ALM => "DB426_ALARMS_WARNINGS".GENERAL."700124");
END_REGION

REGION Network 22: AXIS X23 OPERATOR HELP
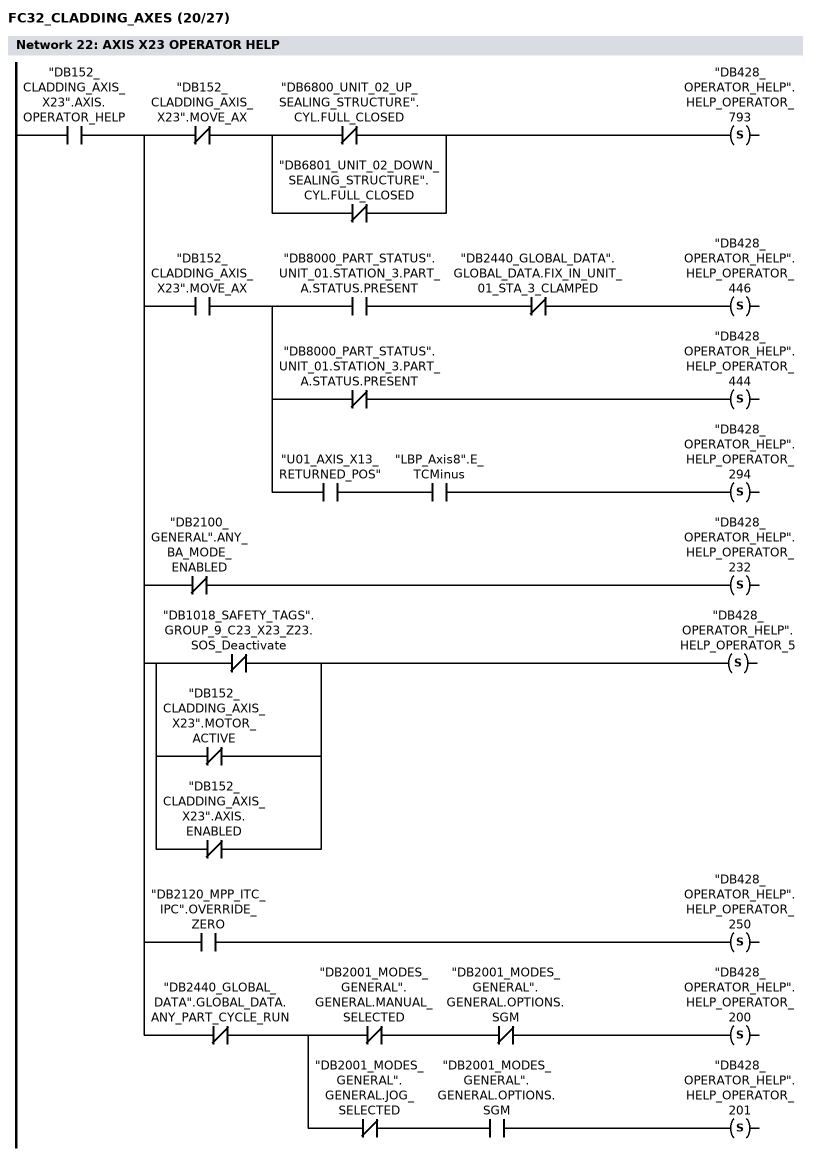
   RUNG wire#powerrail
      Contact( "DB152_CLADDING_AXIS_X23".AXIS.OPERATOR_HELP )
      wire#w1
      I_Contact( "DB152_CLADDING_AXIS_X23".MOVE_AX )
      wire#w2
      I_Contact( "DB6800_UNIT_02_UP_SEALING_STRUCTURE".CYL.FULL_CLOSED )
      wire#w3
      S_Coil( "DB428_OPERATOR_HELP".HELP_OPERATOR_793 )
   END_RUNG
   RUNG wire#w2
      I_Contact( "DB6801_UNIT_02_DOWN_SEALING_STRUCTURE".CYL.FULL_CLOSED )
   END_RUNG wire#w3
   RUNG wire#w1
      Contact( "DB152_CLADDING_AXIS_X23".MOVE_AX )
      wire#w4
      Contact( "DB8000_PART_STATUS".UNIT_01.STATION_3.PART_A.STATUS.PRESENT )
      I_Contact( "DB2440_GLOBAL_DATA".GLOBAL_DATA.FIX_IN_UNIT_01_STA_3_CLAMPED )
      S_Coil( "DB428_OPERATOR_HELP".HELP_OPERATOR_446 )
   END_RUNG
   RUNG wire#w4
      I_Contact( "DB8000_PART_STATUS".UNIT_01.STATION_3.PART_A.STATUS.PRESENT )
      S_Coil( "DB428_OPERATOR_HELP".HELP_OPERATOR_444 )
   END_RUNG
   RUNG wire#w4
      Contact( "U01_AXIS_X13_RETURNED_POS" )
      Contact( "LBP_Axis8".E_TCMinus )
      S_Coil( "DB428_OPERATOR_HELP".HELP_OPERATOR_294 )
   END_RUNG
   RUNG wire#w1
      I_Contact( "DB2100_GENERAL".ANY_BA_MODE_ENABLED )
      S_Coil( "DB428_OPERATOR_HELP".HELP_OPERATOR_232 )
   END_RUNG
   RUNG wire#w1
      I_Contact( "DB1018_SAFETY_TAGS".GROUP_9_C23_X23_Z23.SOS_Deactivate )
      wire#w5
      S_Coil( "DB428_OPERATOR_HELP".HELP_OPERATOR_5 )
   END_RUNG
   RUNG wire#w1
      I_Contact( "DB152_CLADDING_AXIS_X23".MOTOR_ACTIVE )
   END_RUNG wire#w5
   RUNG wire#w1
      I_Contact( "DB152_CLADDING_AXIS_X23".AXIS.ENABLED )
   END_RUNG wire#w5
   RUNG wire#w1
      Contact( "DB2120_MPP_ITC_IPC".OVERRIDE_ZERO )
      S_Coil( "DB428_OPERATOR_HELP".HELP_OPERATOR_250 )
   END_RUNG
   RUNG wire#w1
      I_Contact( "DB2440_GLOBAL_DATA".GLOBAL_DATA.ANY_PART_CYCLE_RUN )
      wire#w6
      I_Contact( "DB2001_MODES_GENERAL".GENERAL.MANUAL_SELECTED )
      I_Contact( "DB2001_MODES_GENERAL".GENERAL.OPTIONS.SGM )
      S_Coil( "DB428_OPERATOR_HELP".HELP_OPERATOR_200 )
   END_RUNG
   RUNG wire#w6
      I_Contact( "DB2001_MODES_GENERAL".GENERAL.JOG_SELECTED )
      Contact( "DB2001_MODES_GENERAL".GENERAL.OPTIONS.SGM )
      S_Coil( "DB428_OPERATOR_HELP".HELP_OPERATOR_201 )
   END_RUNG
   // the same network as SCL:
   IF "DB152_CLADDING_AXIS_X23".AXIS.OPERATOR_HELP AND NOT "DB152_CLADDING_AXIS_X23".MOVE_AX AND (NOT "DB6800_UNIT_02_UP_SEALING_STRUCTURE".CYL.FULL_CLOSED OR NOT "DB6801_UNIT_02_DOWN_SEALING_STRUCTURE".CYL.FULL_CLOSED) THEN
       "DB428_OPERATOR_HELP".HELP_OPERATOR_793 := TRUE;
   END_IF;
   #_w1 := "DB152_CLADDING_AXIS_X23".AXIS.OPERATOR_HELP AND "DB152_CLADDING_AXIS_X23".MOVE_AX;
   IF #_w1 AND "DB8000_PART_STATUS".UNIT_01.STATION_3.PART_A.STATUS.PRESENT AND NOT "DB2440_GLOBAL_DATA".GLOBAL_DATA.FIX_IN_UNIT_01_STA_3_CLAMPED THEN
       "DB428_OPERATOR_HELP".HELP_OPERATOR_446 := TRUE;
   END_IF;
   IF #_w1 AND NOT "DB8000_PART_STATUS".UNIT_01.STATION_3.PART_A.STATUS.PRESENT THEN
       "DB428_OPERATOR_HELP".HELP_OPERATOR_444 := TRUE;
   END_IF;
   IF #_w1 AND "U01_AXIS_X13_RETURNED_POS" AND "LBP_Axis8".E_TCMinus THEN
       "DB428_OPERATOR_HELP".HELP_OPERATOR_294 := TRUE;
   END_IF;
   IF "DB152_CLADDING_AXIS_X23".AXIS.OPERATOR_HELP AND NOT "DB2100_GENERAL".ANY_BA_MODE_ENABLED THEN
       "DB428_OPERATOR_HELP".HELP_OPERATOR_232 := TRUE;
   END_IF;
   IF "DB152_CLADDING_AXIS_X23".AXIS.OPERATOR_HELP AND (NOT "DB1018_SAFETY_TAGS".GROUP_9_C23_X23_Z23.SOS_Deactivate OR NOT "DB152_CLADDING_AXIS_X23".MOTOR_ACTIVE OR NOT "DB152_CLADDING_AXIS_X23".AXIS.ENABLED) THEN
       "DB428_OPERATOR_HELP".HELP_OPERATOR_5 := TRUE;
   END_IF;
   IF "DB152_CLADDING_AXIS_X23".AXIS.OPERATOR_HELP AND "DB2120_MPP_ITC_IPC".OVERRIDE_ZERO THEN
       "DB428_OPERATOR_HELP".HELP_OPERATOR_250 := TRUE;
   END_IF;
   #_w2 := "DB152_CLADDING_AXIS_X23".AXIS.OPERATOR_HELP AND NOT "DB2440_GLOBAL_DATA".GLOBAL_DATA.ANY_PART_CYCLE_RUN;
   IF #_w2 AND NOT "DB2001_MODES_GENERAL".GENERAL.MANUAL_SELECTED AND NOT "DB2001_MODES_GENERAL".GENERAL.OPTIONS.SGM THEN
       "DB428_OPERATOR_HELP".HELP_OPERATOR_200 := TRUE;
   END_IF;
   IF #_w2 AND NOT "DB2001_MODES_GENERAL".GENERAL.JOG_SELECTED AND "DB2001_MODES_GENERAL".GENERAL.OPTIONS.SGM THEN
       "DB428_OPERATOR_HELP".HELP_OPERATOR_201 := TRUE;
   END_IF;
END_REGION

